REGION Network 6: Print Logic
   RUNG wire#powerrail
      Contact( #AlwaysTrue )
      wire#w1
      P_Contact(operand := #Selected, bit := #RE3)
      { S7_GenerateENO := "TRUE" } Move(in := 1, out1 => #PrintWord)   // 'STARTED'
      S_Move(in := #STATUS1, out => #PrintStatus)
      S_Coil( #PrintTriggerTemp )
   END_RUNG
   RUNG wire#w1
      Contact( #Selected )
      N_Contact(operand := #Running, bit := #RE4)
      I_Contact( #Close )
      { S7_GenerateENO := "TRUE" } Move(in := 2, out1 => #PrintWord)   // 'PAUSED'
      S_Move(in := #STATUS2, out => #PrintStatus)
      wire#w2
      S_Coil( #PrintTriggerTemp )
   END_RUNG
   RUNG wire#w2
      S_Coil( #Paused )
   END_RUNG
   RUNG wire#w1
      Contact( #Selected )
      Contact( #Paused )
      P_Contact(operand := #Running, bit := #RE5)
      { S7_GenerateENO := "TRUE" } Move(in := 3, out1 => #PrintWord)   // 'RESUMED'
      S_Move(in := #STATUS3, out => #PrintStatus)
      wire#w3
      S_Coil( #PrintTriggerTemp )
   END_RUNG
   RUNG wire#w3
      R_Coil( #Paused )
   END_RUNG
   RUNG wire#w1
      P_Contact(operand := #SpargingOver, bit := #RE6)
      { S7_GenerateENO := "TRUE" } Move(in := 4, out1 => #PrintWord)   // 'OVER'
      S_Move(in := #STATUS4, out => #PrintStatus)
      S_Coil( #PrintTriggerTemp )
   END_RUNG
   RUNG wire#w1
      P_Contact(operand := #Close, bit := #RE7)
      { S7_GenerateENO := "TRUE" } Move(in := 5, out1 => #PrintWord)   // 'RESETED'
      S_Move(in := #STATUS5, out => #PrintStatus)
      S_Coil( #PrintTriggerTemp )
   END_RUNG
   RUNG wire#w1
      I_Contact( #Selected )
      R_Coil( #Paused )
   END_RUNG
   RUNG wire#w1
      Contact( #PrintTriggerTemp )
      Coil( #PrintTrigger )
   END_RUNG
   // the same network as SCL:
   // ENO of a box is taken as its EN; it also drops when the box reports an error
   #_w1 := #AlwaysTrue AND #Selected AND NOT #RE3;   // rising edge of #Selected
   #RE3 := #Selected;
   IF #_w1 THEN
       #PrintWord := 1;   // 'STARTED'
       #PrintStatus := #STATUS1;
       #PrintTriggerTemp := TRUE;
   END_IF;
   #_w2 := #AlwaysTrue AND #Selected AND NOT #Running AND #RE4;   // falling edge of #Running
   #RE4 := #Running;
   IF #_w2 AND NOT #Close THEN
       #PrintWord := 2;   // 'PAUSED'
       #PrintStatus := #STATUS2;
       #PrintTriggerTemp := TRUE;
       #Paused := TRUE;
   END_IF;
   #_w3 := #AlwaysTrue AND #Selected AND #Paused AND #Running AND NOT #RE5;   // rising edge of #Running
   #RE5 := #Running;
   IF #_w3 THEN
       #PrintWord := 3;   // 'RESUMED'
       #PrintStatus := #STATUS3;
       #PrintTriggerTemp := TRUE;
       #Paused := FALSE;
   END_IF;
   #_w4 := #AlwaysTrue AND #SpargingOver AND NOT #RE6;   // rising edge of #SpargingOver
   #RE6 := #SpargingOver;
   IF #_w4 THEN
       #PrintWord := 4;   // 'OVER'
       #PrintStatus := #STATUS4;
       #PrintTriggerTemp := TRUE;
   END_IF;
   #_w5 := #AlwaysTrue AND #Close AND NOT #RE7;   // rising edge of #Close
   #RE7 := #Close;
   IF #_w5 THEN
       #PrintWord := 5;   // 'RESETED'
       #PrintStatus := #STATUS5;
       #PrintTriggerTemp := TRUE;
   END_IF;
   IF #AlwaysTrue AND NOT #Selected THEN #Paused := FALSE; END_IF;
   #PrintTrigger := #AlwaysTrue AND #PrintTriggerTemp;
END_REGION

REGION Network 7: Print Trigger Reset
   RUNG wire#powerrail
      Contact( #PrintTriggerTemp )
      { S7_Templates := "time_type := Time" } #PrintTriggerResetTimer.TON(pt := T#1s, et =>)
      R_Coil( #PrintTriggerTemp )
   END_RUNG
   // the same network as SCL:
   #PrintTriggerResetTimer(IN := #PrintTriggerTemp, PT := T#1s);   // TON
   IF #PrintTriggerResetTimer.Q THEN #PrintTriggerTemp := FALSE; END_IF;
END_REGION

REGION Network 8: Button Reset
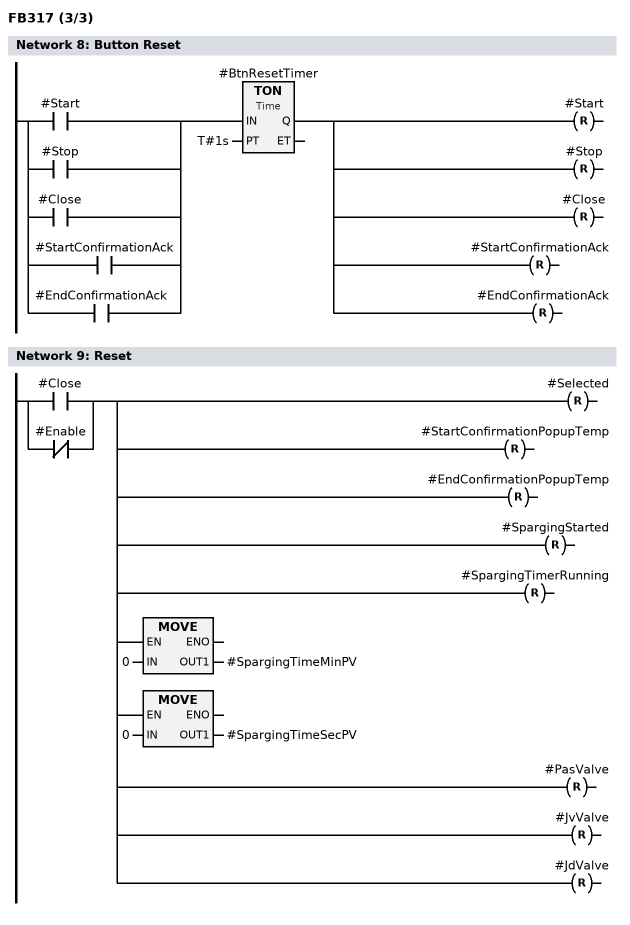
   RUNG wire#powerrail
      Contact( #Start )
      wire#w1
      { S7_Templates := "time_type := Time" } #BtnResetTimer.TON(pt := T#1s, et =>)
      wire#w2
      R_Coil( #Start )
   END_RUNG
   RUNG wire#powerrail
      Contact( #Stop )
   END_RUNG wire#w1
   RUNG wire#powerrail
      Contact( #Close )
   END_RUNG wire#w1
   RUNG wire#powerrail
      Contact( #StartConfirmationAck )
   END_RUNG wire#w1
   RUNG wire#powerrail
      Contact( #EndConfirmationAck )
   END_RUNG wire#w1
   RUNG wire#w2
      R_Coil( #Stop )
   END_RUNG
   RUNG wire#w2
      R_Coil( #Close )
   END_RUNG
   RUNG wire#w2
      R_Coil( #StartConfirmationAck )
   END_RUNG
   RUNG wire#w2
      R_Coil( #EndConfirmationAck )
   END_RUNG
   // the same network as SCL:
   #BtnResetTimer(IN := #Start OR #Stop OR #Close OR #StartConfirmationAck OR #EndConfirmationAck, PT := T#1s);   // TON
   IF #BtnResetTimer.Q THEN
       #Start := FALSE;
       #Stop := FALSE;
       #Close := FALSE;
       #StartConfirmationAck := FALSE;
       #EndConfirmationAck := FALSE;
   END_IF;
END_REGION

REGION Network 9: Reset
   RUNG wire#powerrail
      Contact( #Close )
      wire#w1
      R_Coil( #Selected )
   END_RUNG
   RUNG wire#powerrail
      I_Contact( #Enable )
   END_RUNG wire#w1
   RUNG wire#w1
      R_Coil( #StartConfirmationPopupTemp )
   END_RUNG
   RUNG wire#w1
      R_Coil( #EndConfirmationPopupTemp )
   END_RUNG
   RUNG wire#w1
      R_Coil( #SpargingStarted )
   END_RUNG
   RUNG wire#w1
      R_Coil( #SpargingTimerRunning )
   END_RUNG
   RUNG wire#w1
      { S7_GenerateENO := "TRUE" } Move(in := 0, out1 => #SpargingTimeMinPV)
   END_RUNG
   RUNG wire#w1
      { S7_GenerateENO := "TRUE" } Move(in := 0, out1 => #SpargingTimeSecPV)
   END_RUNG
   RUNG wire#w1
      R_Coil( #PasValve )
   END_RUNG
   RUNG wire#w1
      R_Coil( #JvValve )
   END_RUNG
   RUNG wire#w1
      R_Coil( #JdValve )
   END_RUNG
   // the same network as SCL:
   IF #Close OR NOT #Enable THEN
       #Selected := FALSE;
       #StartConfirmationPopupTemp := FALSE;
       #EndConfirmationPopupTemp := FALSE;
       #SpargingStarted := FALSE;
       #SpargingTimerRunning := FALSE;
       #SpargingTimeMinPV := 0;
       #SpargingTimeSecPV := 0;
       #PasValve := FALSE;
       #JvValve := FALSE;
       #JdValve := FALSE;
   END_IF;
END_REGION
END_FUNCTION_BLOCK

FUNCTION_BLOCK "BATCH LINE PRINT"   // FB5, LAD
{ S7_Optimized_Access := 'TRUE' }
// stored: MemoryReserve 100, SetENOAutomatically false
   VAR_INPUT
      PrintInetrval : Int;
      SecPulse : Bool;
   END_VAR
   VAR_IN_OUT
      ResetBatchTimer : Bool;
      BatchSelected : Bool;
   END_VAR
   VAR
      IEC_Counter_0_Instance { S7_SetPoint := 'True'} : CTU_INT;
   END_VAR
BEGIN

REGION Network 2
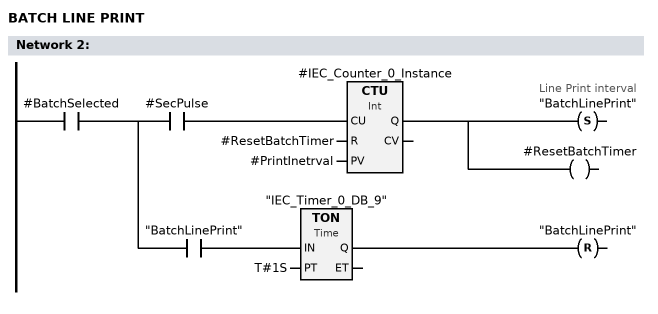
   RUNG wire#powerrail
      Contact( #BatchSelected )
      wire#w1
      Contact( #SecPulse )
      { S7_Templates := "value_type := Int" } #IEC_Counter_0_Instance.CTU(r := #ResetBatchTimer, pv := #PrintInetrval, cv =>)
      wire#w2
      S_Coil( "BatchLinePrint" )   // Line Print interval
   END_RUNG
   RUNG wire#w2
      Coil( #ResetBatchTimer )
   END_RUNG
   RUNG wire#w1
      Contact( "BatchLinePrint" )
      { S7_Templates := "time_type := Time" } "IEC_Timer_0_DB_9".TON(pt := T#1S, et =>)
      R_Coil( "BatchLinePrint" )
   END_RUNG
   // the same network as SCL:
   #IEC_Counter_0_Instance(CU := #BatchSelected AND #SecPulse, R := #ResetBatchTimer, PV := #PrintInetrval);   // CTU
   IF #IEC_Counter_0_Instance.Q THEN
       "BatchLinePrint" := TRUE;   // Line Print interval
   END_IF;
   #ResetBatchTimer := #IEC_Counter_0_Instance.Q;
   "IEC_Timer_0_DB_9".TON(IN := #BatchSelected AND "BatchLinePrint", PT := T#1S);
   IF "IEC_Timer_0_DB_9".Q THEN "BatchLinePrint" := FALSE; END_IF;
END_REGION
END_FUNCTION_BLOCK

FUNCTION "BatchValves" : Void   // FC302, LAD
{ S7_Optimized_Access := 'TRUE' }
// stored: AutoNumber false, SetENOAutomatically false
BEGIN

REGION Network 1: ***************FILL WFI *****************
END_REGION

REGION Network 2: "BatchVessel".Cv02 ----- Wfi
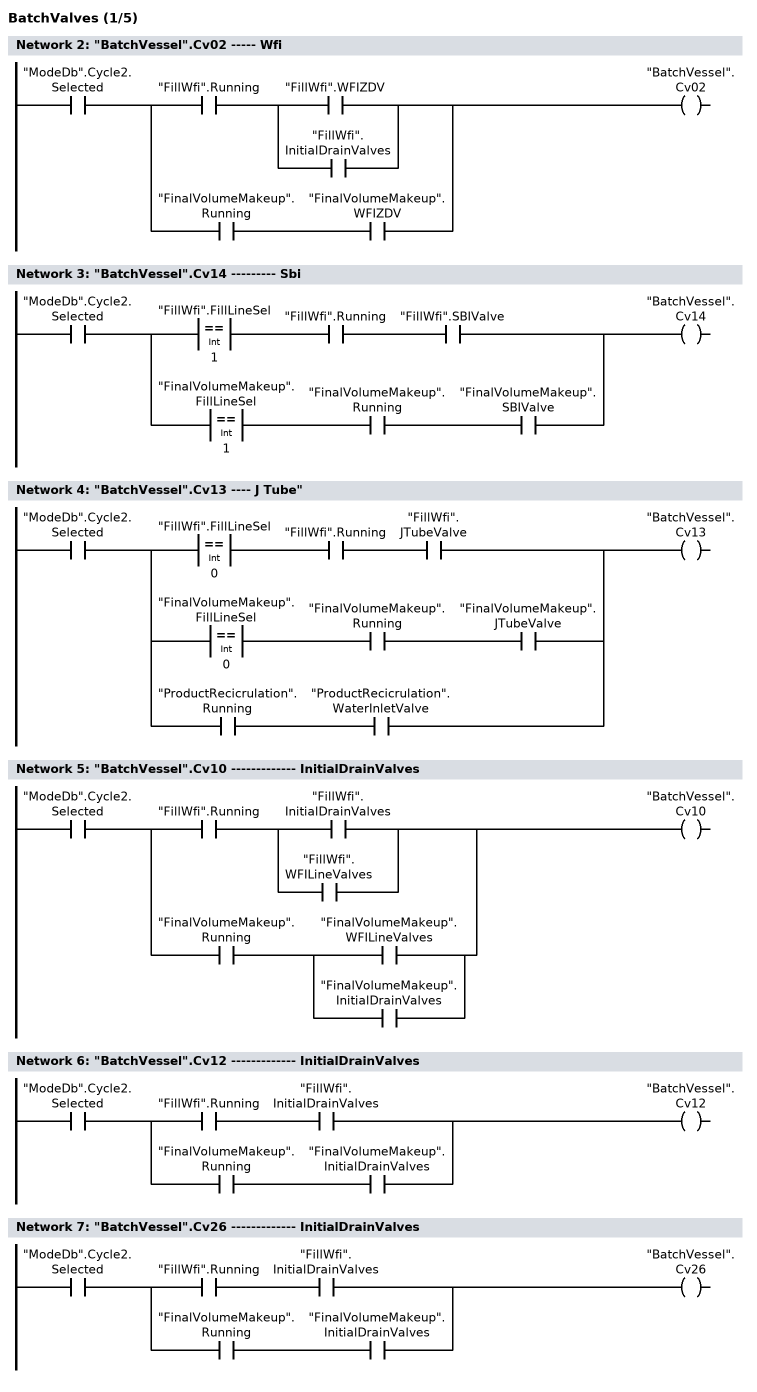
   RUNG wire#powerrail
      Contact( "ModeDb".Cycle2.Selected )
      wire#w1
      Contact( "FillWfi".Running )
      wire#w2
      Contact( "FillWfi".WFIZDV )
      wire#w3
      Coil( "BatchVessel".Cv02 )
   END_RUNG
   RUNG wire#w2
      Contact( "FillWfi".InitialDrainValves )
   END_RUNG wire#w3
   RUNG wire#w1
      Contact( "FinalVolumeMakeup".Running )
      Contact( "FinalVolumeMakeup".WFIZDV )
   END_RUNG wire#w3
   // the same network as SCL:
   "BatchVessel".Cv02 := "ModeDb".Cycle2.Selected AND (("FillWfi".Running AND ("FillWfi".WFIZDV OR "FillWfi".InitialDrainValves)) OR ("FinalVolumeMakeup".Running AND "FinalVolumeMakeup".WFIZDV));
END_REGION

REGION Network 3: "BatchVessel".Cv14 --------- Sbi
   RUNG wire#powerrail
      Contact( "ModeDb".Cycle2.Selected )
      wire#w1
      { S7_Templates := "SrcType := Int" } EQ_Contact(in1 := "FillWfi".FillLineSel, in2 := 1)
      Contact( "FillWfi".Running )
      Contact( "FillWfi".SBIValve )
      wire#w2
      Coil( "BatchVessel".Cv14 )
   END_RUNG
   RUNG wire#w1
      { S7_Templates := "SrcType := Int" } EQ_Contact(in1 := "FinalVolumeMakeup".FillLineSel, in2 := 1)
      Contact( "FinalVolumeMakeup".Running )
      Contact( "FinalVolumeMakeup".SBIValve )
   END_RUNG wire#w2
   // the same network as SCL:
   "BatchVessel".Cv14 := "ModeDb".Cycle2.Selected AND ((("FillWfi".FillLineSel = 1) AND "FillWfi".Running AND "FillWfi".SBIValve) OR (("FinalVolumeMakeup".FillLineSel = 1) AND "FinalVolumeMakeup".Running AND "FinalVolumeMakeup".SBIValve));
END_REGION

REGION Network 4: "BatchVessel".Cv13 ---- J Tube"
   RUNG wire#powerrail
      Contact( "ModeDb".Cycle2.Selected )
      wire#w1
      { S7_Templates := "SrcType := Int" } EQ_Contact(in1 := "FillWfi".FillLineSel, in2 := 0)
      Contact( "FillWfi".Running )
      Contact( "FillWfi".JTubeValve )
      wire#w2
      Coil( "BatchVessel".Cv13 )
   END_RUNG
   RUNG wire#w1
      { S7_Templates := "SrcType := Int" } EQ_Contact(in1 := "FinalVolumeMakeup".FillLineSel, in2 := 0)
      Contact( "FinalVolumeMakeup".Running )
      Contact( "FinalVolumeMakeup".JTubeValve )
   END_RUNG wire#w2
   RUNG wire#w1
      Contact( "ProductRecicrulation".Running )
      Contact( "ProductRecicrulation".WaterInletValve )
   END_RUNG wire#w2
   // the same network as SCL:
   "BatchVessel".Cv13 := "ModeDb".Cycle2.Selected AND ((("FillWfi".FillLineSel = 0) AND "FillWfi".Running AND "FillWfi".JTubeValve) OR (("FinalVolumeMakeup".FillLineSel = 0) AND "FinalVolumeMakeup".Running AND "FinalVolumeMakeup".JTubeValve) OR ("ProductRecicrulation".Running AND "ProductRecicrulation".WaterInletValve));
END_REGION

REGION Network 5: "BatchVessel".Cv10 ------------- InitialDrainValves
   RUNG wire#powerrail
      Contact( "ModeDb".Cycle2.Selected )
      wire#w1
      Contact( "FillWfi".Running )
      wire#w2
      Contact( "FillWfi".InitialDrainValves )
      wire#w3
      Coil( "BatchVessel".Cv10 )
   END_RUNG
   RUNG wire#w2
      Contact( "FillWfi".WFILineValves )
   END_RUNG wire#w3
   RUNG wire#w1
      Contact( "FinalVolumeMakeup".Running )
      wire#w4
      Contact( "FinalVolumeMakeup".WFILineValves )
   END_RUNG wire#w3
   RUNG wire#w4
      Contact( "FinalVolumeMakeup".InitialDrainValves )
   END_RUNG wire#w3
   // the same network as SCL:
   "BatchVessel".Cv10 := "ModeDb".Cycle2.Selected AND (("FillWfi".Running AND ("FillWfi".InitialDrainValves OR "FillWfi".WFILineValves)) OR ("FinalVolumeMakeup".Running AND ("FinalVolumeMakeup".WFILineValves OR "FinalVolumeMakeup".InitialDrainValves)));
END_REGION

REGION Network 6: "BatchVessel".Cv12 ------------- InitialDrainValves
   RUNG wire#powerrail
      Contact( "ModeDb".Cycle2.Selected )
      wire#w1
      Contact( "FillWfi".Running )
      Contact( "FillWfi".InitialDrainValves )
      wire#w2
      Coil( "BatchVessel".Cv12 )
   END_RUNG
   RUNG wire#w1
      Contact( "FinalVolumeMakeup".Running )
      Contact( "FinalVolumeMakeup".InitialDrainValves )
   END_RUNG wire#w2
   // the same network as SCL:
   "BatchVessel".Cv12 := "ModeDb".Cycle2.Selected AND (("FillWfi".Running AND "FillWfi".InitialDrainValves) OR ("FinalVolumeMakeup".Running AND "FinalVolumeMakeup".InitialDrainValves));
END_REGION

REGION Network 7: "BatchVessel".Cv26 ------------- InitialDrainValves
   RUNG wire#powerrail
      Contact( "ModeDb".Cycle2.Selected )
      wire#w1
      Contact( "FillWfi".Running )
      Contact( "FillWfi".InitialDrainValves )
      wire#w2
      Coil( "BatchVessel".Cv26 )
   END_RUNG
   RUNG wire#w1
      Contact( "FinalVolumeMakeup".Running )
      Contact( "FinalVolumeMakeup".InitialDrainValves )
   END_RUNG wire#w2
   // the same network as SCL:
   "BatchVessel".Cv26 := "ModeDb".Cycle2.Selected AND (("FillWfi".Running AND "FillWfi".InitialDrainValves) OR ("FinalVolumeMakeup".Running AND "FinalVolumeMakeup".InitialDrainValves));
END_REGION

REGION Network 8: "BatchVessel".Fbov01 ------------- InitialDrainValves
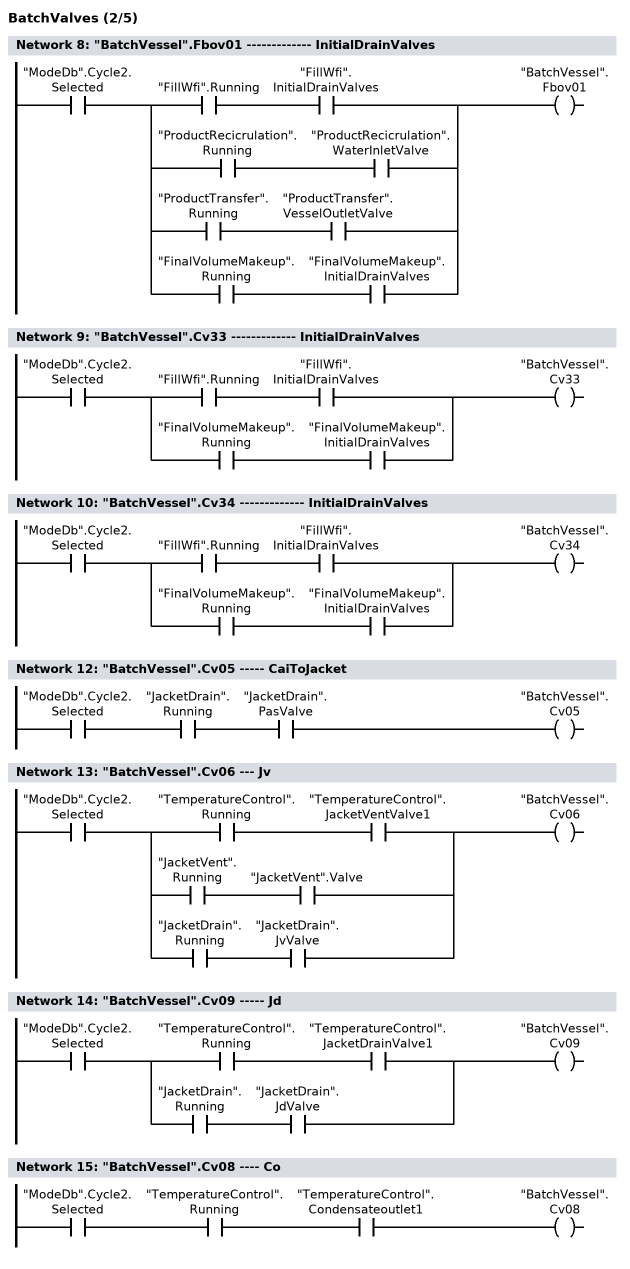
   RUNG wire#powerrail
      Contact( "ModeDb".Cycle2.Selected )
      wire#w1
      Contact( "FillWfi".Running )
      Contact( "FillWfi".InitialDrainValves )
      wire#w2
      Coil( "BatchVessel".Fbov01 )
   END_RUNG
   RUNG wire#w1
      Contact( "ProductRecicrulation".Running )
      Contact( "ProductRecicrulation".WaterInletValve )
   END_RUNG wire#w2
   RUNG wire#w1
      Contact( "ProductTransfer".Running )
      Contact( "ProductTransfer".VesselOutletValve )
   END_RUNG wire#w2
   RUNG wire#w1
      Contact( "FinalVolumeMakeup".Running )
      Contact( "FinalVolumeMakeup".InitialDrainValves )
   END_RUNG wire#w2
   // the same network as SCL:
   "BatchVessel".Fbov01 := "ModeDb".Cycle2.Selected AND (("FillWfi".Running AND "FillWfi".InitialDrainValves) OR ("ProductRecicrulation".Running AND "ProductRecicrulation".WaterInletValve) OR ("ProductTransfer".Running AND "ProductTransfer".VesselOutletValve) OR ("FinalVolumeMakeup".Running AND "FinalVolumeMakeup".InitialDrainValves));
END_REGION

REGION Network 9: "BatchVessel".Cv33 ------------- InitialDrainValves
   RUNG wire#powerrail
      Contact( "ModeDb".Cycle2.Selected )
      wire#w1
      Contact( "FillWfi".Running )
      Contact( "FillWfi".InitialDrainValves )
      wire#w2
      Coil( "BatchVessel".Cv33 )
   END_RUNG
   RUNG wire#w1
      Contact( "FinalVolumeMakeup".Running )
      Contact( "FinalVolumeMakeup".InitialDrainValves )
   END_RUNG wire#w2
   // the same network as SCL:
   "BatchVessel".Cv33 := "ModeDb".Cycle2.Selected AND (("FillWfi".Running AND "FillWfi".InitialDrainValves) OR ("FinalVolumeMakeup".Running AND "FinalVolumeMakeup".InitialDrainValves));
END_REGION

REGION Network 10: "BatchVessel".Cv34 ------------- InitialDrainValves
   RUNG wire#powerrail
      Contact( "ModeDb".Cycle2.Selected )
      wire#w1
      Contact( "FillWfi".Running )
      Contact( "FillWfi".InitialDrainValves )
      wire#w2
      Coil( "BatchVessel".Cv34 )
   END_RUNG
   RUNG wire#w1
      Contact( "FinalVolumeMakeup".Running )
      Contact( "FinalVolumeMakeup".InitialDrainValves )
   END_RUNG wire#w2
   // the same network as SCL:
   "BatchVessel".Cv34 := "ModeDb".Cycle2.Selected AND (("FillWfi".Running AND "FillWfi".InitialDrainValves) OR ("FinalVolumeMakeup".Running AND "FinalVolumeMakeup".InitialDrainValves));
END_REGION

REGION Network 11: ***************TEMPERATURE CONTROL *****************
END_REGION

REGION Network 12: "BatchVessel".Cv05 ----- CaiToJacket
   RUNG wire#powerrail
      Contact( "ModeDb".Cycle2.Selected )
      Contact( "JacketDrain".Running )
      Contact( "JacketDrain".PasValve )
      Coil( "BatchVessel".Cv05 )
   END_RUNG
   // the same network as SCL:
   "BatchVessel".Cv05 := "ModeDb".Cycle2.Selected AND "JacketDrain".Running AND "JacketDrain".PasValve;
END_REGION

REGION Network 13: "BatchVessel".Cv06 --- Jv
   RUNG wire#powerrail
      Contact( "ModeDb".Cycle2.Selected )
      wire#w1
      Contact( "TemperatureControl".Running )
      Contact( "TemperatureControl".JacketVentValve1 )
      wire#w2
      Coil( "BatchVessel".Cv06 )
   END_RUNG
   RUNG wire#w1
      Contact( "JacketVent".Running )
      Contact( "JacketVent".Valve )
   END_RUNG wire#w2
   RUNG wire#w1
      Contact( "JacketDrain".Running )
      Contact( "JacketDrain".JvValve )
   END_RUNG wire#w2
   // the same network as SCL:
   "BatchVessel".Cv06 := "ModeDb".Cycle2.Selected AND (("TemperatureControl".Running AND "TemperatureControl".JacketVentValve1) OR ("JacketVent".Running AND "JacketVent".Valve) OR ("JacketDrain".Running AND "JacketDrain".JvValve));
END_REGION

REGION Network 14: "BatchVessel".Cv09 ----- Jd
   RUNG wire#powerrail
      Contact( "ModeDb".Cycle2.Selected )
      wire#w1
      Contact( "TemperatureControl".Running )
      Contact( "TemperatureControl".JacketDrainValve1 )
      wire#w2
      Coil( "BatchVessel".Cv09 )
   END_RUNG
   RUNG wire#w1
      Contact( "JacketDrain".Running )
      Contact( "JacketDrain".JdValve )
   END_RUNG wire#w2
   // the same network as SCL:
   "BatchVessel".Cv09 := "ModeDb".Cycle2.Selected AND (("TemperatureControl".Running AND "TemperatureControl".JacketDrainValve1) OR ("JacketDrain".Running AND "JacketDrain".JdValve));
END_REGION

REGION Network 15: "BatchVessel".Cv08 ---- Co
   RUNG wire#powerrail
      Contact( "ModeDb".Cycle2.Selected )
      Contact( "TemperatureControl".Running )
      Contact( "TemperatureControl".Condensateoutlet1 )
      Coil( "BatchVessel".Cv08 )
   END_RUNG
   // the same network as SCL:
   "BatchVessel".Cv08 := "ModeDb".Cycle2.Selected AND "TemperatureControl".Running AND "TemperatureControl".Condensateoutlet1;
END_REGION

REGION Network 16: "BatchVessel".Cv04 ---- Psi
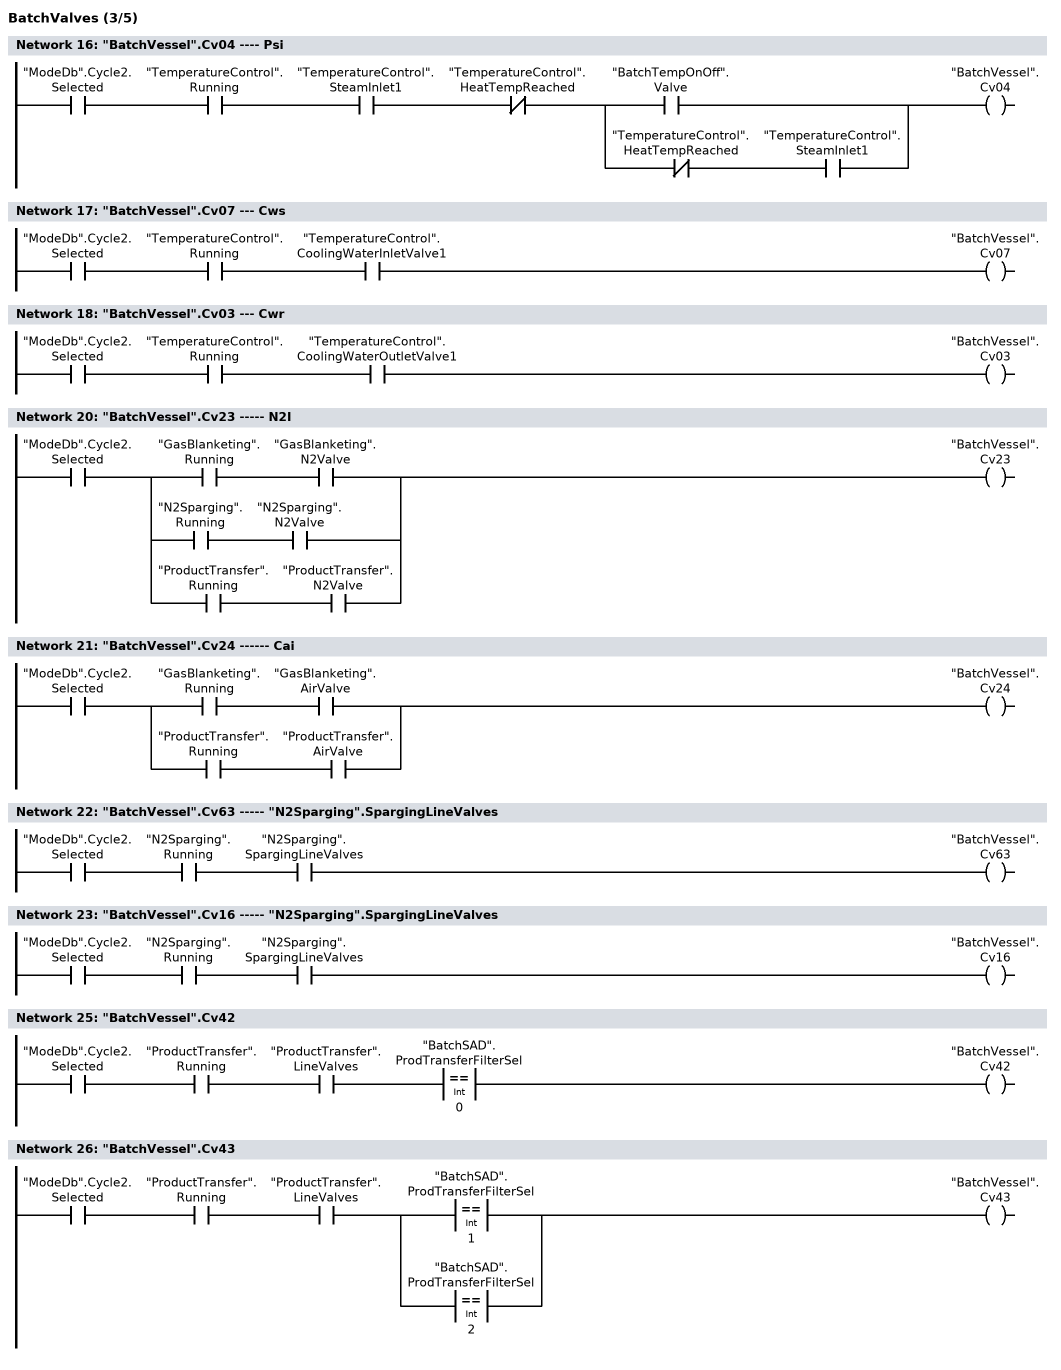
   RUNG wire#powerrail
      Contact( "ModeDb".Cycle2.Selected )
      Contact( "TemperatureControl".Running )
      Contact( "TemperatureControl".SteamInlet1 )
      I_Contact( "TemperatureControl".HeatTempReached )
      wire#w1
      Contact( "BatchTempOnOff".Valve )
      wire#w2
      Coil( "BatchVessel".Cv04 )
   END_RUNG
   RUNG wire#w1
      I_Contact( "TemperatureControl".HeatTempReached )
      Contact( "TemperatureControl".SteamInlet1 )
   END_RUNG wire#w2
   // the same network as SCL:
   "BatchVessel".Cv04 := "ModeDb".Cycle2.Selected AND "TemperatureControl".Running AND "TemperatureControl".SteamInlet1 AND NOT "TemperatureControl".HeatTempReached AND ("BatchTempOnOff".Valve OR (NOT "TemperatureControl".HeatTempReached AND "TemperatureControl".SteamInlet1));
END_REGION

REGION Network 17: "BatchVessel".Cv07 --- Cws
   RUNG wire#powerrail
      Contact( "ModeDb".Cycle2.Selected )
      Contact( "TemperatureControl".Running )
      Contact( "TemperatureControl".CoolingWaterInletValve1 )
      Coil( "BatchVessel".Cv07 )
   END_RUNG
   // the same network as SCL:
   "BatchVessel".Cv07 := "ModeDb".Cycle2.Selected AND "TemperatureControl".Running AND "TemperatureControl".CoolingWaterInletValve1;
END_REGION

REGION Network 18: "BatchVessel".Cv03 --- Cwr
   RUNG wire#powerrail
      Contact( "ModeDb".Cycle2.Selected )
      Contact( "TemperatureControl".Running )
      Contact( "TemperatureControl".CoolingWaterOutletValve1 )
      Coil( "BatchVessel".Cv03 )
   END_RUNG
   // the same network as SCL:
   "BatchVessel".Cv03 := "ModeDb".Cycle2.Selected AND "TemperatureControl".Running AND "TemperatureControl".CoolingWaterOutletValve1;
END_REGION

REGION Network 19: ***************GAS BLANKETING********N2 SPARGING*********
END_REGION

REGION Network 20: "BatchVessel".Cv23 ----- N2I
   RUNG wire#powerrail
      Contact( "ModeDb".Cycle2.Selected )
      wire#w1
      Contact( "GasBlanketing".Running )
      Contact( "GasBlanketing".N2Valve )
      wire#w2
      Coil( "BatchVessel".Cv23 )
   END_RUNG
   RUNG wire#w1
      Contact( "N2Sparging".Running )
      Contact( "N2Sparging".N2Valve )
   END_RUNG wire#w2
   RUNG wire#w1
      Contact( "ProductTransfer".Running )
      Contact( "ProductTransfer".N2Valve )
   END_RUNG wire#w2
   // the same network as SCL:
   "BatchVessel".Cv23 := "ModeDb".Cycle2.Selected AND (("GasBlanketing".Running AND "GasBlanketing".N2Valve) OR ("N2Sparging".Running AND "N2Sparging".N2Valve) OR ("ProductTransfer".Running AND "ProductTransfer".N2Valve));
END_REGION

REGION Network 21: "BatchVessel".Cv24 ------ Cai
   RUNG wire#powerrail
      Contact( "ModeDb".Cycle2.Selected )
      wire#w1
      Contact( "GasBlanketing".Running )
      Contact( "GasBlanketing".AirValve )
      wire#w2
      Coil( "BatchVessel".Cv24 )
   END_RUNG
   RUNG wire#w1
      Contact( "ProductTransfer".Running )
      Contact( "ProductTransfer".AirValve )
   END_RUNG wire#w2
   // the same network as SCL:
   "BatchVessel".Cv24 := "ModeDb".Cycle2.Selected AND (("GasBlanketing".Running AND "GasBlanketing".AirValve) OR ("ProductTransfer".Running AND "ProductTransfer".AirValve));
END_REGION

REGION Network 22: "BatchVessel".Cv63 ----- "N2Sparging".SpargingLineValves
   RUNG wire#powerrail
      Contact( "ModeDb".Cycle2.Selected )
      Contact( "N2Sparging".Running )
      Contact( "N2Sparging".SpargingLineValves )
      Coil( "BatchVessel".Cv63 )
   END_RUNG
   // the same network as SCL:
   "BatchVessel".Cv63 := "ModeDb".Cycle2.Selected AND "N2Sparging".Running AND "N2Sparging".SpargingLineValves;
END_REGION

REGION Network 23: "BatchVessel".Cv16 ----- "N2Sparging".SpargingLineValves
   RUNG wire#powerrail
      Contact( "ModeDb".Cycle2.Selected )
      Contact( "N2Sparging".Running )
      Contact( "N2Sparging".SpargingLineValves )
      Coil( "BatchVessel".Cv16 )
   END_RUNG
   // the same network as SCL:
   "BatchVessel".Cv16 := "ModeDb".Cycle2.Selected AND "N2Sparging".Running AND "N2Sparging".SpargingLineValves;
END_REGION

REGION Network 24: ***************PRODUCT TRANSFER*****************
END_REGION

REGION Network 25: "BatchVessel".Cv42
   RUNG wire#powerrail
      Contact( "ModeDb".Cycle2.Selected )
      Contact( "ProductTransfer".Running )
      Contact( "ProductTransfer".LineValves )
      { S7_Templates := "SrcType := Int" } EQ_Contact(in1 := "BatchSAD".ProdTransferFilterSel, in2 := 0)
      Coil( "BatchVessel".Cv42 )
   END_RUNG
   // the same network as SCL:
   "BatchVessel".Cv42 := "ModeDb".Cycle2.Selected AND "ProductTransfer".Running AND "ProductTransfer".LineValves AND ("BatchSAD".ProdTransferFilterSel = 0);
END_REGION

REGION Network 26: "BatchVessel".Cv43
   RUNG wire#powerrail
      Contact( "ModeDb".Cycle2.Selected )
      Contact( "ProductTransfer".Running )
      Contact( "ProductTransfer".LineValves )
      wire#w1
      { S7_Templates := "SrcType := Int" } EQ_Contact(in1 := "BatchSAD".ProdTransferFilterSel, in2 := 1)
      wire#w2
      Coil( "BatchVessel".Cv43 )
   END_RUNG
   RUNG wire#w1
      { S7_Templates := "SrcType := Int" } EQ_Contact(in1 := "BatchSAD".ProdTransferFilterSel, in2 := 2)
   END_RUNG wire#w2
   // the same network as SCL:
   "BatchVessel".Cv43 := "ModeDb".Cycle2.Selected AND "ProductTransfer".Running AND "ProductTransfer".LineValves AND (("BatchSAD".ProdTransferFilterSel = 1) OR ("BatchSAD".ProdTransferFilterSel = 2));
END_REGION

REGION Network 27: "BatchVessel".Cv48
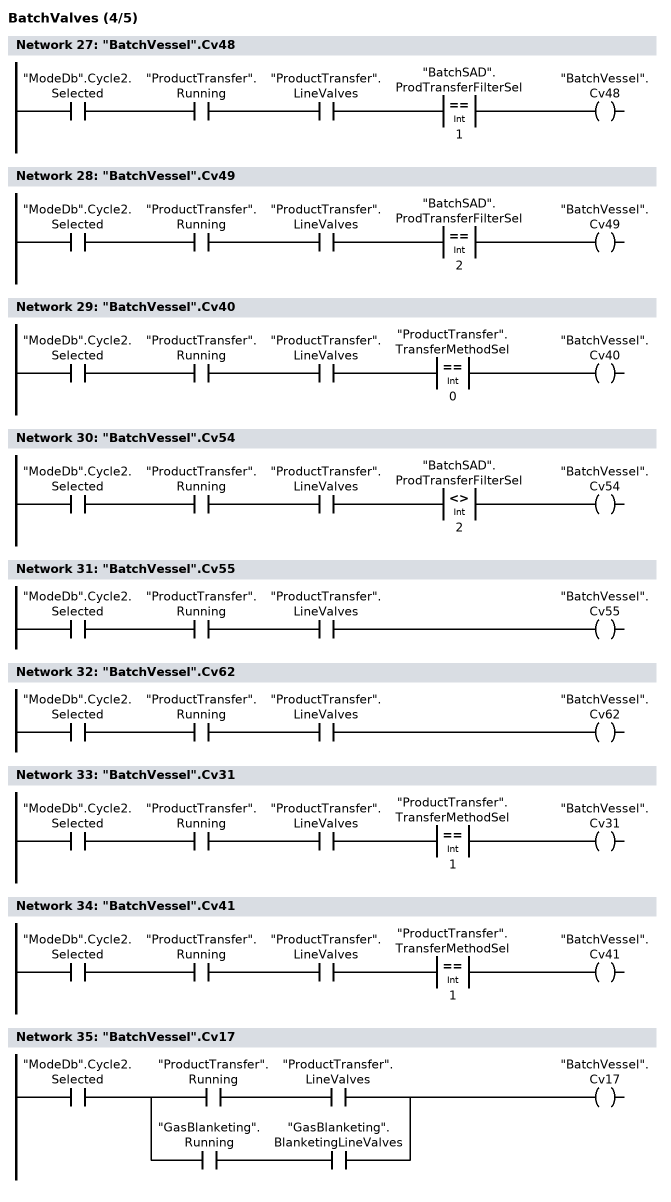
   RUNG wire#powerrail
      Contact( "ModeDb".Cycle2.Selected )
      Contact( "ProductTransfer".Running )
      Contact( "ProductTransfer".LineValves )
      { S7_Templates := "SrcType := Int" } EQ_Contact(in1 := "BatchSAD".ProdTransferFilterSel, in2 := 1)
      Coil( "BatchVessel".Cv48 )
   END_RUNG
   // the same network as SCL:
   "BatchVessel".Cv48 := "ModeDb".Cycle2.Selected AND "ProductTransfer".Running AND "ProductTransfer".LineValves AND ("BatchSAD".ProdTransferFilterSel = 1);
END_REGION

REGION Network 28: "BatchVessel".Cv49
   RUNG wire#powerrail
      Contact( "ModeDb".Cycle2.Selected )
      Contact( "ProductTransfer".Running )
      Contact( "ProductTransfer".LineValves )
      { S7_Templates := "SrcType := Int" } EQ_Contact(in1 := "BatchSAD".ProdTransferFilterSel, in2 := 2)
      Coil( "BatchVessel".Cv49 )
   END_RUNG
   // the same network as SCL:
   "BatchVessel".Cv49 := "ModeDb".Cycle2.Selected AND "ProductTransfer".Running AND "ProductTransfer".LineValves AND ("BatchSAD".ProdTransferFilterSel = 2);
END_REGION

REGION Network 29: "BatchVessel".Cv40
   RUNG wire#powerrail
      Contact( "ModeDb".Cycle2.Selected )
      Contact( "ProductTransfer".Running )
      Contact( "ProductTransfer".LineValves )
      { S7_Templates := "SrcType := Int" } EQ_Contact(in1 := "ProductTransfer".TransferMethodSel, in2 := 0)
      Coil( "BatchVessel".Cv40 )
   END_RUNG
   // the same network as SCL:
   "BatchVessel".Cv40 := "ModeDb".Cycle2.Selected AND "ProductTransfer".Running AND "ProductTransfer".LineValves AND ("ProductTransfer".TransferMethodSel = 0);
END_REGION

REGION Network 30: "BatchVessel".Cv54
   RUNG wire#powerrail
      Contact( "ModeDb".Cycle2.Selected )
      Contact( "ProductTransfer".Running )
      Contact( "ProductTransfer".LineValves )
      { S7_Templates := "SrcType := Int" } NE_Contact(in1 := "BatchSAD".ProdTransferFilterSel, in2 := 2)
      Coil( "BatchVessel".Cv54 )
   END_RUNG
   // the same network as SCL:
   "BatchVessel".Cv54 := "ModeDb".Cycle2.Selected AND "ProductTransfer".Running AND "ProductTransfer".LineValves AND ("BatchSAD".ProdTransferFilterSel <> 2);
END_REGION

REGION Network 31: "BatchVessel".Cv55
   RUNG wire#powerrail
      Contact( "ModeDb".Cycle2.Selected )
      Contact( "ProductTransfer".Running )
      Contact( "ProductTransfer".LineValves )
      Coil( "BatchVessel".Cv55 )
   END_RUNG
   // the same network as SCL:
   "BatchVessel".Cv55 := "ModeDb".Cycle2.Selected AND "ProductTransfer".Running AND "ProductTransfer".LineValves;
END_REGION

REGION Network 32: "BatchVessel".Cv62
   RUNG wire#powerrail
      Contact( "ModeDb".Cycle2.Selected )
      Contact( "ProductTransfer".Running )
      Contact( "ProductTransfer".LineValves )
      Coil( "BatchVessel".Cv62 )
   END_RUNG
   // the same network as SCL:
   "BatchVessel".Cv62 := "ModeDb".Cycle2.Selected AND "ProductTransfer".Running AND "ProductTransfer".LineValves;
END_REGION

REGION Network 33: "BatchVessel".Cv31
   RUNG wire#powerrail
      Contact( "ModeDb".Cycle2.Selected )
      Contact( "ProductTransfer".Running )
      Contact( "ProductTransfer".LineValves )
      { S7_Templates := "SrcType := Int" } EQ_Contact(in1 := "ProductTransfer".TransferMethodSel, in2 := 1)
      Coil( "BatchVessel".Cv31 )
   END_RUNG
   // the same network as SCL:
   "BatchVessel".Cv31 := "ModeDb".Cycle2.Selected AND "ProductTransfer".Running AND "ProductTransfer".LineValves AND ("ProductTransfer".TransferMethodSel = 1);
END_REGION

REGION Network 34: "BatchVessel".Cv41
   RUNG wire#powerrail
      Contact( "ModeDb".Cycle2.Selected )
      Contact( "ProductTransfer".Running )
      Contact( "ProductTransfer".LineValves )
      { S7_Templates := "SrcType := Int" } EQ_Contact(in1 := "ProductTransfer".TransferMethodSel, in2 := 1)
      Coil( "BatchVessel".Cv41 )
   END_RUNG
   // the same network as SCL:
   "BatchVessel".Cv41 := "ModeDb".Cycle2.Selected AND "ProductTransfer".Running AND "ProductTransfer".LineValves AND ("ProductTransfer".TransferMethodSel = 1);
END_REGION

REGION Network 35: "BatchVessel".Cv17
   RUNG wire#powerrail
      Contact( "ModeDb".Cycle2.Selected )
      wire#w1
      Contact( "ProductTransfer".Running )
      Contact( "ProductTransfer".LineValves )
      wire#w2
      Coil( "BatchVessel".Cv17 )
   END_RUNG
   RUNG wire#w1
      Contact( "GasBlanketing".Running )
      Contact( "GasBlanketing".BlanketingLineValves )
   END_RUNG wire#w2
   // the same network as SCL:
   "BatchVessel".Cv17 := "ModeDb".Cycle2.Selected AND (("ProductTransfer".Running AND "ProductTransfer".LineValves) OR ("GasBlanketing".Running AND "GasBlanketing".BlanketingLineValves));
END_REGION

REGION Network 36: ***************RM ADDITION*****************
END_REGION

REGION Network 37: "BatchVessel".Cv21 ---- Vent
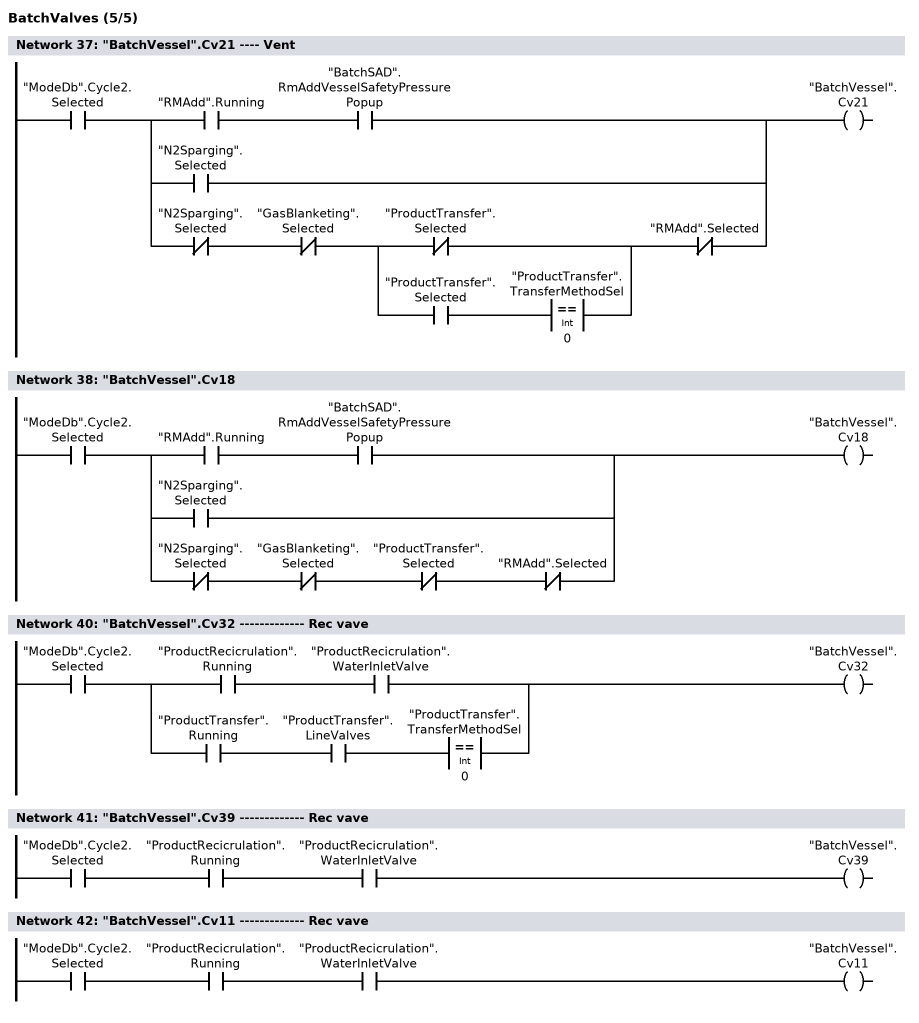
   RUNG wire#powerrail
      Contact( "ModeDb".Cycle2.Selected )
      wire#w1
      Contact( "RMAdd".Running )
      Contact( "BatchSAD".RmAddVesselSafetyPressurePopup )
      wire#w2
      Coil( "BatchVessel".Cv21 )
   END_RUNG
   RUNG wire#w1
      Contact( "N2Sparging".Selected )
   END_RUNG wire#w2
   RUNG wire#w1
      I_Contact( "N2Sparging".Selected )
      I_Contact( "GasBlanketing".Selected )
      wire#w3
      I_Contact( "ProductTransfer".Selected )
      wire#w4
      I_Contact( "RMAdd".Selected )
   END_RUNG wire#w2
   RUNG wire#w3
      Contact( "ProductTransfer".Selected )
      { S7_Templates := "SrcType := Int" } EQ_Contact(in1 := "ProductTransfer".TransferMethodSel, in2 := 0)
   END_RUNG wire#w4
   // the same network as SCL:
   "BatchVessel".Cv21 := "ModeDb".Cycle2.Selected AND (("RMAdd".Running AND "BatchSAD".RmAddVesselSafetyPressurePopup) OR "N2Sparging".Selected OR (NOT "N2Sparging".Selected AND NOT "GasBlanketing".Selected AND (NOT "ProductTransfer".Selected OR ("ProductTransfer".Selected AND ("ProductTransfer".TransferMethodSel = 0))) AND NOT "RMAdd".Selected));
END_REGION

REGION Network 38: "BatchVessel".Cv18
   RUNG wire#powerrail
      Contact( "ModeDb".Cycle2.Selected )
      wire#w1
      Contact( "RMAdd".Running )
      Contact( "BatchSAD".RmAddVesselSafetyPressurePopup )
      wire#w2
      Coil( "BatchVessel".Cv18 )
   END_RUNG
   RUNG wire#w1
      Contact( "N2Sparging".Selected )
   END_RUNG wire#w2
   RUNG wire#w1
      I_Contact( "N2Sparging".Selected )
      I_Contact( "GasBlanketing".Selected )
      I_Contact( "ProductTransfer".Selected )
      I_Contact( "RMAdd".Selected )
   END_RUNG wire#w2
   // the same network as SCL:
   "BatchVessel".Cv18 := "ModeDb".Cycle2.Selected AND (("RMAdd".Running AND "BatchSAD".RmAddVesselSafetyPressurePopup) OR "N2Sparging".Selected OR (NOT "N2Sparging".Selected AND NOT "GasBlanketing".Selected AND NOT "ProductTransfer".Selected AND NOT "RMAdd".Selected));
END_REGION

REGION Network 39: *************** PRODUCT RECIRCULATION *****************
END_REGION

REGION Network 40: "BatchVessel".Cv32 ------------- Rec vave
   RUNG wire#powerrail
      Contact( "ModeDb".Cycle2.Selected )
      wire#w1
      Contact( "ProductRecicrulation".Running )
      Contact( "ProductRecicrulation".WaterInletValve )
      wire#w2
      Coil( "BatchVessel".Cv32 )
   END_RUNG
   RUNG wire#w1
      Contact( "ProductTransfer".Running )
      Contact( "ProductTransfer".LineValves )
      { S7_Templates := "SrcType := Int" } EQ_Contact(in1 := "ProductTransfer".TransferMethodSel, in2 := 0)
   END_RUNG wire#w2
   // the same network as SCL:
   "BatchVessel".Cv32 := "ModeDb".Cycle2.Selected AND (("ProductRecicrulation".Running AND "ProductRecicrulation".WaterInletValve) OR ("ProductTransfer".Running AND "ProductTransfer".LineValves AND ("ProductTransfer".TransferMethodSel = 0)));
END_REGION

REGION Network 41: "BatchVessel".Cv39 ------------- Rec vave
   RUNG wire#powerrail
      Contact( "ModeDb".Cycle2.Selected )
      Contact( "ProductRecicrulation".Running )
      Contact( "ProductRecicrulation".WaterInletValve )
      Coil( "BatchVessel".Cv39 )
   END_RUNG
   // the same network as SCL:
   "BatchVessel".Cv39 := "ModeDb".Cycle2.Selected AND "ProductRecicrulation".Running AND "ProductRecicrulation".WaterInletValve;
END_REGION

REGION Network 42: "BatchVessel".Cv11 ------------- Rec vave
   RUNG wire#powerrail
      Contact( "ModeDb".Cycle2.Selected )
      Contact( "ProductRecicrulation".Running )
      Contact( "ProductRecicrulation".WaterInletValve )
      Coil( "BatchVessel".Cv11 )
   END_RUNG
   // the same network as SCL:
   "BatchVessel".Cv11 := "ModeDb".Cycle2.Selected AND "ProductRecicrulation".Running AND "ProductRecicrulation".WaterInletValve;
END_REGION
END_FUNCTION

FUNCTION "FC601" : Void   // FC601, LAD
TITLE = FC601
{ S7_Optimized_Access := 'TRUE' }
// MAIN CIP CALL BLOCK
// stored: AutoNumber false, SetENOAutomatically false
   VAR_TEMP   // added for the SCL form of the ladder/FBD networks
      _w1 : Bool;
      _w2 : Bool;
      _w3 : Bool;
   END_VAR
BEGIN

REGION Network 1: "FC604"
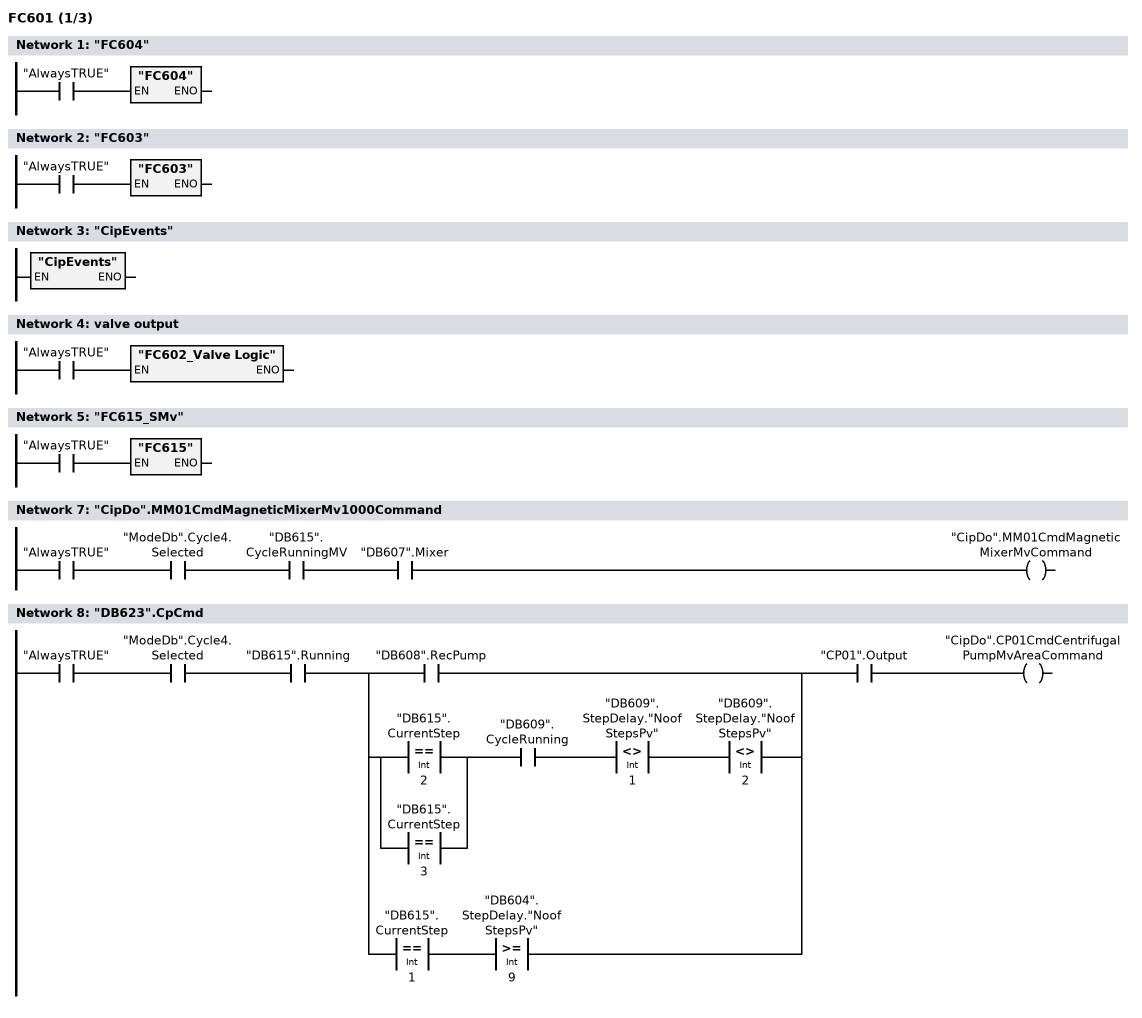
   RUNG wire#powerrail
      Contact( "AlwaysTRUE" )
      "FC604"()
   END_RUNG
   // the same network as SCL:
   IF "AlwaysTRUE" THEN "FC604"(); END_IF;
END_REGION

REGION Network 2: "FC603"
   RUNG wire#powerrail
      Contact( "AlwaysTRUE" )
      "FC603"()
   END_RUNG
   // the same network as SCL:
   IF "AlwaysTRUE" THEN "FC603"(); END_IF;
END_REGION

REGION Network 3: "CipEvents"
   RUNG wire#powerrail
      "CipEvents"()
   END_RUNG
   // the same network as SCL:
   "CipEvents"();
END_REGION

REGION Network 4: valve output
   RUNG wire#powerrail
      Contact( "AlwaysTRUE" )
      "FC602_Valve Logic"()
   END_RUNG
   // the same network as SCL:
   IF "AlwaysTRUE" THEN "FC602_Valve Logic"(); END_IF;
END_REGION

REGION Network 5: "FC615_SMv"
   RUNG wire#powerrail
      Contact( "AlwaysTRUE" )
      "FC615"()
   END_RUNG
   // the same network as SCL:
   IF "AlwaysTRUE" THEN "FC615"(); END_IF;
END_REGION

REGION Network 6: *************DO ***********************
END_REGION

REGION Network 7: "CipDo".MM01CmdMagneticMixerMv1000Command
   RUNG wire#powerrail
      Contact( "AlwaysTRUE" )
      Contact( "ModeDb".Cycle4.Selected )
      Contact( "DB615".CycleRunningMV )
      Contact( "DB607".Mixer )
      Coil( "CipDo".MM01CmdMagneticMixerMvCommand )
   END_RUNG
   // the same network as SCL:
   "CipDo".MM01CmdMagneticMixerMvCommand := "AlwaysTRUE" AND "ModeDb".Cycle4.Selected AND "DB615".CycleRunningMV AND "DB607".Mixer;
END_REGION

REGION Network 8: "DB623".CpCmd
   RUNG wire#powerrail
      Contact( "AlwaysTRUE" )
      Contact( "ModeDb".Cycle4.Selected )
      Contact( "DB615".Running )
      wire#w1
      Contact( "DB608".RecPump )
      wire#w2
      Contact( "CP01".Output )
      Coil( "CipDo".CP01CmdCentrifugalPumpMvAreaCommand )
   END_RUNG
   RUNG wire#w1
      { S7_Templates := "SrcType := Int" } EQ_Contact(in1 := "DB615".CurrentStep, in2 := 2)
      wire#w3
      Contact( "DB609".CycleRunning )
      { S7_Templates := "SrcType := Int" } NE_Contact(in1 := "DB609".StepDelay."Noof StepsPv", in2 := 1)
      { S7_Templates := "SrcType := Int" } NE_Contact(in1 := "DB609".StepDelay."Noof StepsPv", in2 := 2)
   END_RUNG wire#w2
   RUNG wire#w1
      { S7_Templates := "SrcType := Int" } EQ_Contact(in1 := "DB615".CurrentStep, in2 := 3)
   END_RUNG wire#w3
   RUNG wire#w1
      { S7_Templates := "SrcType := Int" } EQ_Contact(in1 := "DB615".CurrentStep, in2 := 1)
      { S7_Templates := "SrcType := Int" } GE_Contact(in1 := "DB604".StepDelay."Noof StepsPv", in2 := 9)
   END_RUNG wire#w2
   // the same network as SCL:
   "CipDo".CP01CmdCentrifugalPumpMvAreaCommand := "AlwaysTRUE" AND "ModeDb".Cycle4.Selected AND "DB615".Running AND ("DB608".RecPump OR ((("DB615".CurrentStep = 2) OR ("DB615".CurrentStep = 3)) AND "DB609".CycleRunning AND ("DB609".StepDelay."Noof StepsPv" <> 1) AND ("DB609".StepDelay."Noof StepsPv" <> 2)) OR (("DB615".CurrentStep = 1) AND ("DB604".StepDelay."Noof StepsPv" >= 9))) AND "CP01".Output;
END_REGION

REGION Network 9: "CipDo".CP01CmdCentrifugalPump
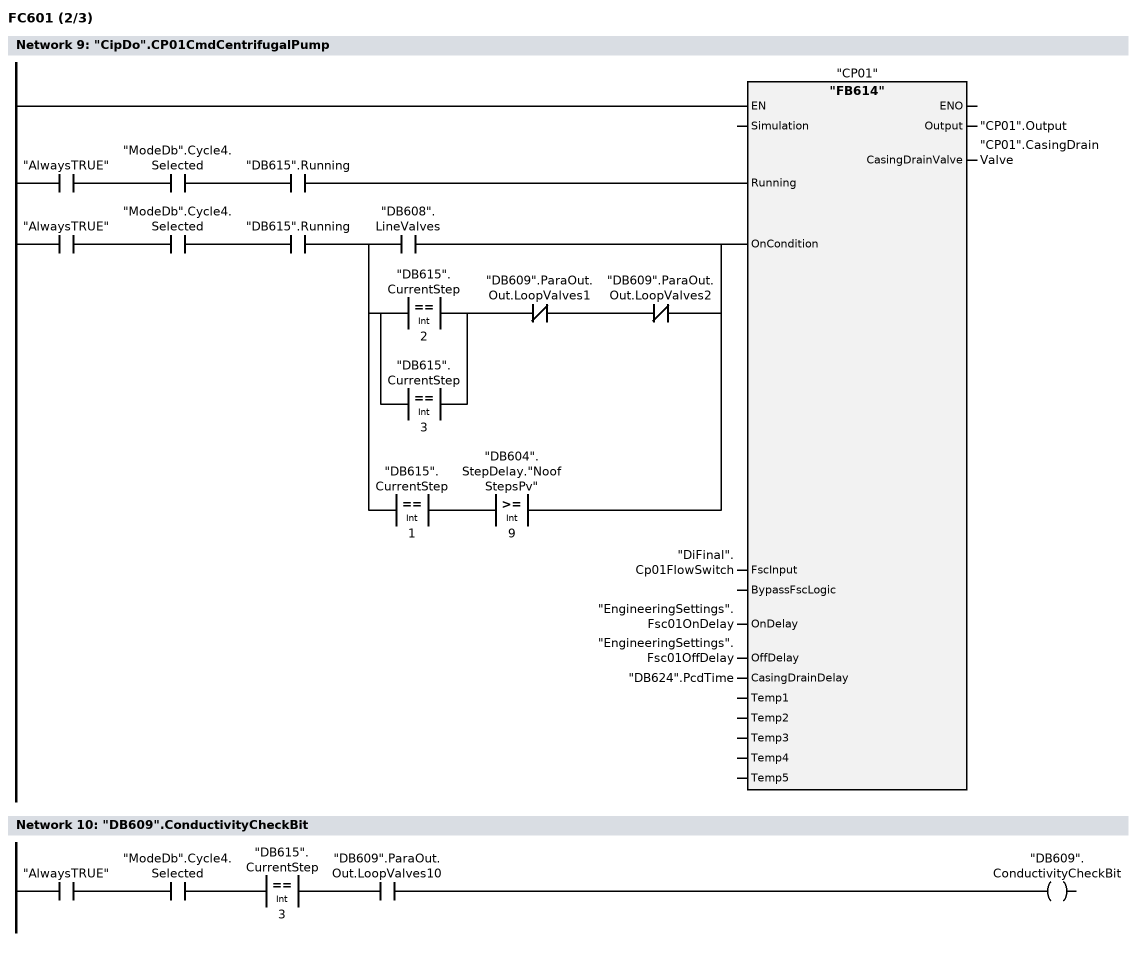
   RUNG wire#powerrail
      "CP01"(Running := wire#w1, OnCondition := wire#w4, Simulation :=, FscInput := "DiFinal".Cp01FlowSwitch, BypassFscLogic :=, OnDelay := "EngineeringSettings".Fsc01OnDelay, OffDelay := "EngineeringSettings".Fsc01OffDelay, CasingDrainDelay := "DB624".PcdTime, Temp1 :=, Temp2 :=, Temp3 :=, Temp4 :=, Temp5 :=, Output => "CP01".Output, CasingDrainValve => "CP01".CasingDrainValve)
   END_RUNG
   RUNG wire#powerrail
      Contact( "AlwaysTRUE" )
      Contact( "ModeDb".Cycle4.Selected )
      Contact( "DB615".Running )
   END_RUNG wire#w1
   RUNG wire#powerrail
      Contact( "AlwaysTRUE" )
      Contact( "ModeDb".Cycle4.Selected )
      Contact( "DB615".Running )
      wire#w2
      Contact( "DB608".LineValves )
   END_RUNG wire#w4
   RUNG wire#w2
      { S7_Templates := "SrcType := Int" } EQ_Contact(in1 := "DB615".CurrentStep, in2 := 2)
      wire#w3
      I_Contact( "DB609".ParaOut.Out.LoopValves1 )
      I_Contact( "DB609".ParaOut.Out.LoopValves2 )
   END_RUNG wire#w4
   RUNG wire#w2
      { S7_Templates := "SrcType := Int" } EQ_Contact(in1 := "DB615".CurrentStep, in2 := 3)
   END_RUNG wire#w3
   RUNG wire#w2
      { S7_Templates := "SrcType := Int" } EQ_Contact(in1 := "DB615".CurrentStep, in2 := 1)
      { S7_Templates := "SrcType := Int" } GE_Contact(in1 := "DB604".StepDelay."Noof StepsPv", in2 := 9)
   END_RUNG wire#w4
   // the same network as SCL:
   "CP01"(Running := "AlwaysTRUE" AND "ModeDb".Cycle4.Selected AND "DB615".Running,   // "FB614"
          OnCondition := "AlwaysTRUE" AND "ModeDb".Cycle4.Selected AND "DB615".Running AND ("DB608".LineValves OR ((("DB615".CurrentStep = 2) OR ("DB615".CurrentStep = 3)) AND NOT "DB609".ParaOut.Out.LoopValves1 AND NOT "DB609".ParaOut.Out.LoopValves2) OR (("DB615".CurrentStep = 1) AND ("DB604".StepDelay."Noof StepsPv" >= 9))),
          FscInput := "DiFinal".Cp01FlowSwitch,
          OnDelay := "EngineeringSettings".Fsc01OnDelay,
          OffDelay := "EngineeringSettings".Fsc01OffDelay,
          CasingDrainDelay := "DB624".PcdTime,
          Output => "CP01".Output,
          CasingDrainValve => "CP01".CasingDrainValve);
END_REGION

REGION Network 10: "DB609".ConductivityCheckBit
   RUNG wire#powerrail
      Contact( "AlwaysTRUE" )
      Contact( "ModeDb".Cycle4.Selected )
      { S7_Templates := "SrcType := Int" } EQ_Contact(in1 := "DB615".CurrentStep, in2 := 3)
      Contact( "DB609".ParaOut.Out.LoopValves10 )
      Coil( "DB609".ConductivityCheckBit )
   END_RUNG
   // the same network as SCL:
   "DB609".ConductivityCheckBit := "AlwaysTRUE" AND "ModeDb".Cycle4.Selected AND ("DB615".CurrentStep = 3) AND "DB609".ParaOut.Out.LoopValves10;
END_REGION

REGION Network 12: "ProcessAlarms".MvVesselWfiFlowLow
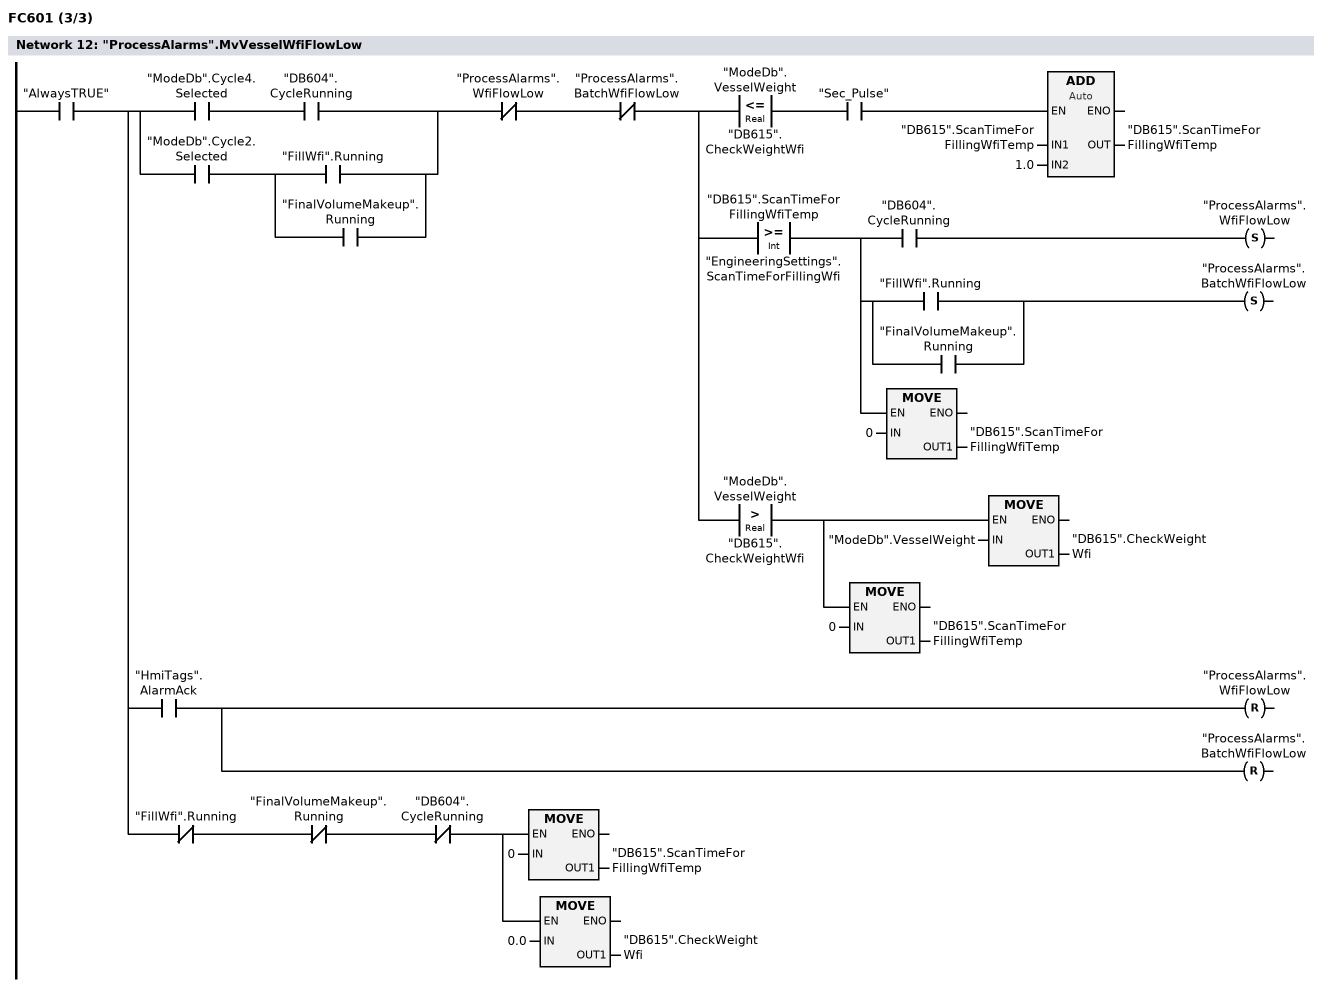
   RUNG wire#powerrail
      Contact( "AlwaysTRUE" )
      wire#w1
      Contact( "ModeDb".Cycle4.Selected )
      Contact( "DB604".CycleRunning )
      wire#w2
      I_Contact( "ProcessAlarms".WfiFlowLow )
      I_Contact( "ProcessAlarms".BatchWfiFlowLow )
      wire#w4
      { S7_Templates := "SrcType := Real" } LE_Contact(in1 := "ModeDb".VesselWeight, in2 := "DB615".CheckWeightWfi)
      Contact( "Sec_Pulse" )
      Add(in1 := "DB615".ScanTimeForFillingWfiTemp, in2 := 1.0, out => "DB615".ScanTimeForFillingWfiTemp)
   END_RUNG
   RUNG wire#w1
      Contact( "ModeDb".Cycle2.Selected )
      wire#w3
      Contact( "FillWfi".Running )
   END_RUNG wire#w2
   RUNG wire#w3
      Contact( "FinalVolumeMakeup".Running )
   END_RUNG wire#w2
   RUNG wire#w4
      { S7_Templates := "SrcType := Int" } GE_Contact(in1 := "DB615".ScanTimeForFillingWfiTemp, in2 := "EngineeringSettings".ScanTimeForFillingWfi)
      wire#w5
      Contact( "DB604".CycleRunning )
      S_Coil( "ProcessAlarms".WfiFlowLow )
   END_RUNG
   RUNG wire#w5
      Contact( "FillWfi".Running )
      wire#w6
      S_Coil( "ProcessAlarms".BatchWfiFlowLow )
   END_RUNG
   RUNG wire#w5
      Contact( "FinalVolumeMakeup".Running )
   END_RUNG wire#w6
   RUNG wire#w5
      Move(in := 0, out1 => "DB615".ScanTimeForFillingWfiTemp)
   END_RUNG
   RUNG wire#w4
      { S7_Templates := "SrcType := Real" } GT_Contact(in1 := "ModeDb".VesselWeight, in2 := "DB615".CheckWeightWfi)
      wire#w7
      Move(in := "ModeDb".VesselWeight, out1 => "DB615".CheckWeightWfi)
   END_RUNG
   RUNG wire#w7
      Move(in := 0, out1 => "DB615".ScanTimeForFillingWfiTemp)
   END_RUNG
   RUNG wire#w1
      Contact( "HmiTags".AlarmAck )
      wire#w8
      R_Coil( "ProcessAlarms".WfiFlowLow )
   END_RUNG
   RUNG wire#w8
      R_Coil( "ProcessAlarms".BatchWfiFlowLow )
   END_RUNG
   RUNG wire#w1
      I_Contact( "FillWfi".Running )
      I_Contact( "FinalVolumeMakeup".Running )
      I_Contact( "DB604".CycleRunning )
      wire#w9
      Move(in := 0, out1 => "DB615".ScanTimeForFillingWfiTemp)
   END_RUNG
   RUNG wire#w9
      Move(in := 0.0, out1 => "DB615".CheckWeightWfi)
   END_RUNG
   // the same network as SCL:
   #_w1 := "AlwaysTRUE" AND (("ModeDb".Cycle4.Selected AND "DB604".CycleRunning) OR ("ModeDb".Cycle2.Selected AND ("FillWfi".Running OR "FinalVolumeMakeup".Running))) AND NOT "ProcessAlarms".WfiFlowLow AND NOT "ProcessAlarms".BatchWfiFlowLow;
   IF #_w1 AND ("ModeDb".VesselWeight <= "DB615".CheckWeightWfi) AND "Sec_Pulse" THEN
       "DB615".ScanTimeForFillingWfiTemp := "DB615".ScanTimeForFillingWfiTemp + 1.0;
   END_IF;
   #_w2 := #_w1 AND ("DB615".ScanTimeForFillingWfiTemp >= "EngineeringSettings".ScanTimeForFillingWfi);
   IF #_w2 AND "DB604".CycleRunning THEN "ProcessAlarms".WfiFlowLow := TRUE; END_IF;
   IF #_w2 AND ("FillWfi".Running OR "FinalVolumeMakeup".Running) THEN
       "ProcessAlarms".BatchWfiFlowLow := TRUE;
   END_IF;
   IF #_w2 THEN "DB615".ScanTimeForFillingWfiTemp := 0; END_IF;
   #_w3 := #_w1 AND ("ModeDb".VesselWeight > "DB615".CheckWeightWfi);
   IF #_w3 THEN
       "DB615".CheckWeightWfi := "ModeDb".VesselWeight;
       "DB615".ScanTimeForFillingWfiTemp := 0;
   END_IF;
   IF "AlwaysTRUE" AND "HmiTags".AlarmAck THEN
       "ProcessAlarms".WfiFlowLow := FALSE;
       "ProcessAlarms".BatchWfiFlowLow := FALSE;
   END_IF;
   IF "AlwaysTRUE" AND NOT "FillWfi".Running AND NOT "FinalVolumeMakeup".Running AND NOT "DB604".CycleRunning THEN
       "DB615".ScanTimeForFillingWfiTemp := 0;
       "DB615".CheckWeightWfi := 0.0;
   END_IF;
END_REGION
END_FUNCTION

FUNCTION "FC604" : Void   // FC604, LAD
TITLE = FC604
{ S7_Optimized_Access := 'TRUE' }
// CIP BLOCK CALL
// stored: AutoNumber false, SetENOAutomatically false
BEGIN

REGION Network 1: #CycleSelection
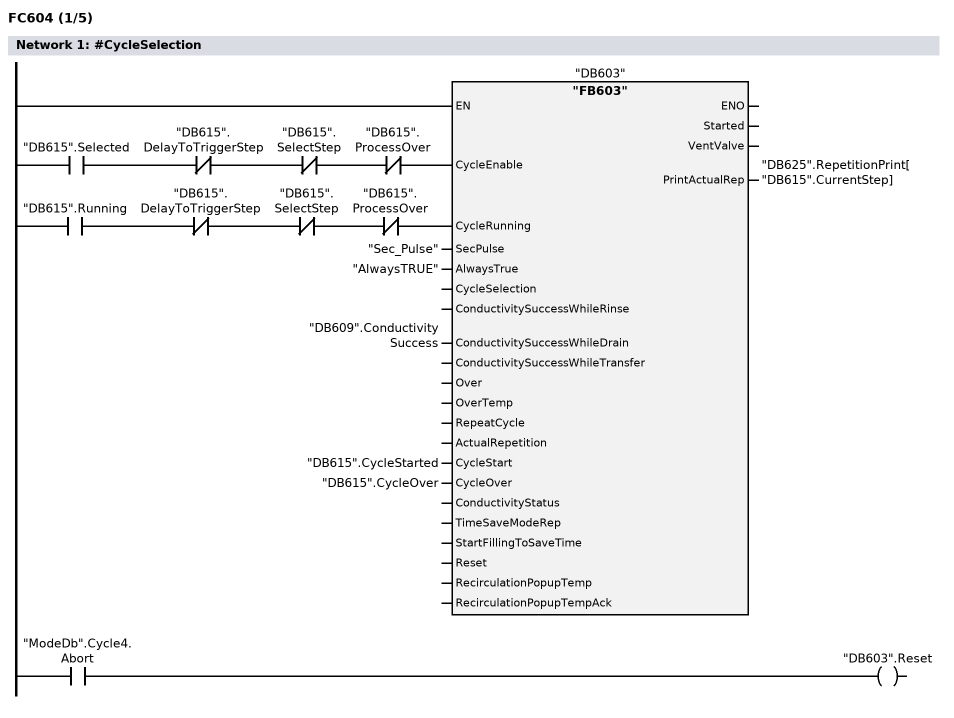
   RUNG wire#powerrail
      "DB603"(CycleEnable := wire#w1, CycleRunning := wire#w2, SecPulse := "Sec_Pulse", AlwaysTrue := "AlwaysTRUE", CycleSelection :=, ConductivitySuccessWhileRinse :=, ConductivitySuccessWhileDrain := "DB609".ConductivitySuccess, ConductivitySuccessWhileTransfer :=, Over :=, OverTemp :=, RepeatCycle :=, ActualRepetition :=, CycleStart := "DB615".CycleStarted, CycleOver := "DB615".CycleOver, ConductivityStatus :=, TimeSaveModeRep :=, StartFillingToSaveTime :=, Reset :=, RecirculationPopupTemp :=, RecirculationPopupTempAck :=, Started =>, VentValve =>, PrintActualRep => "DB625".RepetitionPrint["DB615".CurrentStep])
   END_RUNG
   RUNG wire#powerrail
      Contact( "DB615".Selected )
      I_Contact( "DB615".DelayToTriggerStep )
      I_Contact( "DB615".SelectStep )
      I_Contact( "DB615".ProcessOver )
   END_RUNG wire#w1
   RUNG wire#powerrail
      Contact( "DB615".Running )
      I_Contact( "DB615".DelayToTriggerStep )
      I_Contact( "DB615".SelectStep )
      I_Contact( "DB615".ProcessOver )
   END_RUNG wire#w2
   RUNG wire#powerrail
      Contact( "ModeDb".Cycle4.Abort )
      Coil( "DB603".Reset )
   END_RUNG
   // the same network as SCL:
   "DB603"(CycleEnable := "DB615".Selected AND NOT "DB615".DelayToTriggerStep AND NOT "DB615".SelectStep AND NOT "DB615".ProcessOver,   // "FB603"
           CycleRunning := "DB615".Running AND NOT "DB615".DelayToTriggerStep AND NOT "DB615".SelectStep AND NOT "DB615".ProcessOver,
           SecPulse := "Sec_Pulse",
           AlwaysTrue := "AlwaysTRUE",
           ConductivitySuccessWhileDrain := "DB609".ConductivitySuccess,
           CycleStart := "DB615".CycleStarted,
           CycleOver := "DB615".CycleOver,
           PrintActualRep => "DB625".RepetitionPrint["DB615".CurrentStep]);
   "DB603".Reset := "ModeDb".Cycle4.Abort;
END_REGION

REGION Network 2: #Filling
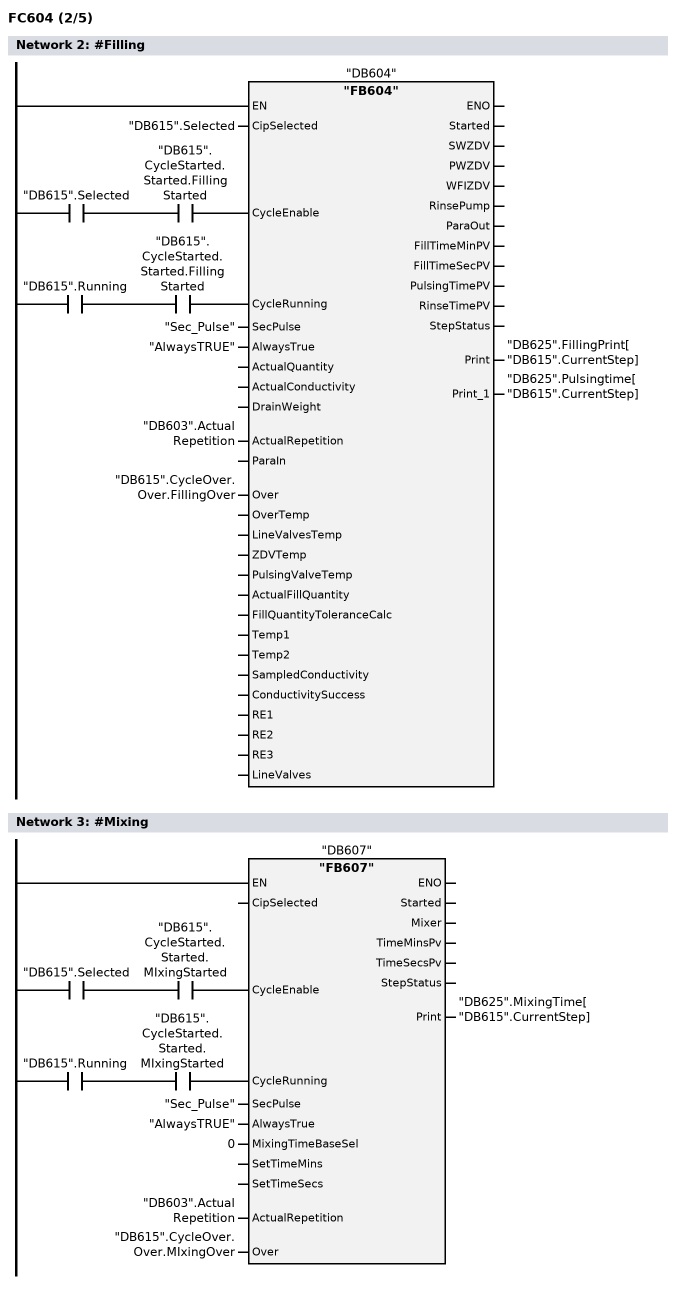
   RUNG wire#powerrail
      "DB604"(CycleEnable := wire#w1, CycleRunning := wire#w2, CipSelected := "DB615".Selected, SecPulse := "Sec_Pulse", AlwaysTrue := "AlwaysTRUE", ActualQuantity :=, ActualConductivity :=, DrainWeight :=, ActualRepetition := "DB603".ActualRepetition, ParaIn :=, Over := "DB615".CycleOver.Over.FillingOver, OverTemp :=, LineValvesTemp :=, ZDVTemp :=, PulsingValveTemp :=, ActualFillQuantity :=, FillQuantityToleranceCalc :=, Temp1 :=, Temp2 :=, SampledConductivity :=, ConductivitySuccess :=, RE1 :=, RE2 :=, RE3 :=, LineValves :=, Started =>, SWZDV =>, PWZDV =>, WFIZDV =>, RinsePump =>, ParaOut =>, FillTimeMinPV =>, FillTimeSecPV =>, PulsingTimePV =>, RinseTimePV =>, StepStatus =>, Print => "DB625".FillingPrint["DB615".CurrentStep], Print_1 => "DB625".Pulsingtime["DB615".CurrentStep])
   END_RUNG
   RUNG wire#powerrail
      Contact( "DB615".Selected )
      Contact( "DB615".CycleStarted.Started.FillingStarted )
   END_RUNG wire#w1
   RUNG wire#powerrail
      Contact( "DB615".Running )
      Contact( "DB615".CycleStarted.Started.FillingStarted )
   END_RUNG wire#w2
   // the same network as SCL:
   "DB604"(CipSelected := "DB615".Selected,   // "FB604"
           CycleEnable := "DB615".Selected AND "DB615".CycleStarted.Started.FillingStarted,
           CycleRunning := "DB615".Running AND "DB615".CycleStarted.Started.FillingStarted,
           SecPulse := "Sec_Pulse",
           AlwaysTrue := "AlwaysTRUE",
           ActualRepetition := "DB603".ActualRepetition,
           Over := "DB615".CycleOver.Over.FillingOver,
           Print => "DB625".FillingPrint["DB615".CurrentStep],
           Print_1 => "DB625".Pulsingtime["DB615".CurrentStep]);
END_REGION

REGION Network 3: #Mixing
   RUNG wire#powerrail
      "DB607"(CycleEnable := wire#w1, CycleRunning := wire#w2, CipSelected :=, SecPulse := "Sec_Pulse", AlwaysTrue := "AlwaysTRUE", MixingTimeBaseSel := 0, SetTimeMins :=, SetTimeSecs :=, ActualRepetition := "DB603".ActualRepetition, Over := "DB615".CycleOver.Over.MIxingOver, Started =>, Mixer =>, TimeMinsPv =>, TimeSecsPv =>, StepStatus =>, Print => "DB625".MixingTime["DB615".CurrentStep])
   END_RUNG
   RUNG wire#powerrail
      Contact( "DB615".Selected )
      Contact( "DB615".CycleStarted.Started.MIxingStarted )
   END_RUNG wire#w1
   RUNG wire#powerrail
      Contact( "DB615".Running )
      Contact( "DB615".CycleStarted.Started.MIxingStarted )
   END_RUNG wire#w2
   // the same network as SCL:
   "DB607"(CycleEnable := "DB615".Selected AND "DB615".CycleStarted.Started.MIxingStarted,   // "FB607"
           CycleRunning := "DB615".Running AND "DB615".CycleStarted.Started.MIxingStarted,
           SecPulse := "Sec_Pulse",
           AlwaysTrue := "AlwaysTRUE",
           MixingTimeBaseSel := 0,
           ActualRepetition := "DB603".ActualRepetition,
           Over := "DB615".CycleOver.Over.MIxingOver,
           Print => "DB625".MixingTime["DB615".CurrentStep]);
END_REGION

REGION Network 4: #Recirculation
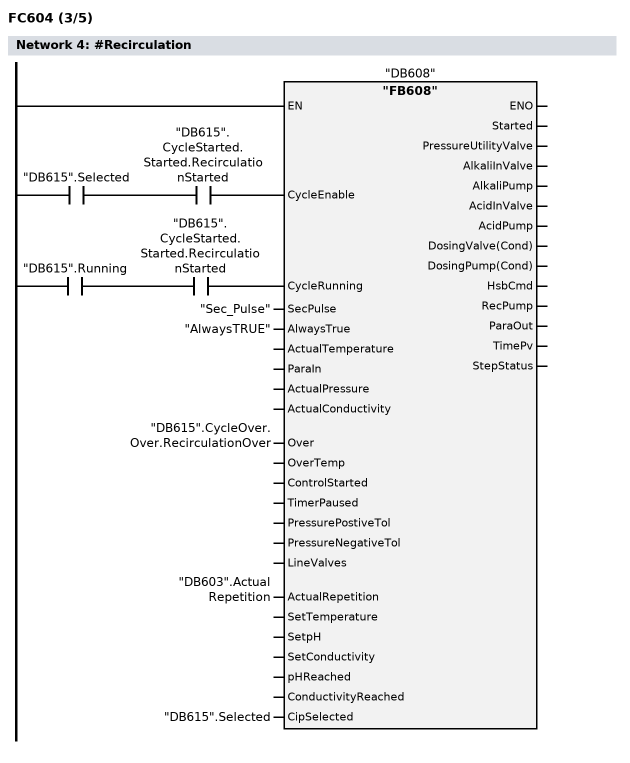
   RUNG wire#powerrail
      "DB608"(CycleEnable := wire#w1, CycleRunning := wire#w2, SecPulse := "Sec_Pulse", AlwaysTrue := "AlwaysTRUE", ActualTemperature :=, ParaIn :=, ActualPressure :=, ActualConductivity :=, Over := "DB615".CycleOver.Over.RecirculationOver, OverTemp :=, ControlStarted :=, TimerPaused :=, PressurePostiveTol :=, PressureNegativeTol :=, LineValves :=, ActualRepetition := "DB603".ActualRepetition, SetTemperature :=, SetpH :=, SetConductivity :=, pHReached :=, ConductivityReached :=, CipSelected := "DB615".Selected, Started =>, PressureUtilityValve =>, AlkaliInValve =>, AlkaliPump =>, AcidInValve =>, AcidPump =>, "DosingValve(Cond)" =>, "DosingPump(Cond)" =>, HsbCmd =>, RecPump =>, ParaOut =>, TimePv =>, StepStatus =>)
   END_RUNG
   RUNG wire#powerrail
      Contact( "DB615".Selected )
      Contact( "DB615".CycleStarted.Started.RecirculationStarted )
   END_RUNG wire#w1
   RUNG wire#powerrail
      Contact( "DB615".Running )
      Contact( "DB615".CycleStarted.Started.RecirculationStarted )
   END_RUNG wire#w2
   // the same network as SCL:
   "DB608"(CycleEnable := "DB615".Selected AND "DB615".CycleStarted.Started.RecirculationStarted,   // "FB608"
           CycleRunning := "DB615".Running AND "DB615".CycleStarted.Started.RecirculationStarted,
           SecPulse := "Sec_Pulse",
           AlwaysTrue := "AlwaysTRUE",
           Over := "DB615".CycleOver.Over.RecirculationOver,
           ActualRepetition := "DB603".ActualRepetition,
           CipSelected := "DB615".Selected);
END_REGION

REGION Network 5: #Drain
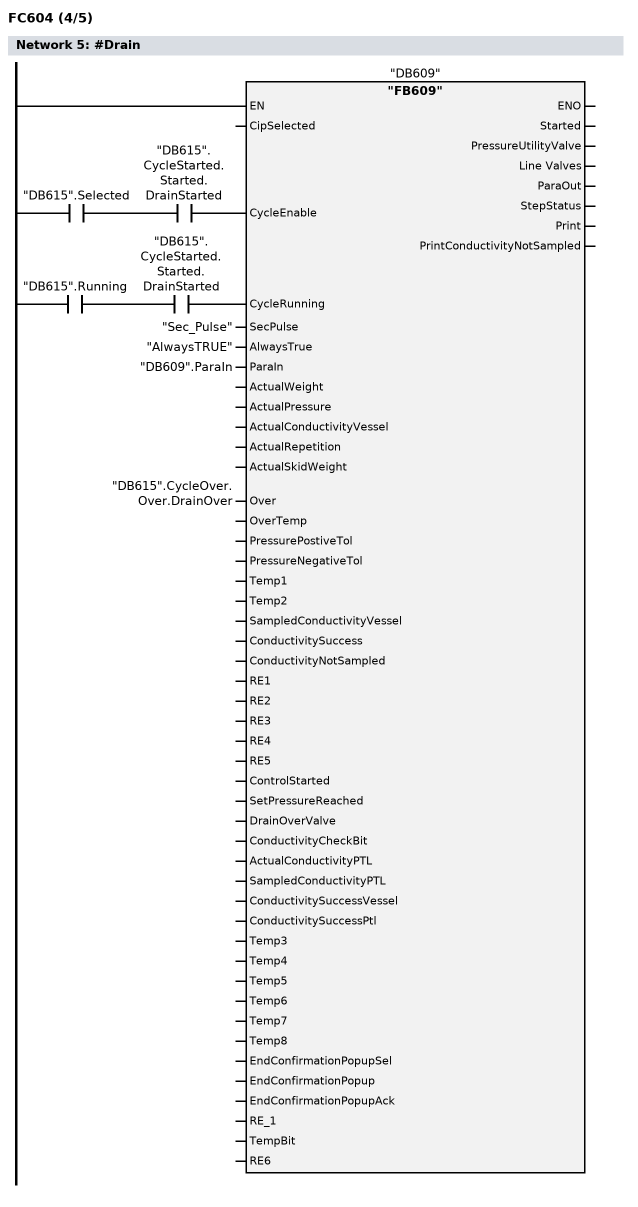
   RUNG wire#powerrail
      "DB609"(CycleEnable := wire#w1, CycleRunning := wire#w2, CipSelected :=, SecPulse := "Sec_Pulse", AlwaysTrue := "AlwaysTRUE", ParaIn := "DB609".ParaIn, ActualWeight :=, ActualPressure :=, ActualConductivityVessel :=, ActualRepetition :=, ActualSkidWeight :=, Over := "DB615".CycleOver.Over.DrainOver, OverTemp :=, PressurePostiveTol :=, PressureNegativeTol :=, Temp1 :=, Temp2 :=, SampledConductivityVessel :=, ConductivitySuccess :=, ConductivityNotSampled :=, RE1 :=, RE2 :=, RE3 :=, RE4 :=, RE5 :=, ControlStarted :=, SetPressureReached :=, DrainOverValve :=, ConductivityCheckBit :=, ActualConductivityPTL :=, SampledConductivityPTL :=, ConductivitySuccessVessel :=, ConductivitySuccessPtl :=, Temp3 :=, Temp4 :=, Temp5 :=, Temp6 :=, Temp7 :=, Temp8 :=, EndConfirmationPopupSel :=, EndConfirmationPopup :=, EndConfirmationPopupAck :=, RE_1 :=, TempBit :=, RE6 :=, Started =>, PressureUtilityValve =>, "Line Valves" =>, ParaOut =>, StepStatus =>, Print =>, PrintConductivityNotSampled =>)
   END_RUNG
   RUNG wire#powerrail
      Contact( "DB615".Selected )
      Contact( "DB615".CycleStarted.Started.DrainStarted )
   END_RUNG wire#w1
   RUNG wire#powerrail
      Contact( "DB615".Running )
      Contact( "DB615".CycleStarted.Started.DrainStarted )
   END_RUNG wire#w2
   // the same network as SCL:
   "DB609"(CycleEnable := "DB615".Selected AND "DB615".CycleStarted.Started.DrainStarted,   // "FB609"
           CycleRunning := "DB615".Running AND "DB615".CycleStarted.Started.DrainStarted,
           SecPulse := "Sec_Pulse",
           AlwaysTrue := "AlwaysTRUE",
           ParaIn := "DB609".ParaIn,
           Over := "DB615".CycleOver.Over.DrainOver);
END_REGION

REGION Network 6: #SystemDrain
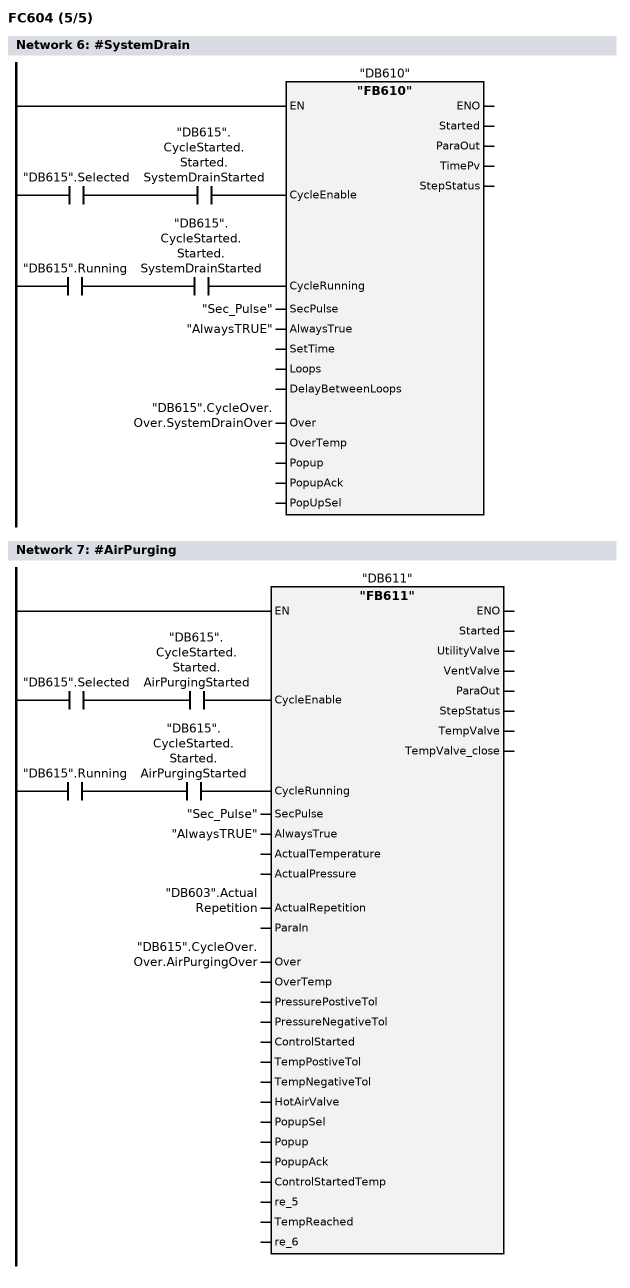
   RUNG wire#powerrail
      "DB610"(CycleEnable := wire#w1, CycleRunning := wire#w2, SecPulse := "Sec_Pulse", AlwaysTrue := "AlwaysTRUE", SetTime :=, Loops :=, DelayBetweenLoops :=, Over := "DB615".CycleOver.Over.SystemDrainOver, OverTemp :=, Popup :=, PopupAck :=, PopUpSel :=, Started =>, ParaOut =>, TimePv =>, StepStatus =>)
   END_RUNG
   RUNG wire#powerrail
      Contact( "DB615".Selected )
      Contact( "DB615".CycleStarted.Started.SystemDrainStarted )
   END_RUNG wire#w1
   RUNG wire#powerrail
      Contact( "DB615".Running )
      Contact( "DB615".CycleStarted.Started.SystemDrainStarted )
   END_RUNG wire#w2
   // the same network as SCL:
   "DB610"(CycleEnable := "DB615".Selected AND "DB615".CycleStarted.Started.SystemDrainStarted,   // "FB610"
           CycleRunning := "DB615".Running AND "DB615".CycleStarted.Started.SystemDrainStarted,
           SecPulse := "Sec_Pulse",
           AlwaysTrue := "AlwaysTRUE",
           Over := "DB615".CycleOver.Over.SystemDrainOver);
END_REGION

REGION Network 7: #AirPurging
   RUNG wire#powerrail
      "DB611"(CycleEnable := wire#w1, CycleRunning := wire#w2, SecPulse := "Sec_Pulse", AlwaysTrue := "AlwaysTRUE", ActualTemperature :=, ActualPressure :=, ActualRepetition := "DB603".ActualRepetition, ParaIn :=, Over := "DB615".CycleOver.Over.AirPurgingOver, OverTemp :=, PressurePostiveTol :=, PressureNegativeTol :=, ControlStarted :=, TempPostiveTol :=, TempNegativeTol :=, HotAirValve :=, PopupSel :=, Popup :=, PopupAck :=, ControlStartedTemp :=, re_5 :=, TempReached :=, re_6 :=, Started =>, UtilityValve =>, VentValve =>, ParaOut =>, StepStatus =>, TempValve =>, TempValve_close =>)
   END_RUNG
   RUNG wire#powerrail
      Contact( "DB615".Selected )
      Contact( "DB615".CycleStarted.Started.AirPurgingStarted )
   END_RUNG wire#w1
   RUNG wire#powerrail
      Contact( "DB615".Running )
      Contact( "DB615".CycleStarted.Started.AirPurgingStarted )
   END_RUNG wire#w2
   // the same network as SCL:
   "DB611"(CycleEnable := "DB615".Selected AND "DB615".CycleStarted.Started.AirPurgingStarted,   // "FB611"
           CycleRunning := "DB615".Running AND "DB615".CycleStarted.Started.AirPurgingStarted,
           SecPulse := "Sec_Pulse",
           AlwaysTrue := "AlwaysTRUE",
           ActualRepetition := "DB603".ActualRepetition,
           Over := "DB615".CycleOver.Over.AirPurgingOver);
END_REGION
END_FUNCTION

FUNCTION_BLOCK "FB603"   // FB603, LAD
TITLE = FB603
{ S7_Optimized_Access := 'FALSE' }
AUTHOR : PRECISE
FAMILY : PRECISE
// CIP
// stored: AutoNumber false, SetENOAutomatically false
   VAR_INPUT
      CycleEnable : Bool;
      CycleRunning : Bool;
      SecPulse : Bool;
      AlwaysTrue : Bool;
      CycleSelection : "CIP";
      ConductivitySuccessWhileRinse : Bool;
      ConductivitySuccessWhileDrain : Bool;
      ConductivitySuccessWhileTransfer : Bool;
   END_VAR
   VAR_OUTPUT
      Started : Bool;
      VentValve : Bool;
      PrintActualRep : Int;
   END_VAR
   VAR_IN_OUT
      Over : Bool;
      OverTemp : Bool;
      RepeatCycle : Bool;
      ActualRepetition : Int;
      CycleStart : "CipCycleStarted";
      CycleOver : "CipCycleOver";
      ConductivityStatus : Bool;
      TimeSaveModeRep : Int;
      StartFillingToSaveTime : Bool;
      Reset : Bool;
      RecirculationPopupTemp : Bool;
      RecirculationPopupTempAck : Bool;
   END_VAR
   VAR
      Re : Array[0..30] of Bool;
   END_VAR
   VAR_TEMP   // added for the SCL form of the ladder/FBD networks
      _w1 : Bool;
      _w2 : Bool;
      _w3 : Bool;
      _w4 : Bool;
      _w5 : Bool;
      _w6 : Bool;
      _w7 : Bool;
      _w8 : Bool;
      _w9 : Bool;
      _w10 : Bool;
      _w11 : Bool;
      _w12 : Bool;
   END_VAR
BEGIN

REGION Network 1
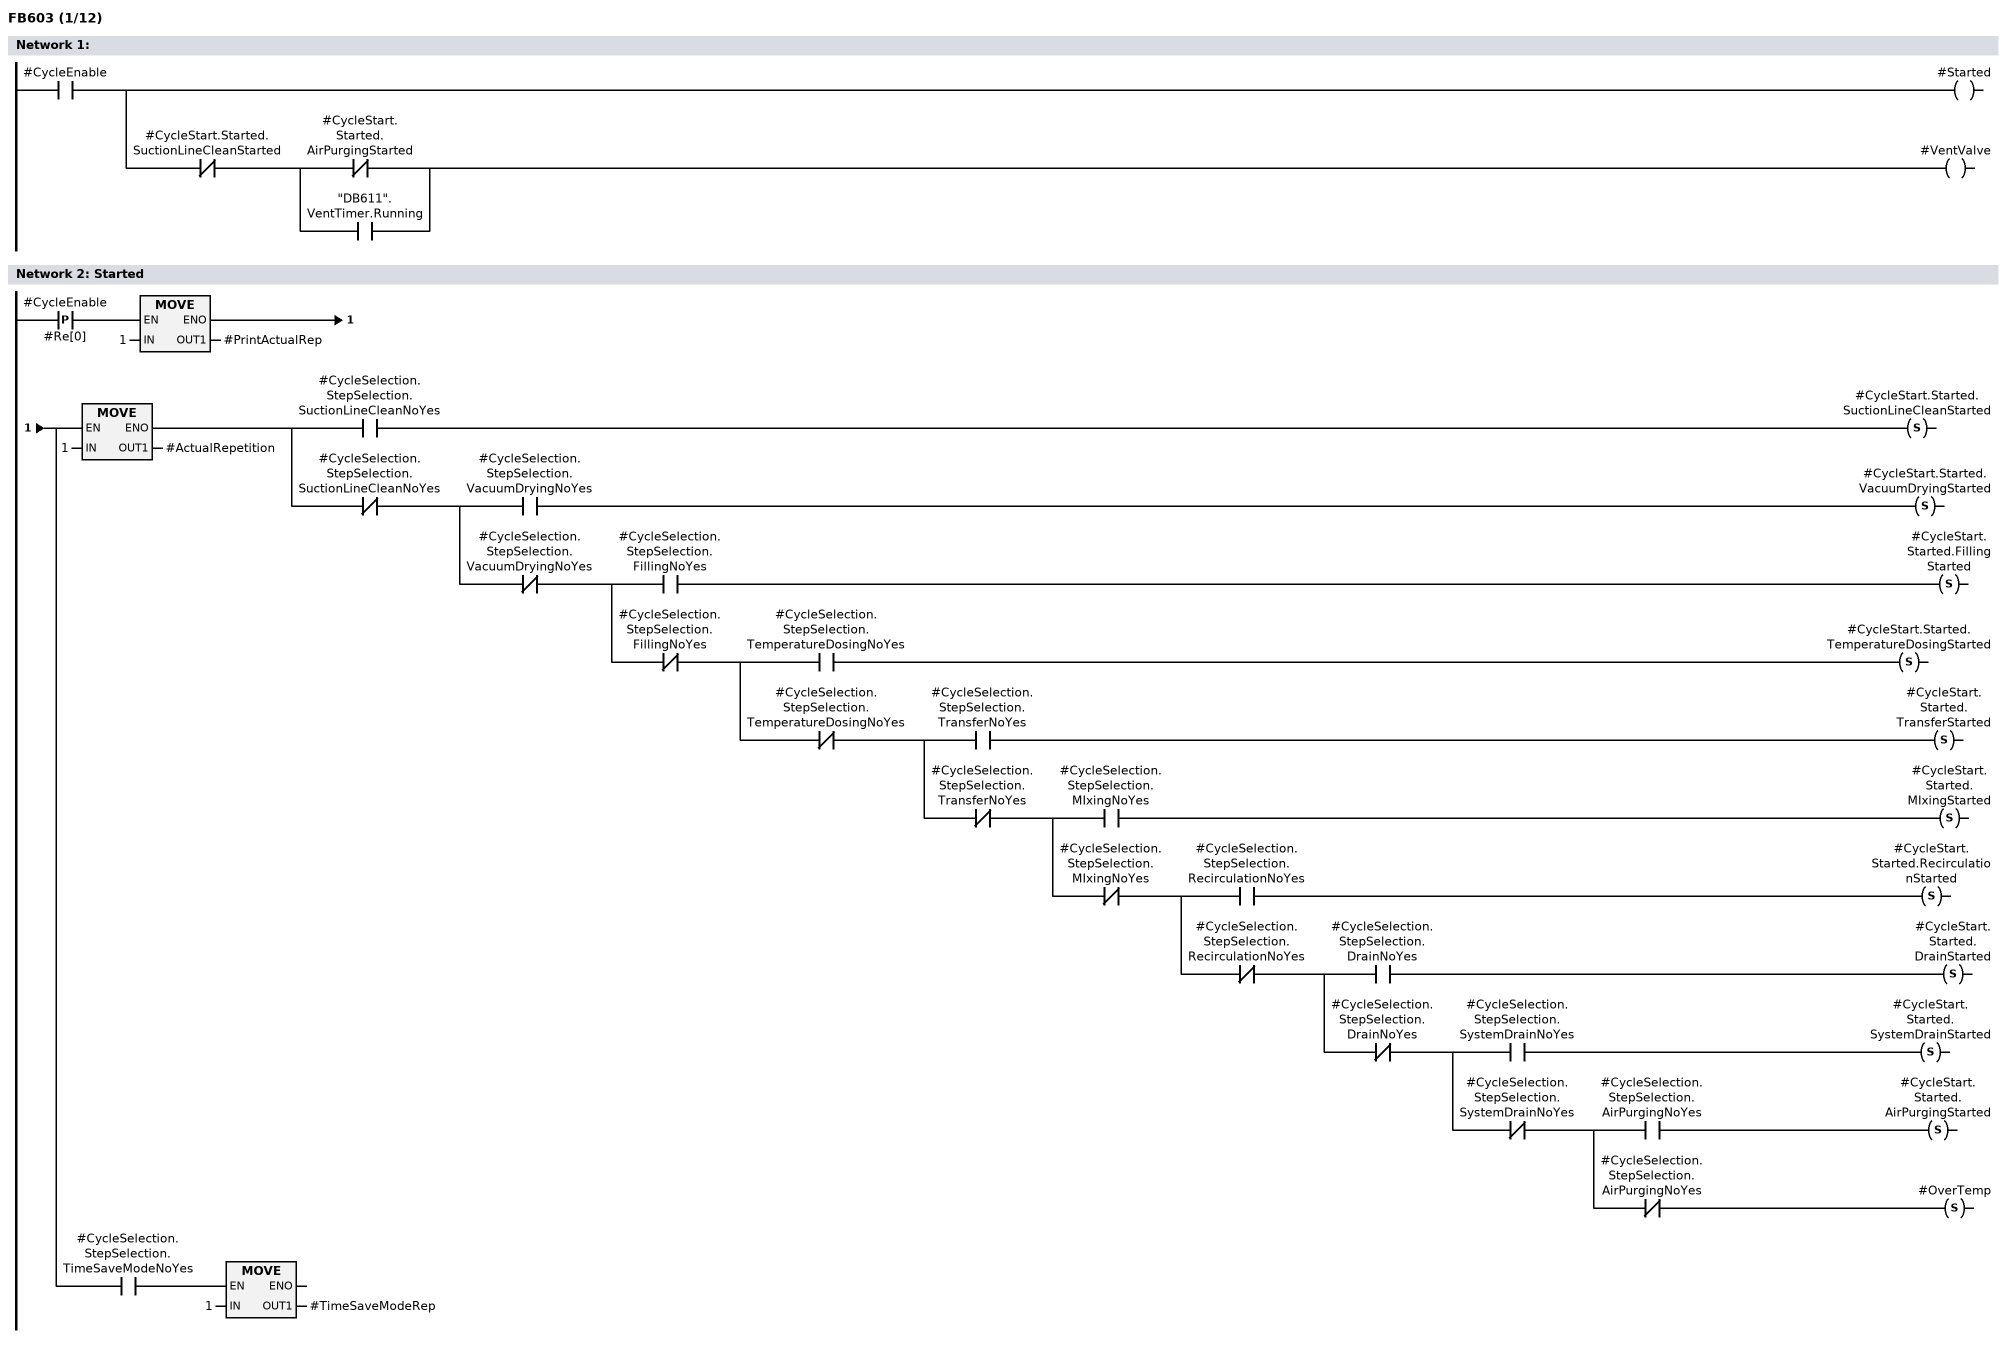
   RUNG wire#powerrail
      Contact( #CycleEnable )
      wire#w1
      Coil( #Started )
   END_RUNG
   RUNG wire#w1
      I_Contact( #CycleStart.Started.SuctionLineCleanStarted )
      wire#w2
      I_Contact( #CycleStart.Started.AirPurgingStarted )
      wire#w3
      Coil( #VentValve )
   END_RUNG
   RUNG wire#w2
      Contact( "DB611".VentTimer.Running )
   END_RUNG wire#w3
   // the same network as SCL:
   #Started := #CycleEnable;
   #VentValve := #CycleEnable AND NOT #CycleStart.Started.SuctionLineCleanStarted AND (NOT #CycleStart.Started.AirPurgingStarted OR "DB611".VentTimer.Running);
END_REGION

REGION Network 2: Started
   RUNG wire#powerrail
      P_Contact(operand := #CycleEnable, bit := #Re[0])
      Move(in := 1, out1 => #PrintActualRep)
      wire#w1
      Move(in := 1, out1 => #ActualRepetition)
      wire#w2
      Contact( #CycleSelection.StepSelection.SuctionLineCleanNoYes )
      S_Coil( #CycleStart.Started.SuctionLineCleanStarted )
   END_RUNG
   RUNG wire#w2
      I_Contact( #CycleSelection.StepSelection.SuctionLineCleanNoYes )
      wire#w3
      Contact( #CycleSelection.StepSelection.VacuumDryingNoYes )
      S_Coil( #CycleStart.Started.VacuumDryingStarted )
   END_RUNG
   RUNG wire#w3
      I_Contact( #CycleSelection.StepSelection.VacuumDryingNoYes )
      wire#w4
      Contact( #CycleSelection.StepSelection.FillingNoYes )
      S_Coil( #CycleStart.Started.FillingStarted )
   END_RUNG
   RUNG wire#w4
      I_Contact( #CycleSelection.StepSelection.FillingNoYes )
      wire#w5
      Contact( #CycleSelection.StepSelection.TemperatureDosingNoYes )
      S_Coil( #CycleStart.Started.TemperatureDosingStarted )
   END_RUNG
   RUNG wire#w5
      I_Contact( #CycleSelection.StepSelection.TemperatureDosingNoYes )
      wire#w6
      Contact( #CycleSelection.StepSelection.TransferNoYes )
      S_Coil( #CycleStart.Started.TransferStarted )
   END_RUNG
   RUNG wire#w6
      I_Contact( #CycleSelection.StepSelection.TransferNoYes )
      wire#w7
      Contact( #CycleSelection.StepSelection.MIxingNoYes )
      S_Coil( #CycleStart.Started.MIxingStarted )
   END_RUNG
   RUNG wire#w7
      I_Contact( #CycleSelection.StepSelection.MIxingNoYes )
      wire#w8
      Contact( #CycleSelection.StepSelection.RecirculationNoYes )
      S_Coil( #CycleStart.Started.RecirculationStarted )
   END_RUNG
   RUNG wire#w8
      I_Contact( #CycleSelection.StepSelection.RecirculationNoYes )
      wire#w9
      Contact( #CycleSelection.StepSelection.DrainNoYes )
      S_Coil( #CycleStart.Started.DrainStarted )
   END_RUNG
   RUNG wire#w9
      I_Contact( #CycleSelection.StepSelection.DrainNoYes )
      wire#w10
      Contact( #CycleSelection.StepSelection.SystemDrainNoYes )
      S_Coil( #CycleStart.Started.SystemDrainStarted )
   END_RUNG
   RUNG wire#w10
      I_Contact( #CycleSelection.StepSelection.SystemDrainNoYes )
      wire#w11
      Contact( #CycleSelection.StepSelection.AirPurgingNoYes )
      S_Coil( #CycleStart.Started.AirPurgingStarted )
   END_RUNG
   RUNG wire#w11
      I_Contact( #CycleSelection.StepSelection.AirPurgingNoYes )
      S_Coil( #OverTemp )
   END_RUNG
   RUNG wire#w1
      Contact( #CycleSelection.StepSelection.TimeSaveModeNoYes )
      Move(in := 1, out1 => #TimeSaveModeRep)
   END_RUNG
   // the same network as SCL:
   #_w1 := #CycleEnable AND NOT #Re[0];   // rising edge of #CycleEnable
   #Re[0] := #CycleEnable;
   IF #_w1 THEN
       #PrintActualRep := 1;
       #ActualRepetition := 1;
   END_IF;
   IF #_w1 AND #CycleSelection.StepSelection.SuctionLineCleanNoYes THEN
       #CycleStart.Started.SuctionLineCleanStarted := TRUE;
   END_IF;
   #_w2 := #_w1 AND NOT #CycleSelection.StepSelection.SuctionLineCleanNoYes;
   IF #_w2 AND #CycleSelection.StepSelection.VacuumDryingNoYes THEN
       #CycleStart.Started.VacuumDryingStarted := TRUE;
   END_IF;
   #_w3 := #_w2 AND NOT #CycleSelection.StepSelection.VacuumDryingNoYes;
   IF #_w3 AND #CycleSelection.StepSelection.FillingNoYes THEN
       #CycleStart.Started.FillingStarted := TRUE;
   END_IF;
   #_w4 := #_w3 AND NOT #CycleSelection.StepSelection.FillingNoYes;
   IF #_w4 AND #CycleSelection.StepSelection.TemperatureDosingNoYes THEN
       #CycleStart.Started.TemperatureDosingStarted := TRUE;
   END_IF;
   #_w5 := #_w4 AND NOT #CycleSelection.StepSelection.TemperatureDosingNoYes;
   IF #_w5 AND #CycleSelection.StepSelection.TransferNoYes THEN
       #CycleStart.Started.TransferStarted := TRUE;
   END_IF;
   #_w6 := #_w5 AND NOT #CycleSelection.StepSelection.TransferNoYes;
   IF #_w6 AND #CycleSelection.StepSelection.MIxingNoYes THEN
       #CycleStart.Started.MIxingStarted := TRUE;
   END_IF;
   #_w7 := #_w6 AND NOT #CycleSelection.StepSelection.MIxingNoYes;
   IF #_w7 AND #CycleSelection.StepSelection.RecirculationNoYes THEN
       #CycleStart.Started.RecirculationStarted := TRUE;
   END_IF;
   #_w8 := #_w7 AND NOT #CycleSelection.StepSelection.RecirculationNoYes;
   IF #_w8 AND #CycleSelection.StepSelection.DrainNoYes THEN
       #CycleStart.Started.DrainStarted := TRUE;
   END_IF;
   #_w9 := #_w8 AND NOT #CycleSelection.StepSelection.DrainNoYes;
   IF #_w9 AND #CycleSelection.StepSelection.SystemDrainNoYes THEN
       #CycleStart.Started.SystemDrainStarted := TRUE;
   END_IF;
   #_w10 := #_w9 AND NOT #CycleSelection.StepSelection.SystemDrainNoYes;
   IF #_w10 AND #CycleSelection.StepSelection.AirPurgingNoYes THEN
       #CycleStart.Started.AirPurgingStarted := TRUE;
   END_IF;
   IF #_w10 AND NOT #CycleSelection.StepSelection.AirPurgingNoYes THEN #OverTemp := TRUE; END_IF;
   IF #_w1 AND #CycleSelection.StepSelection.TimeSaveModeNoYes THEN #TimeSaveModeRep := 1; END_IF;
END_REGION

REGION Network 3: SuctionLineCleanOver
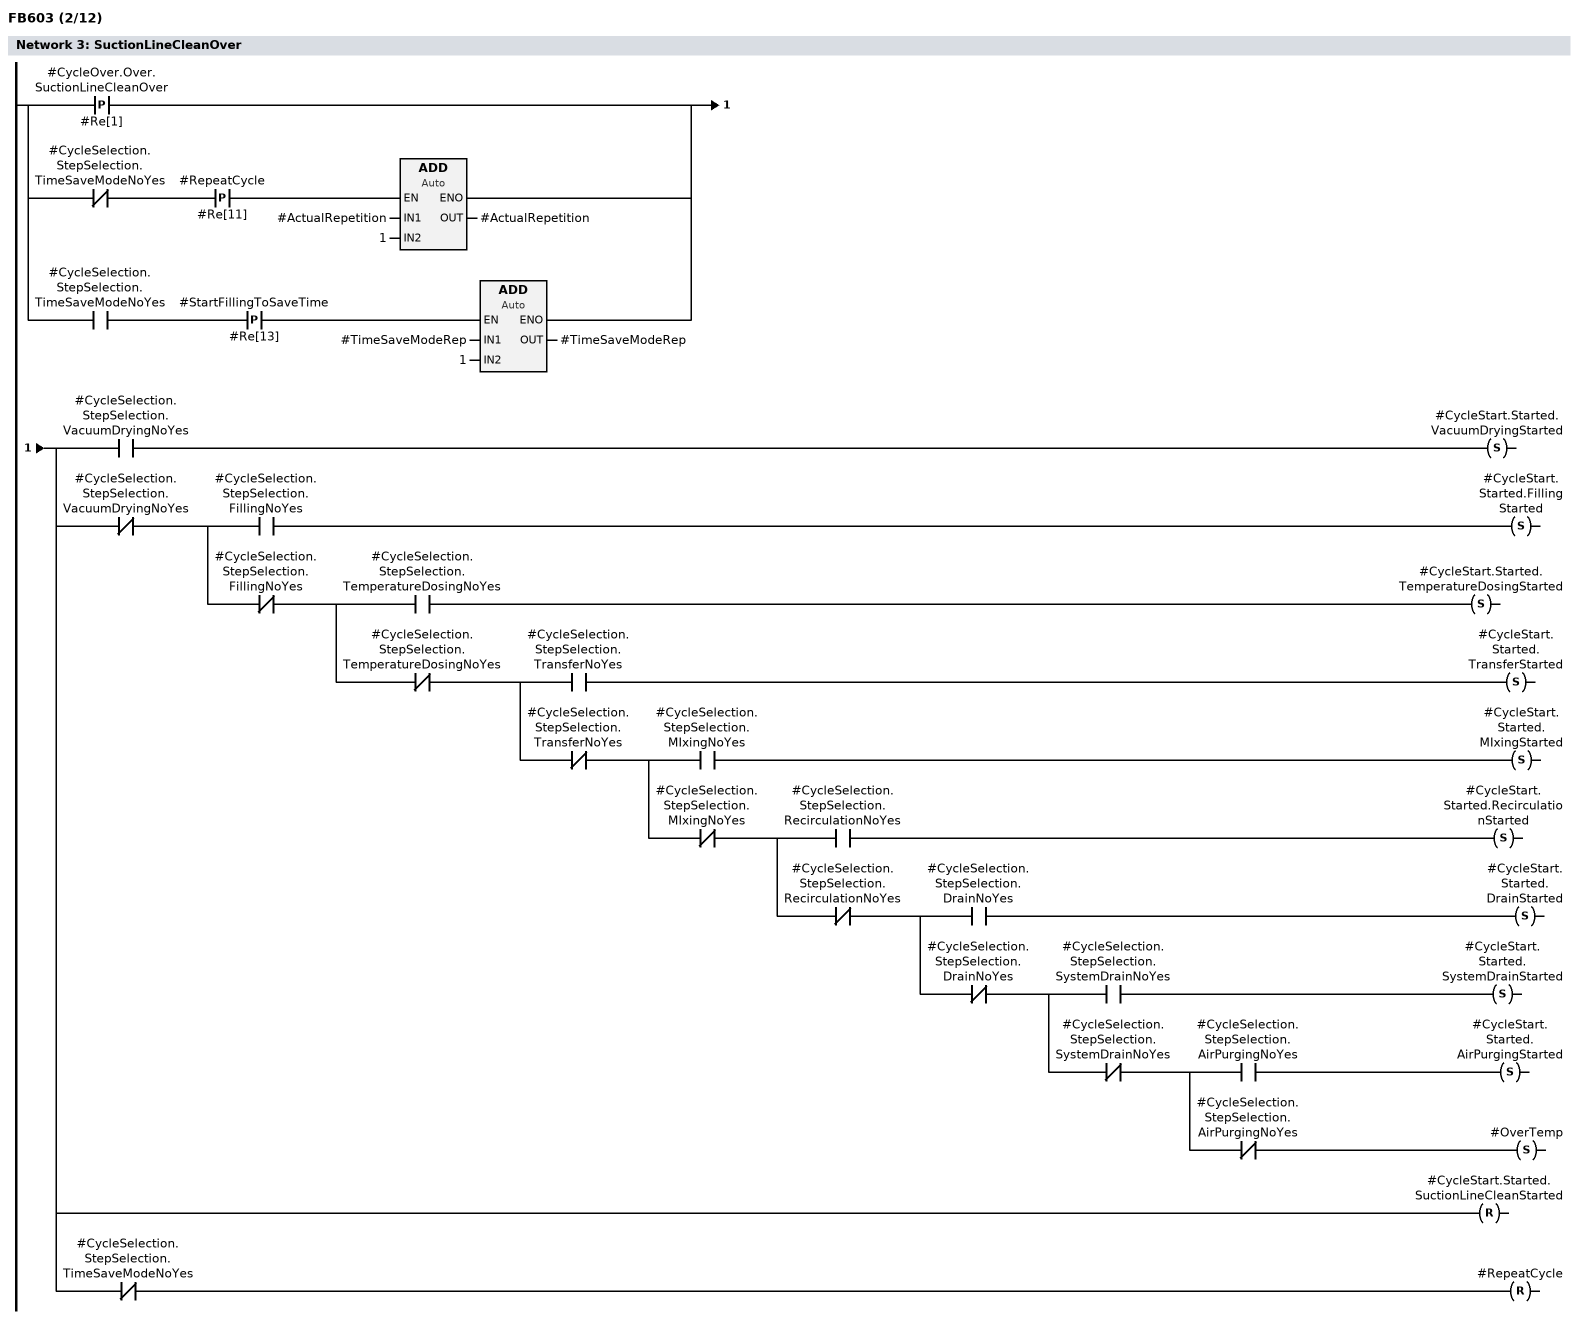
   RUNG wire#powerrail
      P_Contact(operand := #CycleOver.Over.SuctionLineCleanOver, bit := #Re[1])
      wire#w1
      Contact( #CycleSelection.StepSelection.VacuumDryingNoYes )
      S_Coil( #CycleStart.Started.VacuumDryingStarted )
   END_RUNG
   RUNG wire#powerrail
      I_Contact( #CycleSelection.StepSelection.TimeSaveModeNoYes )
      P_Contact(operand := #RepeatCycle, bit := #Re[11])
      Add(in1 := #ActualRepetition, in2 := 1, out => #ActualRepetition)
   END_RUNG wire#w1
   RUNG wire#powerrail
      Contact( #CycleSelection.StepSelection.TimeSaveModeNoYes )
      P_Contact(operand := #StartFillingToSaveTime, bit := #Re[13])
      Add(in1 := #TimeSaveModeRep, in2 := 1, out => #TimeSaveModeRep)
   END_RUNG wire#w1
   RUNG wire#w1
      I_Contact( #CycleSelection.StepSelection.VacuumDryingNoYes )
      wire#w2
      Contact( #CycleSelection.StepSelection.FillingNoYes )
      S_Coil( #CycleStart.Started.FillingStarted )
   END_RUNG
   RUNG wire#w2
      I_Contact( #CycleSelection.StepSelection.FillingNoYes )
      wire#w3
      Contact( #CycleSelection.StepSelection.TemperatureDosingNoYes )
      S_Coil( #CycleStart.Started.TemperatureDosingStarted )
   END_RUNG
   RUNG wire#w3
      I_Contact( #CycleSelection.StepSelection.TemperatureDosingNoYes )
      wire#w4
      Contact( #CycleSelection.StepSelection.TransferNoYes )
      S_Coil( #CycleStart.Started.TransferStarted )
   END_RUNG
   RUNG wire#w4
      I_Contact( #CycleSelection.StepSelection.TransferNoYes )
      wire#w5
      Contact( #CycleSelection.StepSelection.MIxingNoYes )
      S_Coil( #CycleStart.Started.MIxingStarted )
   END_RUNG
   RUNG wire#w5
      I_Contact( #CycleSelection.StepSelection.MIxingNoYes )
      wire#w6
      Contact( #CycleSelection.StepSelection.RecirculationNoYes )
      S_Coil( #CycleStart.Started.RecirculationStarted )
   END_RUNG
   RUNG wire#w6
      I_Contact( #CycleSelection.StepSelection.RecirculationNoYes )
      wire#w7
      Contact( #CycleSelection.StepSelection.DrainNoYes )
      S_Coil( #CycleStart.Started.DrainStarted )
   END_RUNG
   RUNG wire#w7
      I_Contact( #CycleSelection.StepSelection.DrainNoYes )
      wire#w8
      Contact( #CycleSelection.StepSelection.SystemDrainNoYes )
      S_Coil( #CycleStart.Started.SystemDrainStarted )
   END_RUNG
   RUNG wire#w8
      I_Contact( #CycleSelection.StepSelection.SystemDrainNoYes )
      wire#w9
      Contact( #CycleSelection.StepSelection.AirPurgingNoYes )
      S_Coil( #CycleStart.Started.AirPurgingStarted )
   END_RUNG
   RUNG wire#w9
      I_Contact( #CycleSelection.StepSelection.AirPurgingNoYes )
      S_Coil( #OverTemp )
   END_RUNG
   RUNG wire#w1
      R_Coil( #CycleStart.Started.SuctionLineCleanStarted )
   END_RUNG
   RUNG wire#w1
      I_Contact( #CycleSelection.StepSelection.TimeSaveModeNoYes )
      R_Coil( #RepeatCycle )
   END_RUNG
   // the same network as SCL:
   #_w1 := #CycleOver.Over.SuctionLineCleanOver AND NOT #Re[1];   // rising edge of #CycleOver.Over.SuctionLineCleanOver
   #Re[1] := #CycleOver.Over.SuctionLineCleanOver;
   #_w2 := NOT #CycleSelection.StepSelection.TimeSaveModeNoYes AND #RepeatCycle AND NOT #Re[11];   // rising edge of #RepeatCycle
   #Re[11] := #RepeatCycle;
   IF #_w2 THEN #ActualRepetition := #ActualRepetition + 1; END_IF;
   #_w3 := #CycleSelection.StepSelection.TimeSaveModeNoYes AND #StartFillingToSaveTime AND NOT #Re[13];   // rising edge of #StartFillingToSaveTime
   #Re[13] := #StartFillingToSaveTime;
   IF #_w3 THEN #TimeSaveModeRep := #TimeSaveModeRep + 1; END_IF;
   #_w4 := #_w1 OR #_w2 OR #_w3;
   IF #_w4 AND #CycleSelection.StepSelection.VacuumDryingNoYes THEN
       #CycleStart.Started.VacuumDryingStarted := TRUE;
   END_IF;
   #_w5 := #_w4 AND NOT #CycleSelection.StepSelection.VacuumDryingNoYes;
   IF #_w5 AND #CycleSelection.StepSelection.FillingNoYes THEN
       #CycleStart.Started.FillingStarted := TRUE;
   END_IF;
   #_w6 := #_w5 AND NOT #CycleSelection.StepSelection.FillingNoYes;
   IF #_w6 AND #CycleSelection.StepSelection.TemperatureDosingNoYes THEN
       #CycleStart.Started.TemperatureDosingStarted := TRUE;
   END_IF;
   #_w7 := #_w6 AND NOT #CycleSelection.StepSelection.TemperatureDosingNoYes;
   IF #_w7 AND #CycleSelection.StepSelection.TransferNoYes THEN
       #CycleStart.Started.TransferStarted := TRUE;
   END_IF;
   #_w8 := #_w7 AND NOT #CycleSelection.StepSelection.TransferNoYes;
   IF #_w8 AND #CycleSelection.StepSelection.MIxingNoYes THEN
       #CycleStart.Started.MIxingStarted := TRUE;
   END_IF;
   #_w9 := #_w8 AND NOT #CycleSelection.StepSelection.MIxingNoYes;
   IF #_w9 AND #CycleSelection.StepSelection.RecirculationNoYes THEN
       #CycleStart.Started.RecirculationStarted := TRUE;
   END_IF;
   #_w10 := #_w9 AND NOT #CycleSelection.StepSelection.RecirculationNoYes;
   IF #_w10 AND #CycleSelection.StepSelection.DrainNoYes THEN
       #CycleStart.Started.DrainStarted := TRUE;
   END_IF;
   #_w11 := #_w10 AND NOT #CycleSelection.StepSelection.DrainNoYes;
   IF #_w11 AND #CycleSelection.StepSelection.SystemDrainNoYes THEN
       #CycleStart.Started.SystemDrainStarted := TRUE;
   END_IF;
   #_w12 := #_w11 AND NOT #CycleSelection.StepSelection.SystemDrainNoYes;
   IF #_w12 AND #CycleSelection.StepSelection.AirPurgingNoYes THEN
       #CycleStart.Started.AirPurgingStarted := TRUE;
   END_IF;
   IF #_w12 AND NOT #CycleSelection.StepSelection.AirPurgingNoYes THEN #OverTemp := TRUE; END_IF;
   IF #_w4 THEN #CycleStart.Started.SuctionLineCleanStarted := FALSE; END_IF;
   IF #_w4 AND NOT #CycleSelection.StepSelection.TimeSaveModeNoYes THEN #RepeatCycle := FALSE; END_IF;
END_REGION

REGION Network 4: VacuumDryingOver
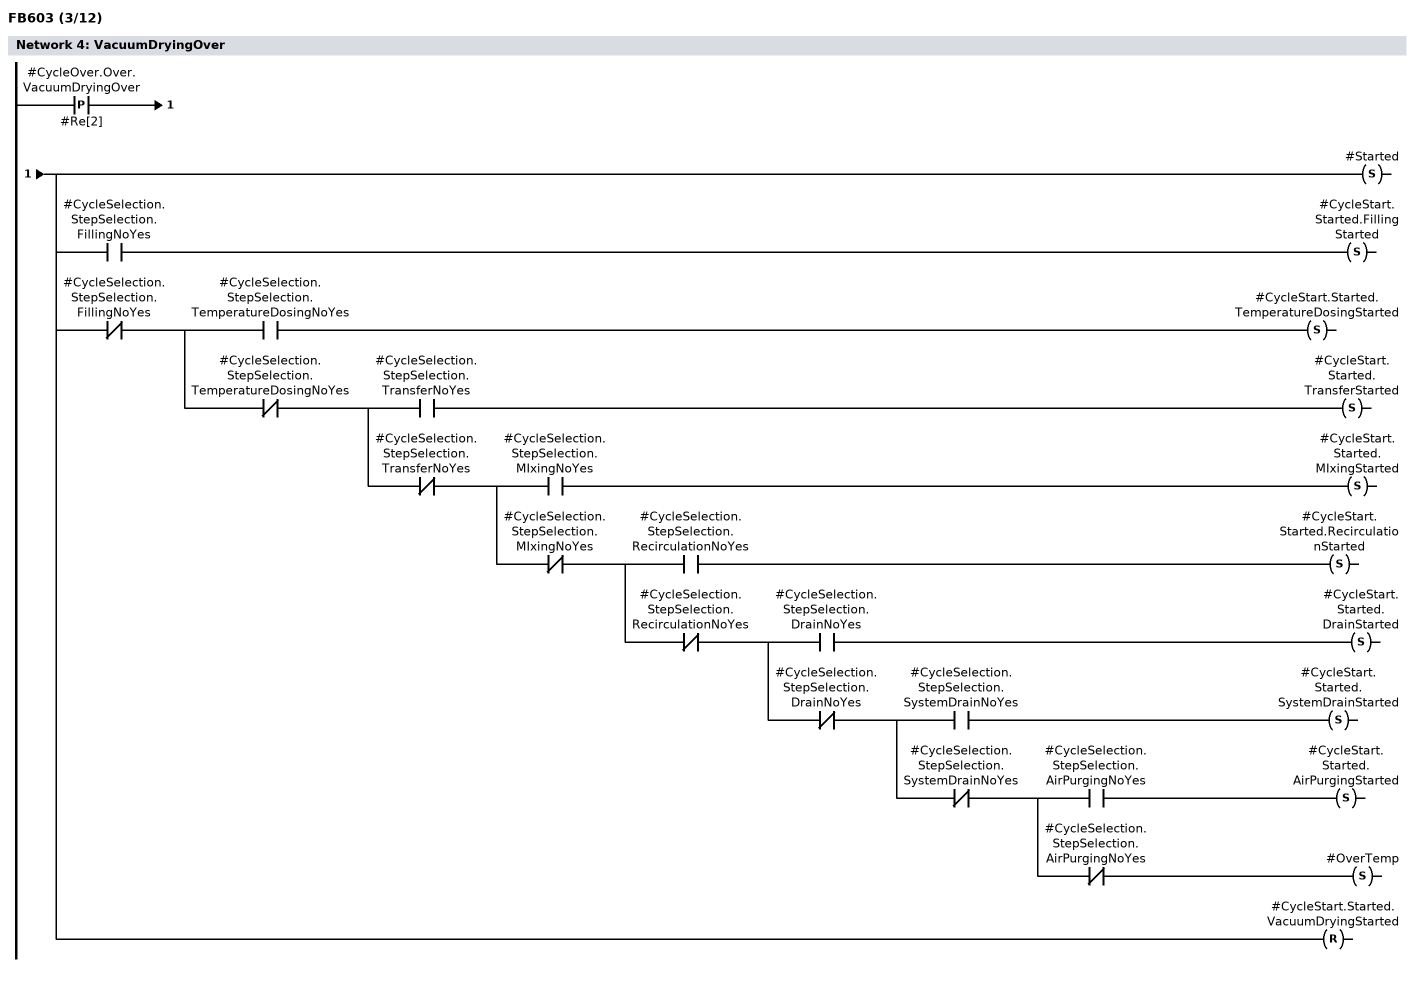
   RUNG wire#powerrail
      P_Contact(operand := #CycleOver.Over.VacuumDryingOver, bit := #Re[2])
      wire#w1
      S_Coil( #Started )
   END_RUNG
   RUNG wire#w1
      Contact( #CycleSelection.StepSelection.FillingNoYes )
      S_Coil( #CycleStart.Started.FillingStarted )
   END_RUNG
   RUNG wire#w1
      I_Contact( #CycleSelection.StepSelection.FillingNoYes )
      wire#w2
      Contact( #CycleSelection.StepSelection.TemperatureDosingNoYes )
      S_Coil( #CycleStart.Started.TemperatureDosingStarted )
   END_RUNG
   RUNG wire#w2
      I_Contact( #CycleSelection.StepSelection.TemperatureDosingNoYes )
      wire#w3
      Contact( #CycleSelection.StepSelection.TransferNoYes )
      S_Coil( #CycleStart.Started.TransferStarted )
   END_RUNG
   RUNG wire#w3
      I_Contact( #CycleSelection.StepSelection.TransferNoYes )
      wire#w4
      Contact( #CycleSelection.StepSelection.MIxingNoYes )
      S_Coil( #CycleStart.Started.MIxingStarted )
   END_RUNG
   RUNG wire#w4
      I_Contact( #CycleSelection.StepSelection.MIxingNoYes )
      wire#w5
      Contact( #CycleSelection.StepSelection.RecirculationNoYes )
      S_Coil( #CycleStart.Started.RecirculationStarted )
   END_RUNG
   RUNG wire#w5
      I_Contact( #CycleSelection.StepSelection.RecirculationNoYes )
      wire#w6
      Contact( #CycleSelection.StepSelection.DrainNoYes )
      S_Coil( #CycleStart.Started.DrainStarted )
   END_RUNG
   RUNG wire#w6
      I_Contact( #CycleSelection.StepSelection.DrainNoYes )
      wire#w7
      Contact( #CycleSelection.StepSelection.SystemDrainNoYes )
      S_Coil( #CycleStart.Started.SystemDrainStarted )
   END_RUNG
   RUNG wire#w7
      I_Contact( #CycleSelection.StepSelection.SystemDrainNoYes )
      wire#w8
      Contact( #CycleSelection.StepSelection.AirPurgingNoYes )
      S_Coil( #CycleStart.Started.AirPurgingStarted )
   END_RUNG
   RUNG wire#w8
      I_Contact( #CycleSelection.StepSelection.AirPurgingNoYes )
      S_Coil( #OverTemp )
   END_RUNG
   RUNG wire#w1
      R_Coil( #CycleStart.Started.VacuumDryingStarted )
   END_RUNG
   // the same network as SCL:
   #_w1 := #CycleOver.Over.VacuumDryingOver AND NOT #Re[2];   // rising edge of #CycleOver.Over.VacuumDryingOver
   #Re[2] := #CycleOver.Over.VacuumDryingOver;
   IF #_w1 THEN #Started := TRUE; END_IF;
   IF #_w1 AND #CycleSelection.StepSelection.FillingNoYes THEN
       #CycleStart.Started.FillingStarted := TRUE;
   END_IF;
   #_w2 := #_w1 AND NOT #CycleSelection.StepSelection.FillingNoYes;
   IF #_w2 AND #CycleSelection.StepSelection.TemperatureDosingNoYes THEN
       #CycleStart.Started.TemperatureDosingStarted := TRUE;
   END_IF;
   #_w3 := #_w2 AND NOT #CycleSelection.StepSelection.TemperatureDosingNoYes;
   IF #_w3 AND #CycleSelection.StepSelection.TransferNoYes THEN
       #CycleStart.Started.TransferStarted := TRUE;
   END_IF;
   #_w4 := #_w3 AND NOT #CycleSelection.StepSelection.TransferNoYes;
   IF #_w4 AND #CycleSelection.StepSelection.MIxingNoYes THEN
       #CycleStart.Started.MIxingStarted := TRUE;
   END_IF;
   #_w5 := #_w4 AND NOT #CycleSelection.StepSelection.MIxingNoYes;
   IF #_w5 AND #CycleSelection.StepSelection.RecirculationNoYes THEN
       #CycleStart.Started.RecirculationStarted := TRUE;
   END_IF;
   #_w6 := #_w5 AND NOT #CycleSelection.StepSelection.RecirculationNoYes;
   IF #_w6 AND #CycleSelection.StepSelection.DrainNoYes THEN
       #CycleStart.Started.DrainStarted := TRUE;
   END_IF;
   #_w7 := #_w6 AND NOT #CycleSelection.StepSelection.DrainNoYes;
   IF #_w7 AND #CycleSelection.StepSelection.SystemDrainNoYes THEN
       #CycleStart.Started.SystemDrainStarted := TRUE;
   END_IF;
   #_w8 := #_w7 AND NOT #CycleSelection.StepSelection.SystemDrainNoYes;
   IF #_w8 AND #CycleSelection.StepSelection.AirPurgingNoYes THEN
       #CycleStart.Started.AirPurgingStarted := TRUE;
   END_IF;
   IF #_w8 AND NOT #CycleSelection.StepSelection.AirPurgingNoYes THEN #OverTemp := TRUE; END_IF;
   IF #_w1 THEN #CycleStart.Started.VacuumDryingStarted := FALSE; END_IF;
END_REGION

REGION Network 5: FillOver
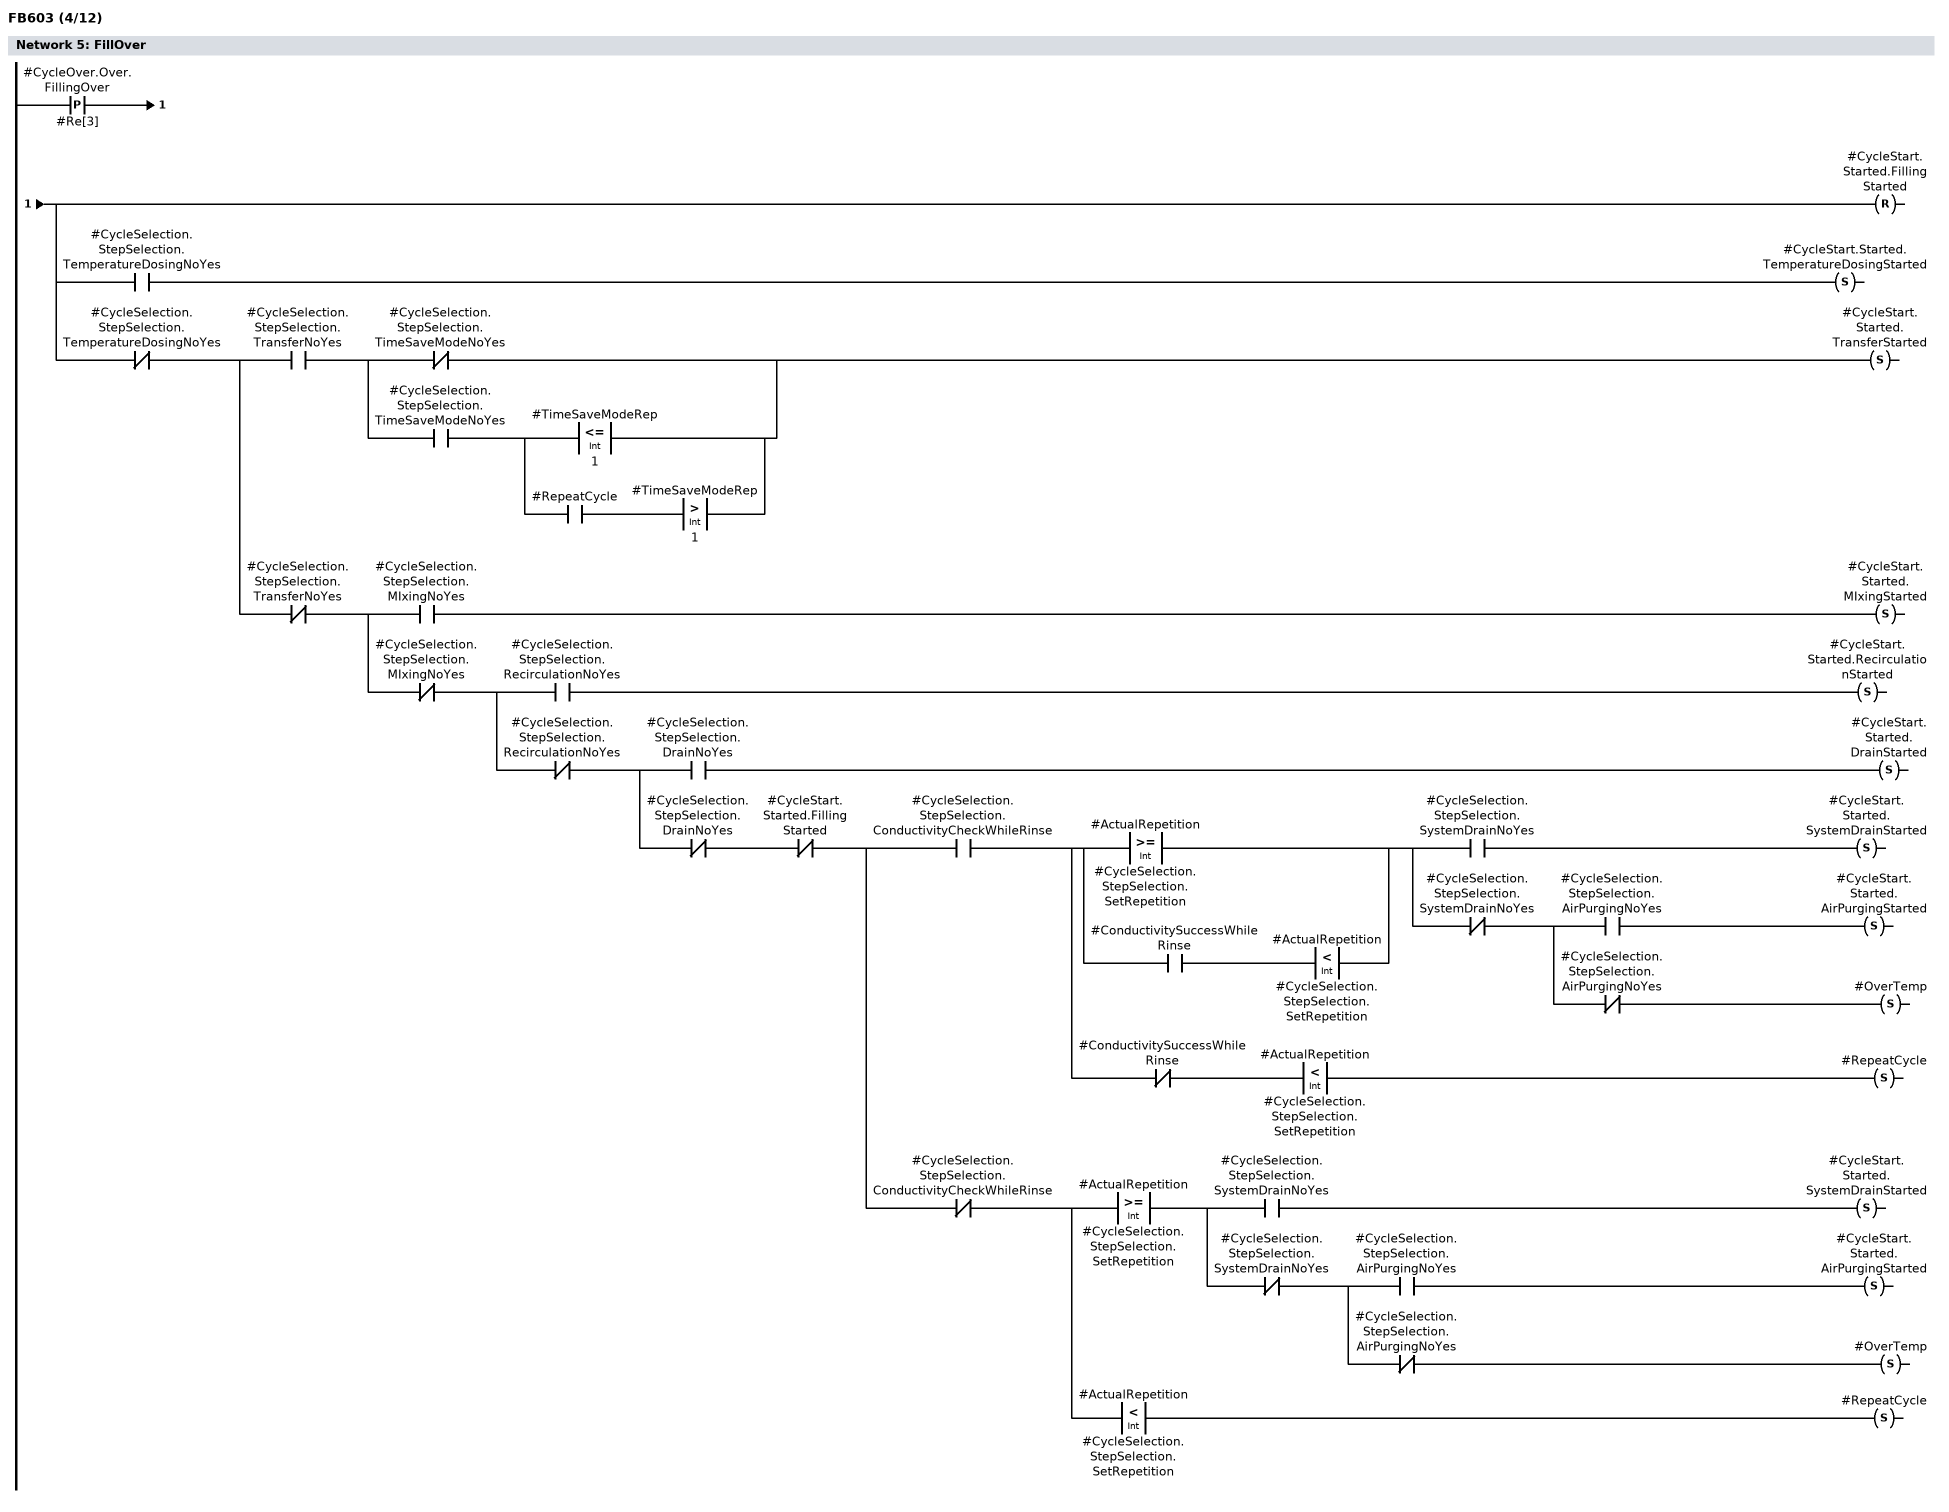
   RUNG wire#powerrail
      P_Contact(operand := #CycleOver.Over.FillingOver, bit := #Re[3])
      wire#w1
      R_Coil( #CycleStart.Started.FillingStarted )
   END_RUNG
   RUNG wire#w1
      Contact( #CycleSelection.StepSelection.TemperatureDosingNoYes )
      S_Coil( #CycleStart.Started.TemperatureDosingStarted )
   END_RUNG
   RUNG wire#w1
      I_Contact( #CycleSelection.StepSelection.TemperatureDosingNoYes )
      wire#w2
      Contact( #CycleSelection.StepSelection.TransferNoYes )
      wire#w3
      I_Contact( #CycleSelection.StepSelection.TimeSaveModeNoYes )
      wire#w4
      S_Coil( #CycleStart.Started.TransferStarted )
   END_RUNG
   RUNG wire#w3
      Contact( #CycleSelection.StepSelection.TimeSaveModeNoYes )
      wire#w5
      { S7_Templates := "SrcType := Int" } LE_Contact(in1 := #TimeSaveModeRep, in2 := 1)
   END_RUNG wire#w4
   RUNG wire#w5
      Contact( #RepeatCycle )
      { S7_Templates := "SrcType := Int" } GT_Contact(in1 := #TimeSaveModeRep, in2 := 1)
   END_RUNG wire#w4
   RUNG wire#w2
      I_Contact( #CycleSelection.StepSelection.TransferNoYes )
      wire#w6
      Contact( #CycleSelection.StepSelection.MIxingNoYes )
      S_Coil( #CycleStart.Started.MIxingStarted )
   END_RUNG
   RUNG wire#w6
      I_Contact( #CycleSelection.StepSelection.MIxingNoYes )
      wire#w7
      Contact( #CycleSelection.StepSelection.RecirculationNoYes )
      S_Coil( #CycleStart.Started.RecirculationStarted )
   END_RUNG
   RUNG wire#w7
      I_Contact( #CycleSelection.StepSelection.RecirculationNoYes )
      wire#w8
      Contact( #CycleSelection.StepSelection.DrainNoYes )
      S_Coil( #CycleStart.Started.DrainStarted )
   END_RUNG
   RUNG wire#w8
      I_Contact( #CycleSelection.StepSelection.DrainNoYes )
      I_Contact( #CycleStart.Started.FillingStarted )
      wire#w9
      Contact( #CycleSelection.StepSelection.ConductivityCheckWhileRinse )
      wire#w10
      { S7_Templates := "SrcType := Int" } GE_Contact(in1 := #ActualRepetition, in2 := #CycleSelection.StepSelection.SetRepetition)
      wire#w11
      Contact( #CycleSelection.StepSelection.SystemDrainNoYes )
      S_Coil( #CycleStart.Started.SystemDrainStarted )
   END_RUNG
   RUNG wire#w10
      Contact( #ConductivitySuccessWhileRinse )
      { S7_Templates := "SrcType := Int" } LT_Contact(in1 := #ActualRepetition, in2 := #CycleSelection.StepSelection.SetRepetition)
   END_RUNG wire#w11
   RUNG wire#w11
      I_Contact( #CycleSelection.StepSelection.SystemDrainNoYes )
      wire#w12
      Contact( #CycleSelection.StepSelection.AirPurgingNoYes )
      S_Coil( #CycleStart.Started.AirPurgingStarted )
   END_RUNG
   RUNG wire#w12
      I_Contact( #CycleSelection.StepSelection.AirPurgingNoYes )
      S_Coil( #OverTemp )
   END_RUNG
   RUNG wire#w10
      I_Contact( #ConductivitySuccessWhileRinse )
      { S7_Templates := "SrcType := Int" } LT_Contact(in1 := #ActualRepetition, in2 := #CycleSelection.StepSelection.SetRepetition)
      S_Coil( #RepeatCycle )
   END_RUNG
   RUNG wire#w9
      I_Contact( #CycleSelection.StepSelection.ConductivityCheckWhileRinse )
      wire#w13
      { S7_Templates := "SrcType := Int" } GE_Contact(in1 := #ActualRepetition, in2 := #CycleSelection.StepSelection.SetRepetition)
      wire#w14
      Contact( #CycleSelection.StepSelection.SystemDrainNoYes )
      S_Coil( #CycleStart.Started.SystemDrainStarted )
   END_RUNG
   RUNG wire#w14
      I_Contact( #CycleSelection.StepSelection.SystemDrainNoYes )
      wire#w15
      Contact( #CycleSelection.StepSelection.AirPurgingNoYes )
      S_Coil( #CycleStart.Started.AirPurgingStarted )
   END_RUNG
   RUNG wire#w15
      I_Contact( #CycleSelection.StepSelection.AirPurgingNoYes )
      S_Coil( #OverTemp )
   END_RUNG
   RUNG wire#w13
      { S7_Templates := "SrcType := Int" } LT_Contact(in1 := #ActualRepetition, in2 := #CycleSelection.StepSelection.SetRepetition)
      S_Coil( #RepeatCycle )
   END_RUNG
   // the same network as SCL:
   #_w1 := #CycleOver.Over.FillingOver AND NOT #Re[3];   // rising edge of #CycleOver.Over.FillingOver
   #Re[3] := #CycleOver.Over.FillingOver;
   IF #_w1 THEN #CycleStart.Started.FillingStarted := FALSE; END_IF;
   IF #_w1 AND #CycleSelection.StepSelection.TemperatureDosingNoYes THEN
       #CycleStart.Started.TemperatureDosingStarted := TRUE;
   END_IF;
   #_w2 := #_w1 AND NOT #CycleSelection.StepSelection.TemperatureDosingNoYes;
   IF #_w2 AND #CycleSelection.StepSelection.TransferNoYes AND (NOT #CycleSelection.StepSelection.TimeSaveModeNoYes OR (#CycleSelection.StepSelection.TimeSaveModeNoYes AND ((#TimeSaveModeRep <= 1) OR (#RepeatCycle AND (#TimeSaveModeRep > 1))))) THEN
       #CycleStart.Started.TransferStarted := TRUE;
   END_IF;
   #_w3 := #_w2 AND NOT #CycleSelection.StepSelection.TransferNoYes;
   IF #_w3 AND #CycleSelection.StepSelection.MIxingNoYes THEN
       #CycleStart.Started.MIxingStarted := TRUE;
   END_IF;
   #_w4 := #_w3 AND NOT #CycleSelection.StepSelection.MIxingNoYes;
   IF #_w4 AND #CycleSelection.StepSelection.RecirculationNoYes THEN
       #CycleStart.Started.RecirculationStarted := TRUE;
   END_IF;
   #_w5 := #_w4 AND NOT #CycleSelection.StepSelection.RecirculationNoYes;
   IF #_w5 AND #CycleSelection.StepSelection.DrainNoYes THEN
       #CycleStart.Started.DrainStarted := TRUE;
   END_IF;
   #_w6 := #_w5 AND NOT #CycleSelection.StepSelection.DrainNoYes AND NOT #CycleStart.Started.FillingStarted;
   #_w7 := #_w6 AND #CycleSelection.StepSelection.ConductivityCheckWhileRinse;
   #_w8 := #_w7 AND ((#ActualRepetition >= #CycleSelection.StepSelection.SetRepetition) OR (#ConductivitySuccessWhileRinse AND (#ActualRepetition < #CycleSelection.StepSelection.SetRepetition)));
   IF #_w8 AND #CycleSelection.StepSelection.SystemDrainNoYes THEN
       #CycleStart.Started.SystemDrainStarted := TRUE;
   END_IF;
   #_w9 := #_w8 AND NOT #CycleSelection.StepSelection.SystemDrainNoYes;
   IF #_w9 AND #CycleSelection.StepSelection.AirPurgingNoYes THEN
       #CycleStart.Started.AirPurgingStarted := TRUE;
   END_IF;
   IF #_w9 AND NOT #CycleSelection.StepSelection.AirPurgingNoYes THEN #OverTemp := TRUE; END_IF;
   IF #_w7 AND NOT #ConductivitySuccessWhileRinse AND (#ActualRepetition < #CycleSelection.StepSelection.SetRepetition) THEN
       #RepeatCycle := TRUE;
   END_IF;
   #_w10 := #_w6 AND NOT #CycleSelection.StepSelection.ConductivityCheckWhileRinse;
   #_w11 := #_w10 AND (#ActualRepetition >= #CycleSelection.StepSelection.SetRepetition);
   IF #_w11 AND #CycleSelection.StepSelection.SystemDrainNoYes THEN
       #CycleStart.Started.SystemDrainStarted := TRUE;
   END_IF;
   #_w12 := #_w11 AND NOT #CycleSelection.StepSelection.SystemDrainNoYes;
   IF #_w12 AND #CycleSelection.StepSelection.AirPurgingNoYes THEN
       #CycleStart.Started.AirPurgingStarted := TRUE;
   END_IF;
   IF #_w12 AND NOT #CycleSelection.StepSelection.AirPurgingNoYes THEN #OverTemp := TRUE; END_IF;
   IF #_w10 AND (#ActualRepetition < #CycleSelection.StepSelection.SetRepetition) THEN
       #RepeatCycle := TRUE;
   END_IF;
END_REGION

REGION Network 6: TemperatureDosingOver
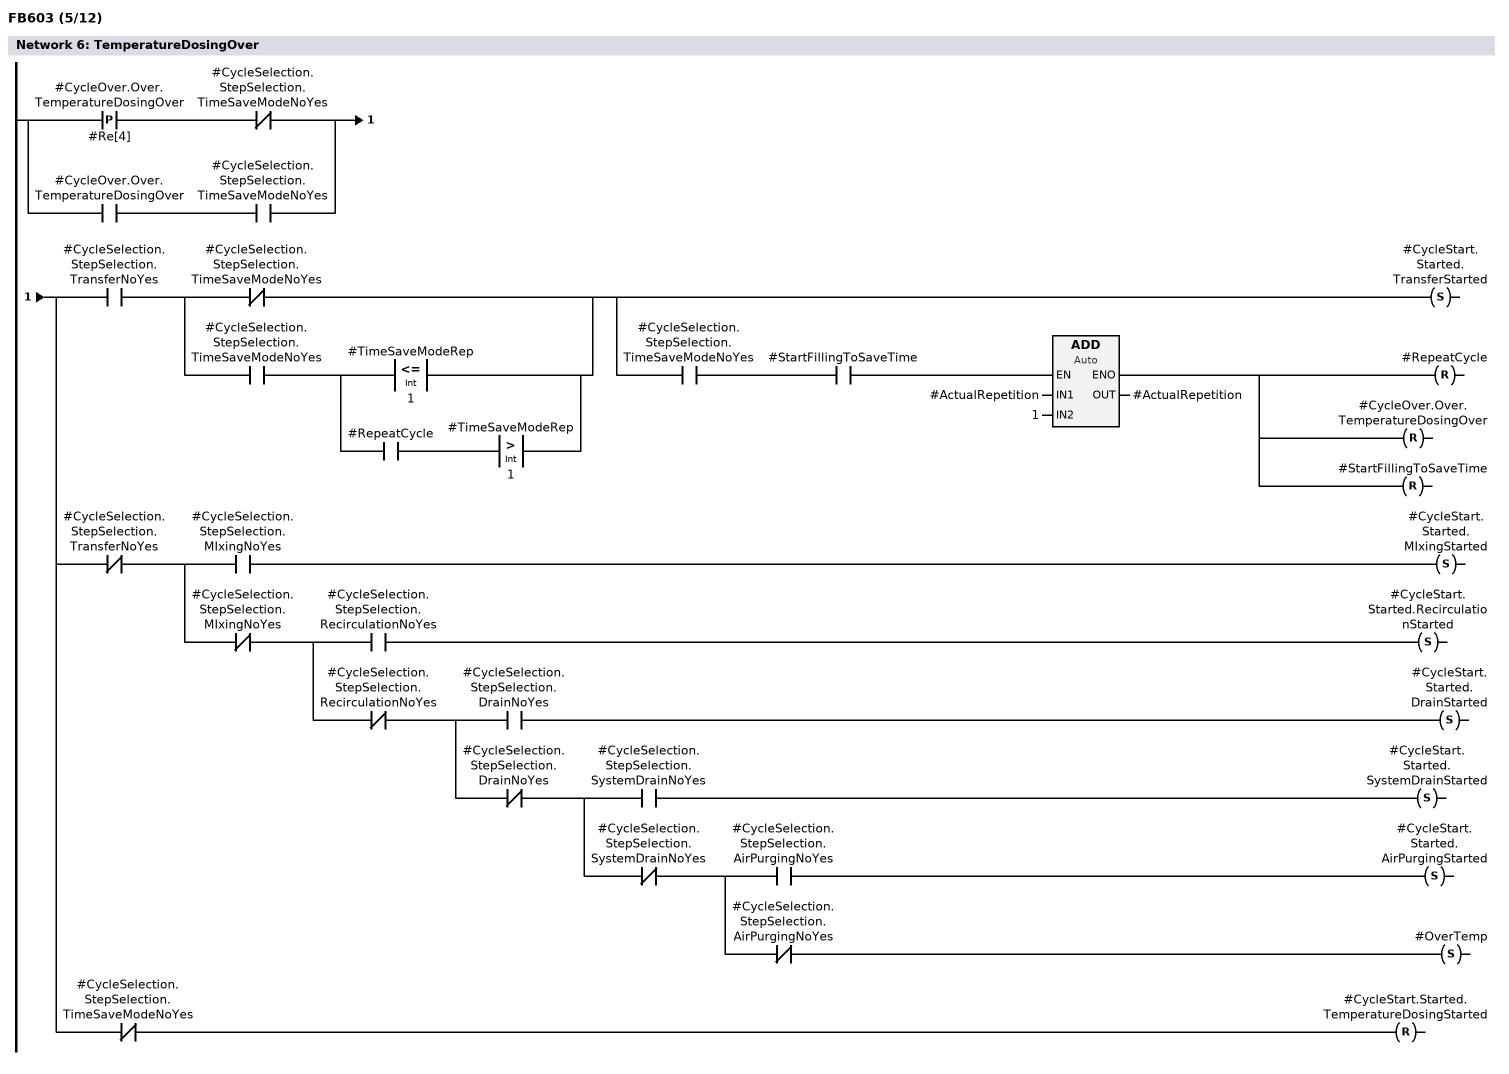
   RUNG wire#powerrail
      P_Contact(operand := #CycleOver.Over.TemperatureDosingOver, bit := #Re[4])
      I_Contact( #CycleSelection.StepSelection.TimeSaveModeNoYes )
      wire#w1
      Contact( #CycleSelection.StepSelection.TransferNoYes )
      wire#w2
      I_Contact( #CycleSelection.StepSelection.TimeSaveModeNoYes )
      wire#w3
      S_Coil( #CycleStart.Started.TransferStarted )
   END_RUNG
   RUNG wire#powerrail
      Contact( #CycleOver.Over.TemperatureDosingOver )
      Contact( #CycleSelection.StepSelection.TimeSaveModeNoYes )
   END_RUNG wire#w1
   RUNG wire#w2
      Contact( #CycleSelection.StepSelection.TimeSaveModeNoYes )
      wire#w4
      { S7_Templates := "SrcType := Int" } LE_Contact(in1 := #TimeSaveModeRep, in2 := 1)
   END_RUNG wire#w3
   RUNG wire#w4
      Contact( #RepeatCycle )
      { S7_Templates := "SrcType := Int" } GT_Contact(in1 := #TimeSaveModeRep, in2 := 1)
   END_RUNG wire#w3
   RUNG wire#w3
      Contact( #CycleSelection.StepSelection.TimeSaveModeNoYes )
      Contact( #StartFillingToSaveTime )
      Add(in1 := #ActualRepetition, in2 := 1, out => #ActualRepetition)
      wire#w5
      R_Coil( #RepeatCycle )
   END_RUNG
   RUNG wire#w5
      R_Coil( #CycleOver.Over.TemperatureDosingOver )
   END_RUNG
   RUNG wire#w5
      R_Coil( #StartFillingToSaveTime )
   END_RUNG
   RUNG wire#w1
      I_Contact( #CycleSelection.StepSelection.TransferNoYes )
      wire#w6
      Contact( #CycleSelection.StepSelection.MIxingNoYes )
      S_Coil( #CycleStart.Started.MIxingStarted )
   END_RUNG
   RUNG wire#w6
      I_Contact( #CycleSelection.StepSelection.MIxingNoYes )
      wire#w7
      Contact( #CycleSelection.StepSelection.RecirculationNoYes )
      S_Coil( #CycleStart.Started.RecirculationStarted )
   END_RUNG
   RUNG wire#w7
      I_Contact( #CycleSelection.StepSelection.RecirculationNoYes )
      wire#w8
      Contact( #CycleSelection.StepSelection.DrainNoYes )
      S_Coil( #CycleStart.Started.DrainStarted )
   END_RUNG
   RUNG wire#w8
      I_Contact( #CycleSelection.StepSelection.DrainNoYes )
      wire#w9
      Contact( #CycleSelection.StepSelection.SystemDrainNoYes )
      S_Coil( #CycleStart.Started.SystemDrainStarted )
   END_RUNG
   RUNG wire#w9
      I_Contact( #CycleSelection.StepSelection.SystemDrainNoYes )
      wire#w10
      Contact( #CycleSelection.StepSelection.AirPurgingNoYes )
      S_Coil( #CycleStart.Started.AirPurgingStarted )
   END_RUNG
   RUNG wire#w10
      I_Contact( #CycleSelection.StepSelection.AirPurgingNoYes )
      S_Coil( #OverTemp )
   END_RUNG
   RUNG wire#w1
      I_Contact( #CycleSelection.StepSelection.TimeSaveModeNoYes )
      R_Coil( #CycleStart.Started.TemperatureDosingStarted )
   END_RUNG
   // the same network as SCL:
   #_w1 := #CycleOver.Over.TemperatureDosingOver AND NOT #Re[4];   // rising edge of #CycleOver.Over.TemperatureDosingOver
   #Re[4] := #CycleOver.Over.TemperatureDosingOver;
   #_w2 := (#_w1 AND NOT #CycleSelection.StepSelection.TimeSaveModeNoYes) OR (#CycleOver.Over.TemperatureDosingOver AND #CycleSelection.StepSelection.TimeSaveModeNoYes);
   #_w3 := #_w2 AND #CycleSelection.StepSelection.TransferNoYes AND (NOT #CycleSelection.StepSelection.TimeSaveModeNoYes OR (#CycleSelection.StepSelection.TimeSaveModeNoYes AND ((#TimeSaveModeRep <= 1) OR (#RepeatCycle AND (#TimeSaveModeRep > 1)))));
   IF #_w3 THEN #CycleStart.Started.TransferStarted := TRUE; END_IF;
   IF #_w3 AND #CycleSelection.StepSelection.TimeSaveModeNoYes AND #StartFillingToSaveTime THEN
       #ActualRepetition := #ActualRepetition + 1;
       #RepeatCycle := FALSE;
       #CycleOver.Over.TemperatureDosingOver := FALSE;
       #StartFillingToSaveTime := FALSE;
   END_IF;
   #_w4 := #_w2 AND NOT #CycleSelection.StepSelection.TransferNoYes;
   IF #_w4 AND #CycleSelection.StepSelection.MIxingNoYes THEN
       #CycleStart.Started.MIxingStarted := TRUE;
   END_IF;
   #_w5 := #_w4 AND NOT #CycleSelection.StepSelection.MIxingNoYes;
   IF #_w5 AND #CycleSelection.StepSelection.RecirculationNoYes THEN
       #CycleStart.Started.RecirculationStarted := TRUE;
   END_IF;
   #_w6 := #_w5 AND NOT #CycleSelection.StepSelection.RecirculationNoYes;
   IF #_w6 AND #CycleSelection.StepSelection.DrainNoYes THEN
       #CycleStart.Started.DrainStarted := TRUE;
   END_IF;
   #_w7 := #_w6 AND NOT #CycleSelection.StepSelection.DrainNoYes;
   IF #_w7 AND #CycleSelection.StepSelection.SystemDrainNoYes THEN
       #CycleStart.Started.SystemDrainStarted := TRUE;
   END_IF;
   #_w8 := #_w7 AND NOT #CycleSelection.StepSelection.SystemDrainNoYes;
   IF #_w8 AND #CycleSelection.StepSelection.AirPurgingNoYes THEN
       #CycleStart.Started.AirPurgingStarted := TRUE;
   END_IF;
   IF #_w8 AND NOT #CycleSelection.StepSelection.AirPurgingNoYes THEN #OverTemp := TRUE; END_IF;
   IF #_w2 AND NOT #CycleSelection.StepSelection.TimeSaveModeNoYes THEN
       #CycleStart.Started.TemperatureDosingStarted := FALSE;
   END_IF;
END_REGION

REGION Network 7: TransferOver
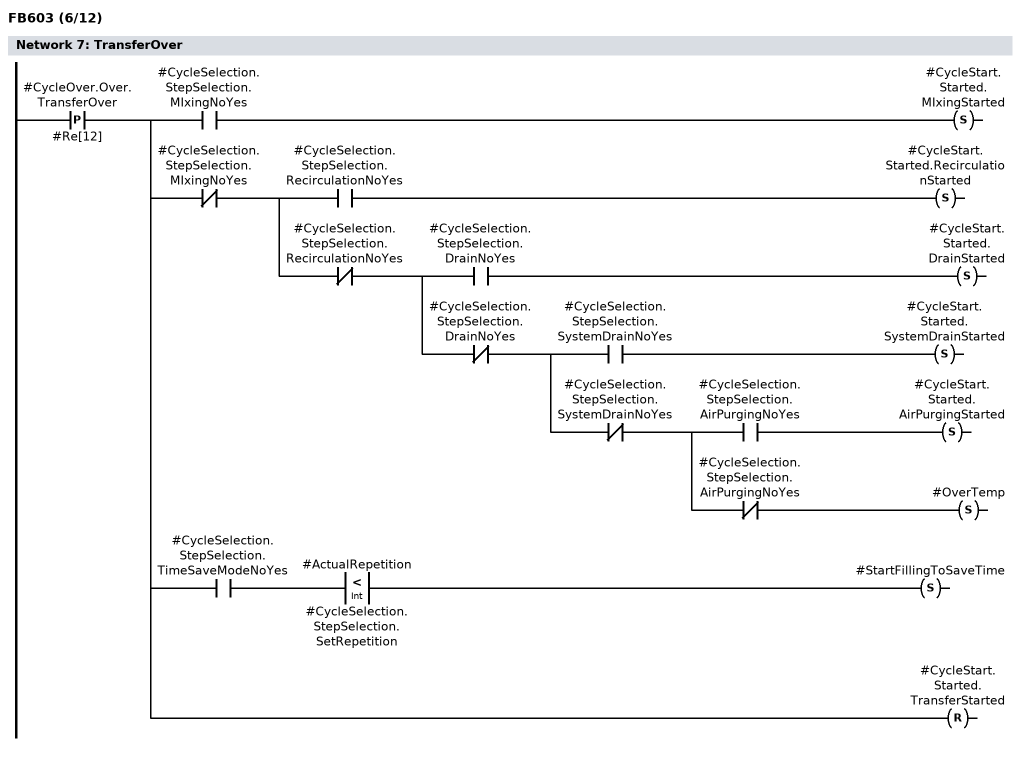
   RUNG wire#powerrail
      P_Contact(operand := #CycleOver.Over.TransferOver, bit := #Re[12])
      wire#w1
      Contact( #CycleSelection.StepSelection.MIxingNoYes )
      S_Coil( #CycleStart.Started.MIxingStarted )
   END_RUNG
   RUNG wire#w1
      I_Contact( #CycleSelection.StepSelection.MIxingNoYes )
      wire#w2
      Contact( #CycleSelection.StepSelection.RecirculationNoYes )
      S_Coil( #CycleStart.Started.RecirculationStarted )
   END_RUNG
   RUNG wire#w2
      I_Contact( #CycleSelection.StepSelection.RecirculationNoYes )
      wire#w3
      Contact( #CycleSelection.StepSelection.DrainNoYes )
      S_Coil( #CycleStart.Started.DrainStarted )
   END_RUNG
   RUNG wire#w3
      I_Contact( #CycleSelection.StepSelection.DrainNoYes )
      wire#w4
      Contact( #CycleSelection.StepSelection.SystemDrainNoYes )
      S_Coil( #CycleStart.Started.SystemDrainStarted )
   END_RUNG
   RUNG wire#w4
      I_Contact( #CycleSelection.StepSelection.SystemDrainNoYes )
      wire#w5
      Contact( #CycleSelection.StepSelection.AirPurgingNoYes )
      S_Coil( #CycleStart.Started.AirPurgingStarted )
   END_RUNG
   RUNG wire#w5
      I_Contact( #CycleSelection.StepSelection.AirPurgingNoYes )
      S_Coil( #OverTemp )
   END_RUNG
   RUNG wire#w1
      Contact( #CycleSelection.StepSelection.TimeSaveModeNoYes )
      { S7_Templates := "SrcType := Int" } LT_Contact(in1 := #ActualRepetition, in2 := #CycleSelection.StepSelection.SetRepetition)
      S_Coil( #StartFillingToSaveTime )
   END_RUNG
   RUNG wire#w1
      R_Coil( #CycleStart.Started.TransferStarted )
   END_RUNG
   // the same network as SCL:
   #_w1 := #CycleOver.Over.TransferOver AND NOT #Re[12];   // rising edge of #CycleOver.Over.TransferOver
   #Re[12] := #CycleOver.Over.TransferOver;
   IF #_w1 AND #CycleSelection.StepSelection.MIxingNoYes THEN
       #CycleStart.Started.MIxingStarted := TRUE;
   END_IF;
   #_w2 := #_w1 AND NOT #CycleSelection.StepSelection.MIxingNoYes;
   IF #_w2 AND #CycleSelection.StepSelection.RecirculationNoYes THEN
       #CycleStart.Started.RecirculationStarted := TRUE;
   END_IF;
   #_w3 := #_w2 AND NOT #CycleSelection.StepSelection.RecirculationNoYes;
   IF #_w3 AND #CycleSelection.StepSelection.DrainNoYes THEN
       #CycleStart.Started.DrainStarted := TRUE;
   END_IF;
   #_w4 := #_w3 AND NOT #CycleSelection.StepSelection.DrainNoYes;
   IF #_w4 AND #CycleSelection.StepSelection.SystemDrainNoYes THEN
       #CycleStart.Started.SystemDrainStarted := TRUE;
   END_IF;
   #_w5 := #_w4 AND NOT #CycleSelection.StepSelection.SystemDrainNoYes;
   IF #_w5 AND #CycleSelection.StepSelection.AirPurgingNoYes THEN
       #CycleStart.Started.AirPurgingStarted := TRUE;
   END_IF;
   IF #_w5 AND NOT #CycleSelection.StepSelection.AirPurgingNoYes THEN #OverTemp := TRUE; END_IF;
   IF #_w1 AND #CycleSelection.StepSelection.TimeSaveModeNoYes AND (#ActualRepetition < #CycleSelection.StepSelection.SetRepetition) THEN
       #StartFillingToSaveTime := TRUE;
   END_IF;
   IF #_w1 THEN #CycleStart.Started.TransferStarted := FALSE; END_IF;
END_REGION

REGION Network 8: TransferOver
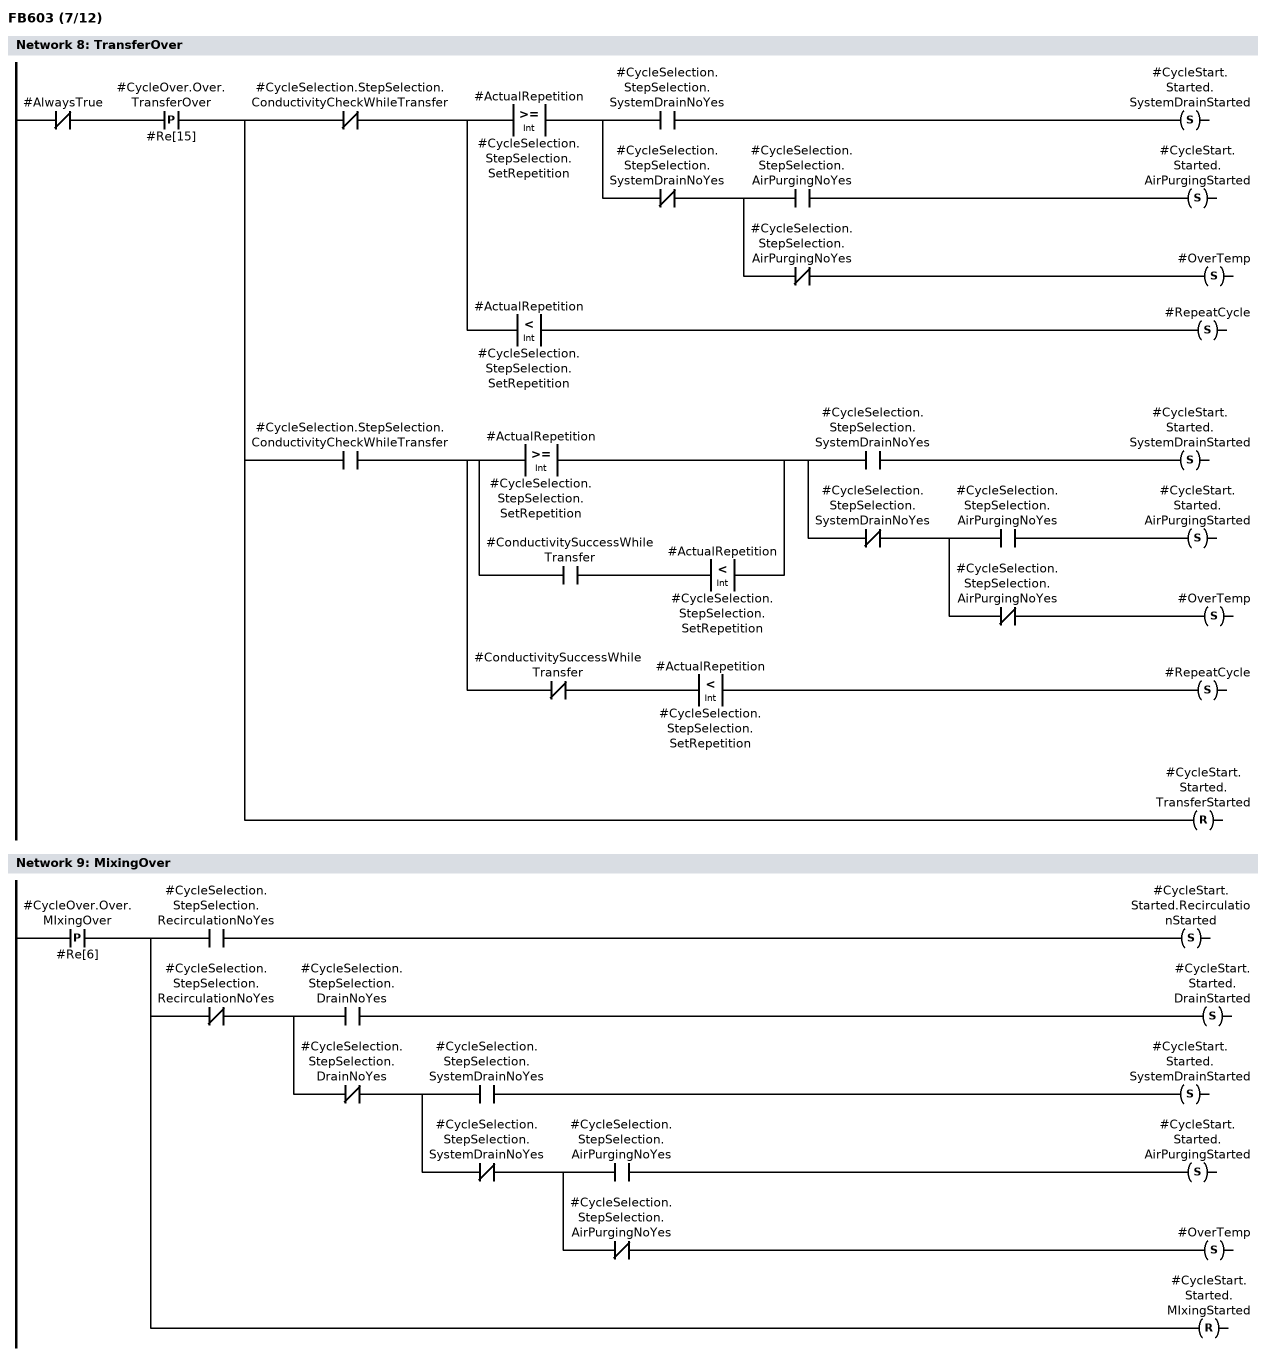
   RUNG wire#powerrail
      I_Contact( #AlwaysTrue )
      P_Contact(operand := #CycleOver.Over.TransferOver, bit := #Re[15])
      wire#w1
      I_Contact( #CycleSelection.StepSelection.ConductivityCheckWhileTransfer )
      wire#w2
      { S7_Templates := "SrcType := Int" } GE_Contact(in1 := #ActualRepetition, in2 := #CycleSelection.StepSelection.SetRepetition)
      wire#w3
      Contact( #CycleSelection.StepSelection.SystemDrainNoYes )
      S_Coil( #CycleStart.Started.SystemDrainStarted )
   END_RUNG
   RUNG wire#w3
      I_Contact( #CycleSelection.StepSelection.SystemDrainNoYes )
      wire#w4
      Contact( #CycleSelection.StepSelection.AirPurgingNoYes )
      S_Coil( #CycleStart.Started.AirPurgingStarted )
   END_RUNG
   RUNG wire#w4
      I_Contact( #CycleSelection.StepSelection.AirPurgingNoYes )
      S_Coil( #OverTemp )
   END_RUNG
   RUNG wire#w2
      { S7_Templates := "SrcType := Int" } LT_Contact(in1 := #ActualRepetition, in2 := #CycleSelection.StepSelection.SetRepetition)
      S_Coil( #RepeatCycle )
   END_RUNG
   RUNG wire#w1
      Contact( #CycleSelection.StepSelection.ConductivityCheckWhileTransfer )
      wire#w5
      { S7_Templates := "SrcType := Int" } GE_Contact(in1 := #ActualRepetition, in2 := #CycleSelection.StepSelection.SetRepetition)
      wire#w6
      Contact( #CycleSelection.StepSelection.SystemDrainNoYes )
      S_Coil( #CycleStart.Started.SystemDrainStarted )
   END_RUNG
   RUNG wire#w5
      Contact( #ConductivitySuccessWhileTransfer )
      { S7_Templates := "SrcType := Int" } LT_Contact(in1 := #ActualRepetition, in2 := #CycleSelection.StepSelection.SetRepetition)
   END_RUNG wire#w6
   RUNG wire#w6
      I_Contact( #CycleSelection.StepSelection.SystemDrainNoYes )
      wire#w7
      Contact( #CycleSelection.StepSelection.AirPurgingNoYes )
      S_Coil( #CycleStart.Started.AirPurgingStarted )
   END_RUNG
   RUNG wire#w7
      I_Contact( #CycleSelection.StepSelection.AirPurgingNoYes )
      S_Coil( #OverTemp )
   END_RUNG
   RUNG wire#w5
      I_Contact( #ConductivitySuccessWhileTransfer )
      { S7_Templates := "SrcType := Int" } LT_Contact(in1 := #ActualRepetition, in2 := #CycleSelection.StepSelection.SetRepetition)
      S_Coil( #RepeatCycle )
   END_RUNG
   RUNG wire#w1
      R_Coil( #CycleStart.Started.TransferStarted )
   END_RUNG
   // the same network as SCL:
   #_w1 := NOT #AlwaysTrue AND #CycleOver.Over.TransferOver AND NOT #Re[15];   // rising edge of #CycleOver.Over.TransferOver
   #Re[15] := #CycleOver.Over.TransferOver;
   #_w2 := #_w1 AND NOT #CycleSelection.StepSelection.ConductivityCheckWhileTransfer;
   #_w3 := #_w2 AND (#ActualRepetition >= #CycleSelection.StepSelection.SetRepetition);
   IF #_w3 AND #CycleSelection.StepSelection.SystemDrainNoYes THEN
       #CycleStart.Started.SystemDrainStarted := TRUE;
   END_IF;
   #_w4 := #_w3 AND NOT #CycleSelection.StepSelection.SystemDrainNoYes;
   IF #_w4 AND #CycleSelection.StepSelection.AirPurgingNoYes THEN
       #CycleStart.Started.AirPurgingStarted := TRUE;
   END_IF;
   IF #_w4 AND NOT #CycleSelection.StepSelection.AirPurgingNoYes THEN #OverTemp := TRUE; END_IF;
   IF #_w2 AND (#ActualRepetition < #CycleSelection.StepSelection.SetRepetition) THEN
       #RepeatCycle := TRUE;
   END_IF;
   #_w5 := #_w1 AND #CycleSelection.StepSelection.ConductivityCheckWhileTransfer;
   #_w6 := #_w5 AND ((#ActualRepetition >= #CycleSelection.StepSelection.SetRepetition) OR (#ConductivitySuccessWhileTransfer AND (#ActualRepetition < #CycleSelection.StepSelection.SetRepetition)));
   IF #_w6 AND #CycleSelection.StepSelection.SystemDrainNoYes THEN
       #CycleStart.Started.SystemDrainStarted := TRUE;
   END_IF;
   #_w7 := #_w6 AND NOT #CycleSelection.StepSelection.SystemDrainNoYes;
   IF #_w7 AND #CycleSelection.StepSelection.AirPurgingNoYes THEN
       #CycleStart.Started.AirPurgingStarted := TRUE;
   END_IF;
   IF #_w7 AND NOT #CycleSelection.StepSelection.AirPurgingNoYes THEN #OverTemp := TRUE; END_IF;
   IF #_w5 AND NOT #ConductivitySuccessWhileTransfer AND (#ActualRepetition < #CycleSelection.StepSelection.SetRepetition) THEN
       #RepeatCycle := TRUE;
   END_IF;
   IF #_w1 THEN #CycleStart.Started.TransferStarted := FALSE; END_IF;
END_REGION

REGION Network 9: MixingOver
   RUNG wire#powerrail
      P_Contact(operand := #CycleOver.Over.MIxingOver, bit := #Re[6])
      wire#w1
      Contact( #CycleSelection.StepSelection.RecirculationNoYes )
      S_Coil( #CycleStart.Started.RecirculationStarted )
   END_RUNG
   RUNG wire#w1
      I_Contact( #CycleSelection.StepSelection.RecirculationNoYes )
      wire#w2
      Contact( #CycleSelection.StepSelection.DrainNoYes )
      S_Coil( #CycleStart.Started.DrainStarted )
   END_RUNG
   RUNG wire#w2
      I_Contact( #CycleSelection.StepSelection.DrainNoYes )
      wire#w3
      Contact( #CycleSelection.StepSelection.SystemDrainNoYes )
      S_Coil( #CycleStart.Started.SystemDrainStarted )
   END_RUNG
   RUNG wire#w3
      I_Contact( #CycleSelection.StepSelection.SystemDrainNoYes )
      wire#w4
      Contact( #CycleSelection.StepSelection.AirPurgingNoYes )
      S_Coil( #CycleStart.Started.AirPurgingStarted )
   END_RUNG
   RUNG wire#w4
      I_Contact( #CycleSelection.StepSelection.AirPurgingNoYes )
      S_Coil( #OverTemp )
   END_RUNG
   RUNG wire#w1
      R_Coil( #CycleStart.Started.MIxingStarted )
   END_RUNG
   // the same network as SCL:
   #_w1 := #CycleOver.Over.MIxingOver AND NOT #Re[6];   // rising edge of #CycleOver.Over.MIxingOver
   #Re[6] := #CycleOver.Over.MIxingOver;
   IF #_w1 AND #CycleSelection.StepSelection.RecirculationNoYes THEN
       #CycleStart.Started.RecirculationStarted := TRUE;
   END_IF;
   #_w2 := #_w1 AND NOT #CycleSelection.StepSelection.RecirculationNoYes;
   IF #_w2 AND #CycleSelection.StepSelection.DrainNoYes THEN
       #CycleStart.Started.DrainStarted := TRUE;
   END_IF;
   #_w3 := #_w2 AND NOT #CycleSelection.StepSelection.DrainNoYes;
   IF #_w3 AND #CycleSelection.StepSelection.SystemDrainNoYes THEN
       #CycleStart.Started.SystemDrainStarted := TRUE;
   END_IF;
   #_w4 := #_w3 AND NOT #CycleSelection.StepSelection.SystemDrainNoYes;
   IF #_w4 AND #CycleSelection.StepSelection.AirPurgingNoYes THEN
       #CycleStart.Started.AirPurgingStarted := TRUE;
   END_IF;
   IF #_w4 AND NOT #CycleSelection.StepSelection.AirPurgingNoYes THEN #OverTemp := TRUE; END_IF;
   IF #_w1 THEN #CycleStart.Started.MIxingStarted := FALSE; END_IF;
END_REGION

REGION Network 10: RecirculationOver
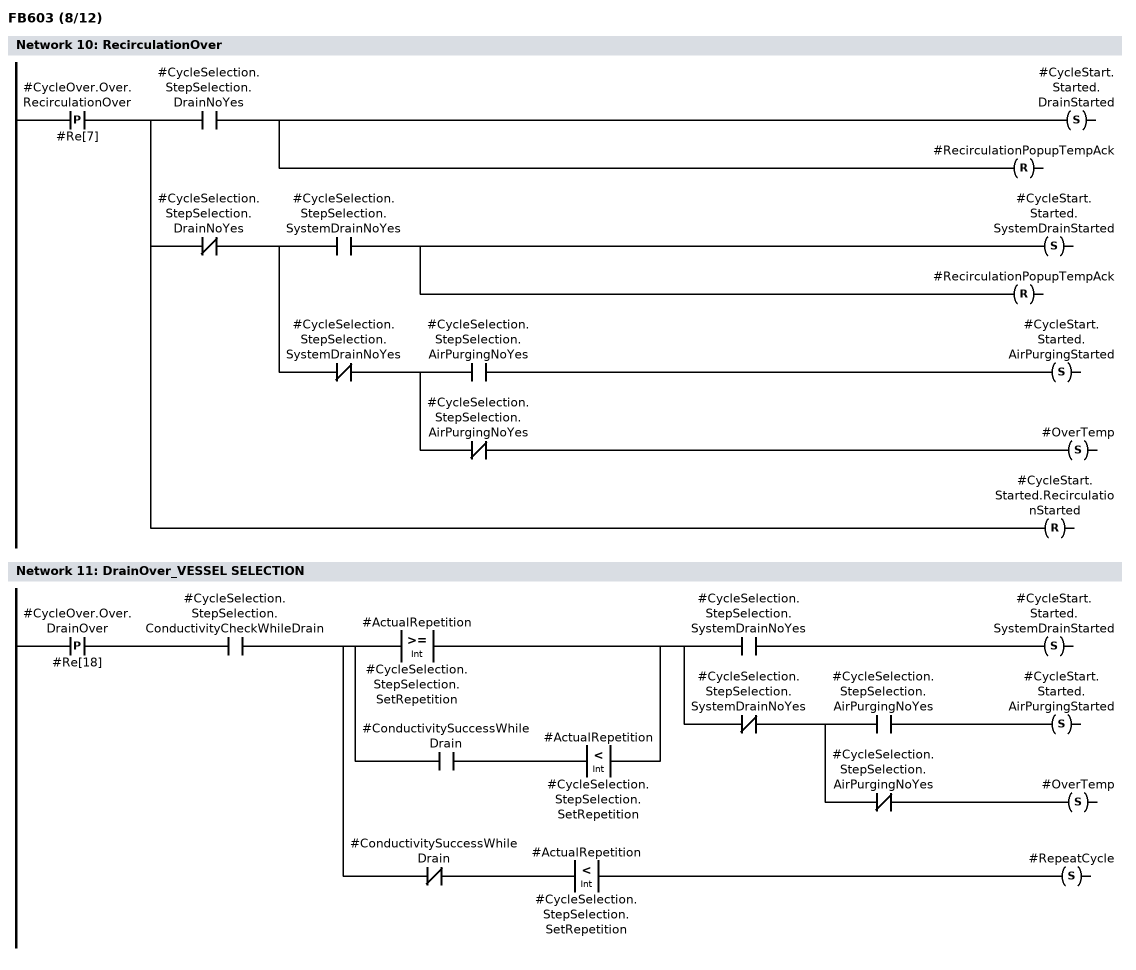
   RUNG wire#powerrail
      P_Contact(operand := #CycleOver.Over.RecirculationOver, bit := #Re[7])
      wire#w1
      Contact( #CycleSelection.StepSelection.DrainNoYes )
      wire#w2
      S_Coil( #CycleStart.Started.DrainStarted )
   END_RUNG
   RUNG wire#w2
      R_Coil( #RecirculationPopupTempAck )
   END_RUNG
   RUNG wire#w1
      I_Contact( #CycleSelection.StepSelection.DrainNoYes )
      wire#w3
      Contact( #CycleSelection.StepSelection.SystemDrainNoYes )
      wire#w4
      S_Coil( #CycleStart.Started.SystemDrainStarted )
   END_RUNG
   RUNG wire#w4
      R_Coil( #RecirculationPopupTempAck )
   END_RUNG
   RUNG wire#w3
      I_Contact( #CycleSelection.StepSelection.SystemDrainNoYes )
      wire#w5
      Contact( #CycleSelection.StepSelection.AirPurgingNoYes )
      S_Coil( #CycleStart.Started.AirPurgingStarted )
   END_RUNG
   RUNG wire#w5
      I_Contact( #CycleSelection.StepSelection.AirPurgingNoYes )
      S_Coil( #OverTemp )
   END_RUNG
   RUNG wire#w1
      R_Coil( #CycleStart.Started.RecirculationStarted )
   END_RUNG
   // the same network as SCL:
   #_w1 := #CycleOver.Over.RecirculationOver AND NOT #Re[7];   // rising edge of #CycleOver.Over.RecirculationOver
   #Re[7] := #CycleOver.Over.RecirculationOver;
   IF #_w1 AND #CycleSelection.StepSelection.DrainNoYes THEN
       #CycleStart.Started.DrainStarted := TRUE;
       #RecirculationPopupTempAck := FALSE;
   END_IF;
   #_w2 := #_w1 AND NOT #CycleSelection.StepSelection.DrainNoYes;
   IF #_w2 AND #CycleSelection.StepSelection.SystemDrainNoYes THEN
       #CycleStart.Started.SystemDrainStarted := TRUE;
       #RecirculationPopupTempAck := FALSE;
   END_IF;
   #_w3 := #_w2 AND NOT #CycleSelection.StepSelection.SystemDrainNoYes;
   IF #_w3 AND #CycleSelection.StepSelection.AirPurgingNoYes THEN
       #CycleStart.Started.AirPurgingStarted := TRUE;
   END_IF;
   IF #_w3 AND NOT #CycleSelection.StepSelection.AirPurgingNoYes THEN #OverTemp := TRUE; END_IF;
   IF #_w1 THEN #CycleStart.Started.RecirculationStarted := FALSE; END_IF;
END_REGION

REGION Network 11: DrainOver_VESSEL SELECTION
   RUNG wire#powerrail
      P_Contact(operand := #CycleOver.Over.DrainOver, bit := #Re[18])
      Contact( #CycleSelection.StepSelection.ConductivityCheckWhileDrain )
      wire#w1
      { S7_Templates := "SrcType := Int" } GE_Contact(in1 := #ActualRepetition, in2 := #CycleSelection.StepSelection.SetRepetition)
      wire#w2
      Contact( #CycleSelection.StepSelection.SystemDrainNoYes )
      S_Coil( #CycleStart.Started.SystemDrainStarted )
   END_RUNG
   RUNG wire#w1
      Contact( #ConductivitySuccessWhileDrain )
      { S7_Templates := "SrcType := Int" } LT_Contact(in1 := #ActualRepetition, in2 := #CycleSelection.StepSelection.SetRepetition)
   END_RUNG wire#w2
   RUNG wire#w2
      I_Contact( #CycleSelection.StepSelection.SystemDrainNoYes )
      wire#w3
      Contact( #CycleSelection.StepSelection.AirPurgingNoYes )
      S_Coil( #CycleStart.Started.AirPurgingStarted )
   END_RUNG
   RUNG wire#w3
      I_Contact( #CycleSelection.StepSelection.AirPurgingNoYes )
      S_Coil( #OverTemp )
   END_RUNG
   RUNG wire#w1
      I_Contact( #ConductivitySuccessWhileDrain )
      { S7_Templates := "SrcType := Int" } LT_Contact(in1 := #ActualRepetition, in2 := #CycleSelection.StepSelection.SetRepetition)
      S_Coil( #RepeatCycle )
   END_RUNG
   // the same network as SCL:
   #_w1 := #CycleOver.Over.DrainOver AND NOT #Re[18];   // rising edge of #CycleOver.Over.DrainOver
   #Re[18] := #CycleOver.Over.DrainOver;
   #_w2 := #_w1 AND #CycleSelection.StepSelection.ConductivityCheckWhileDrain;
   #_w3 := #_w2 AND ((#ActualRepetition >= #CycleSelection.StepSelection.SetRepetition) OR (#ConductivitySuccessWhileDrain AND (#ActualRepetition < #CycleSelection.StepSelection.SetRepetition)));
   IF #_w3 AND #CycleSelection.StepSelection.SystemDrainNoYes THEN
       #CycleStart.Started.SystemDrainStarted := TRUE;
   END_IF;
   #_w4 := #_w3 AND NOT #CycleSelection.StepSelection.SystemDrainNoYes;
   IF #_w4 AND #CycleSelection.StepSelection.AirPurgingNoYes THEN
       #CycleStart.Started.AirPurgingStarted := TRUE;
   END_IF;
   IF #_w4 AND NOT #CycleSelection.StepSelection.AirPurgingNoYes THEN #OverTemp := TRUE; END_IF;
   IF #_w2 AND NOT #ConductivitySuccessWhileDrain AND (#ActualRepetition < #CycleSelection.StepSelection.SetRepetition) THEN
       #RepeatCycle := TRUE;
   END_IF;
END_REGION

REGION Network 12: DRAIN OVER (WITHOUT CONDUCTIVITY SEL.)
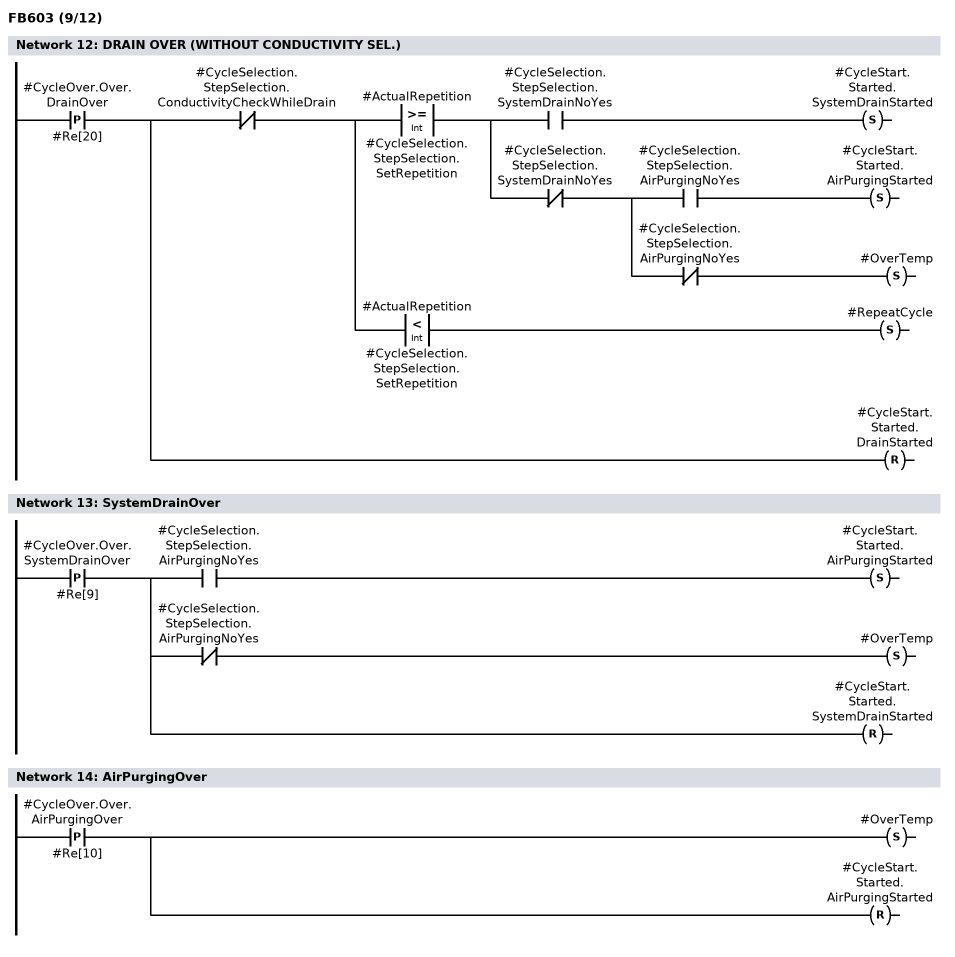
   RUNG wire#powerrail
      P_Contact(operand := #CycleOver.Over.DrainOver, bit := #Re[20])
      wire#w1
      I_Contact( #CycleSelection.StepSelection.ConductivityCheckWhileDrain )
      wire#w2
      { S7_Templates := "SrcType := Int" } GE_Contact(in1 := #ActualRepetition, in2 := #CycleSelection.StepSelection.SetRepetition)
      wire#w3
      Contact( #CycleSelection.StepSelection.SystemDrainNoYes )
      S_Coil( #CycleStart.Started.SystemDrainStarted )
   END_RUNG
   RUNG wire#w3
      I_Contact( #CycleSelection.StepSelection.SystemDrainNoYes )
      wire#w4
      Contact( #CycleSelection.StepSelection.AirPurgingNoYes )
      S_Coil( #CycleStart.Started.AirPurgingStarted )
   END_RUNG
   RUNG wire#w4
      I_Contact( #CycleSelection.StepSelection.AirPurgingNoYes )
      S_Coil( #OverTemp )
   END_RUNG
   RUNG wire#w2
      { S7_Templates := "SrcType := Int" } LT_Contact(in1 := #ActualRepetition, in2 := #CycleSelection.StepSelection.SetRepetition)
      S_Coil( #RepeatCycle )
   END_RUNG
   RUNG wire#w1
      R_Coil( #CycleStart.Started.DrainStarted )
   END_RUNG
   // the same network as SCL:
   #_w1 := #CycleOver.Over.DrainOver AND NOT #Re[20];   // rising edge of #CycleOver.Over.DrainOver
   #Re[20] := #CycleOver.Over.DrainOver;
   #_w2 := #_w1 AND NOT #CycleSelection.StepSelection.ConductivityCheckWhileDrain;
   #_w3 := #_w2 AND (#ActualRepetition >= #CycleSelection.StepSelection.SetRepetition);
   IF #_w3 AND #CycleSelection.StepSelection.SystemDrainNoYes THEN
       #CycleStart.Started.SystemDrainStarted := TRUE;
   END_IF;
   #_w4 := #_w3 AND NOT #CycleSelection.StepSelection.SystemDrainNoYes;
   IF #_w4 AND #CycleSelection.StepSelection.AirPurgingNoYes THEN
       #CycleStart.Started.AirPurgingStarted := TRUE;
   END_IF;
   IF #_w4 AND NOT #CycleSelection.StepSelection.AirPurgingNoYes THEN #OverTemp := TRUE; END_IF;
   IF #_w2 AND (#ActualRepetition < #CycleSelection.StepSelection.SetRepetition) THEN
       #RepeatCycle := TRUE;
   END_IF;
   IF #_w1 THEN #CycleStart.Started.DrainStarted := FALSE; END_IF;
END_REGION

REGION Network 13: SystemDrainOver
   RUNG wire#powerrail
      P_Contact(operand := #CycleOver.Over.SystemDrainOver, bit := #Re[9])
      wire#w1
      Contact( #CycleSelection.StepSelection.AirPurgingNoYes )
      S_Coil( #CycleStart.Started.AirPurgingStarted )
   END_RUNG
   RUNG wire#w1
      I_Contact( #CycleSelection.StepSelection.AirPurgingNoYes )
      S_Coil( #OverTemp )
   END_RUNG
   RUNG wire#w1
      R_Coil( #CycleStart.Started.SystemDrainStarted )
   END_RUNG
   // the same network as SCL:
   #_w1 := #CycleOver.Over.SystemDrainOver AND NOT #Re[9];   // rising edge of #CycleOver.Over.SystemDrainOver
   #Re[9] := #CycleOver.Over.SystemDrainOver;
   IF #_w1 AND #CycleSelection.StepSelection.AirPurgingNoYes THEN
       #CycleStart.Started.AirPurgingStarted := TRUE;
   END_IF;
   IF #_w1 AND NOT #CycleSelection.StepSelection.AirPurgingNoYes THEN #OverTemp := TRUE; END_IF;
   IF #_w1 THEN #CycleStart.Started.SystemDrainStarted := FALSE; END_IF;
END_REGION

REGION Network 14: AirPurgingOver
   RUNG wire#powerrail
      P_Contact(operand := #CycleOver.Over.AirPurgingOver, bit := #Re[10])
      wire#w1
      S_Coil( #OverTemp )
   END_RUNG
   RUNG wire#w1
      R_Coil( #CycleStart.Started.AirPurgingStarted )
   END_RUNG
   // the same network as SCL:
   #_w1 := #CycleOver.Over.AirPurgingOver AND NOT #Re[10];   // rising edge of #CycleOver.Over.AirPurgingOver
   #Re[10] := #CycleOver.Over.AirPurgingOver;
   IF #_w1 THEN
       #OverTemp := TRUE;
       #CycleStart.Started.AirPurgingStarted := FALSE;
   END_IF;
END_REGION

REGION Network 15: Reset
